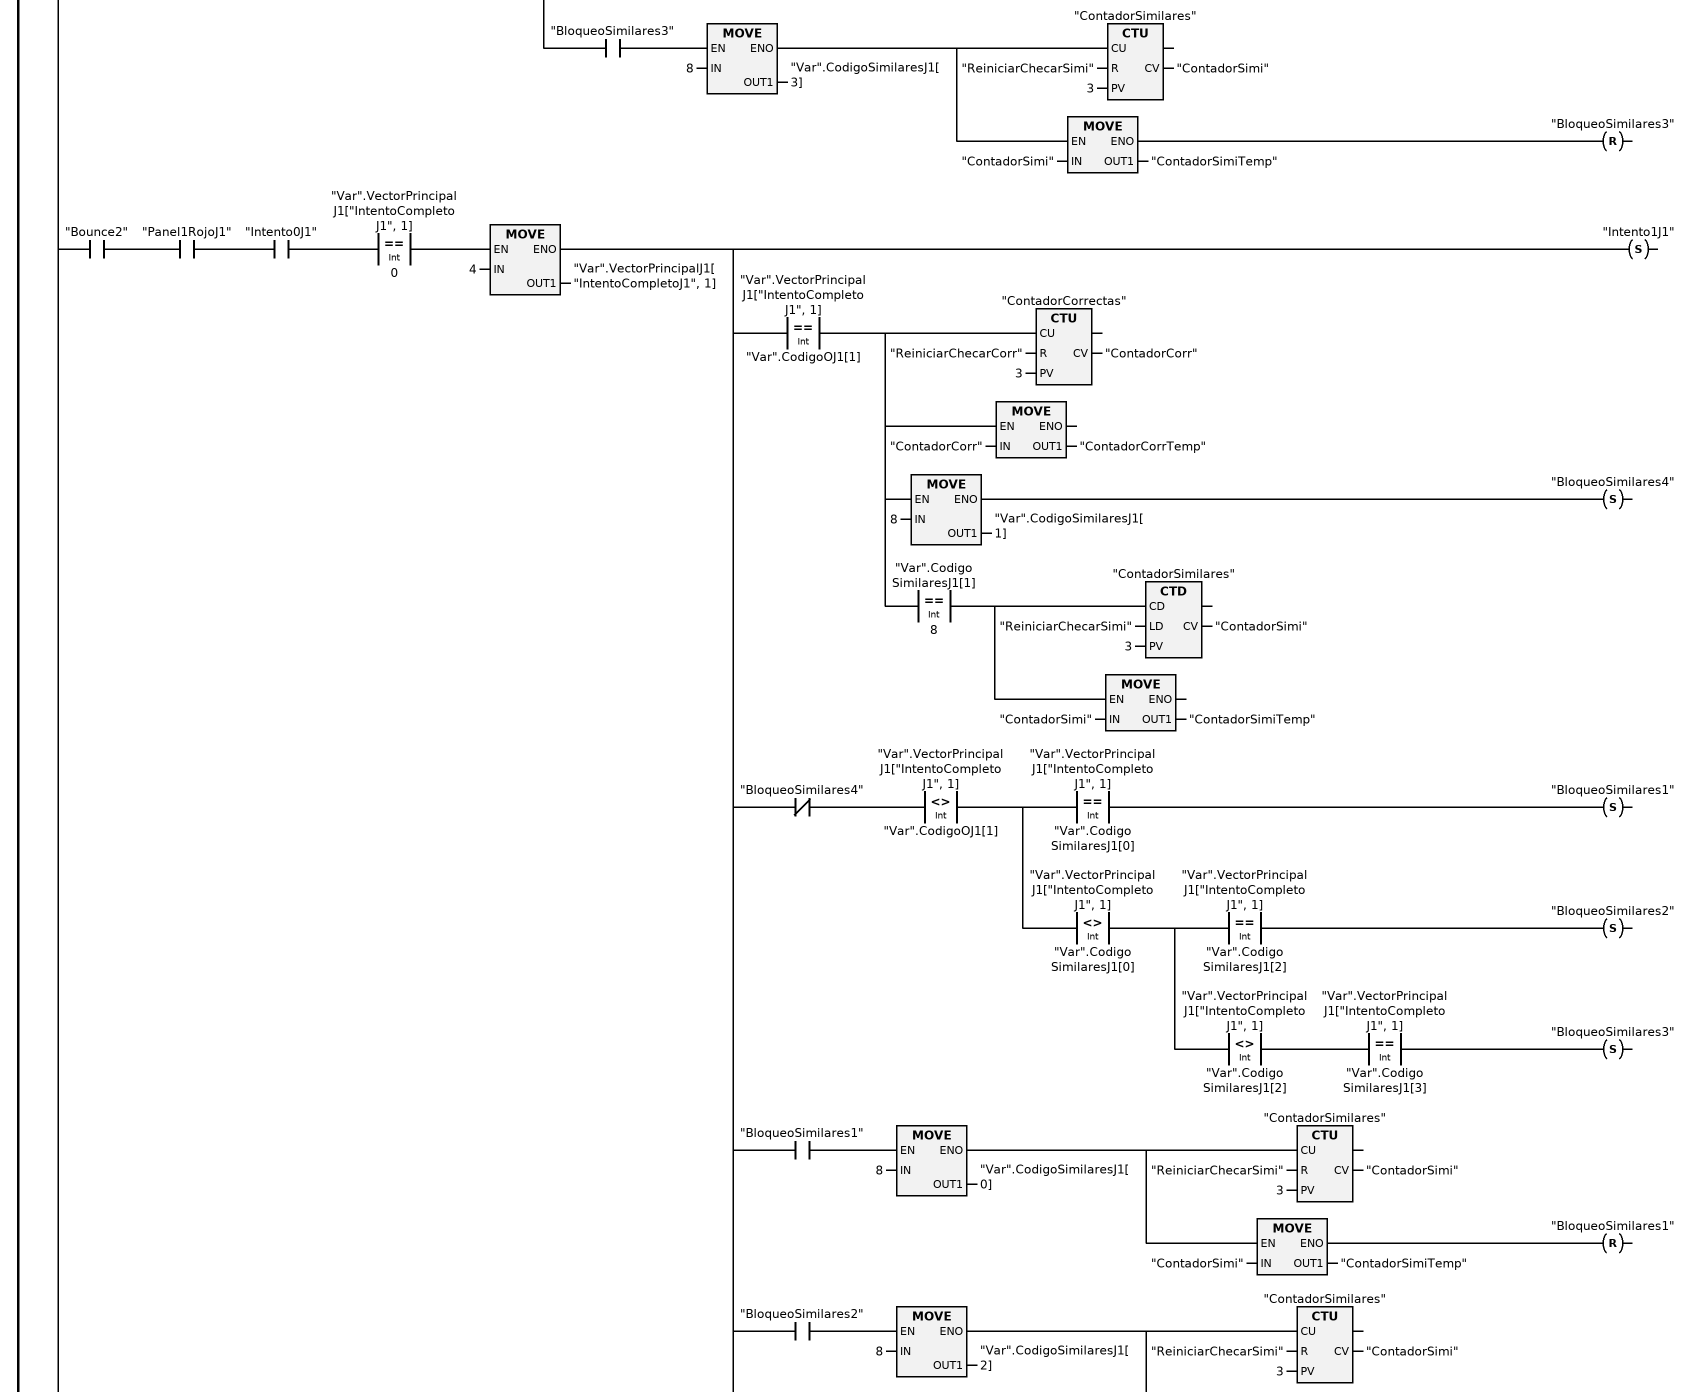
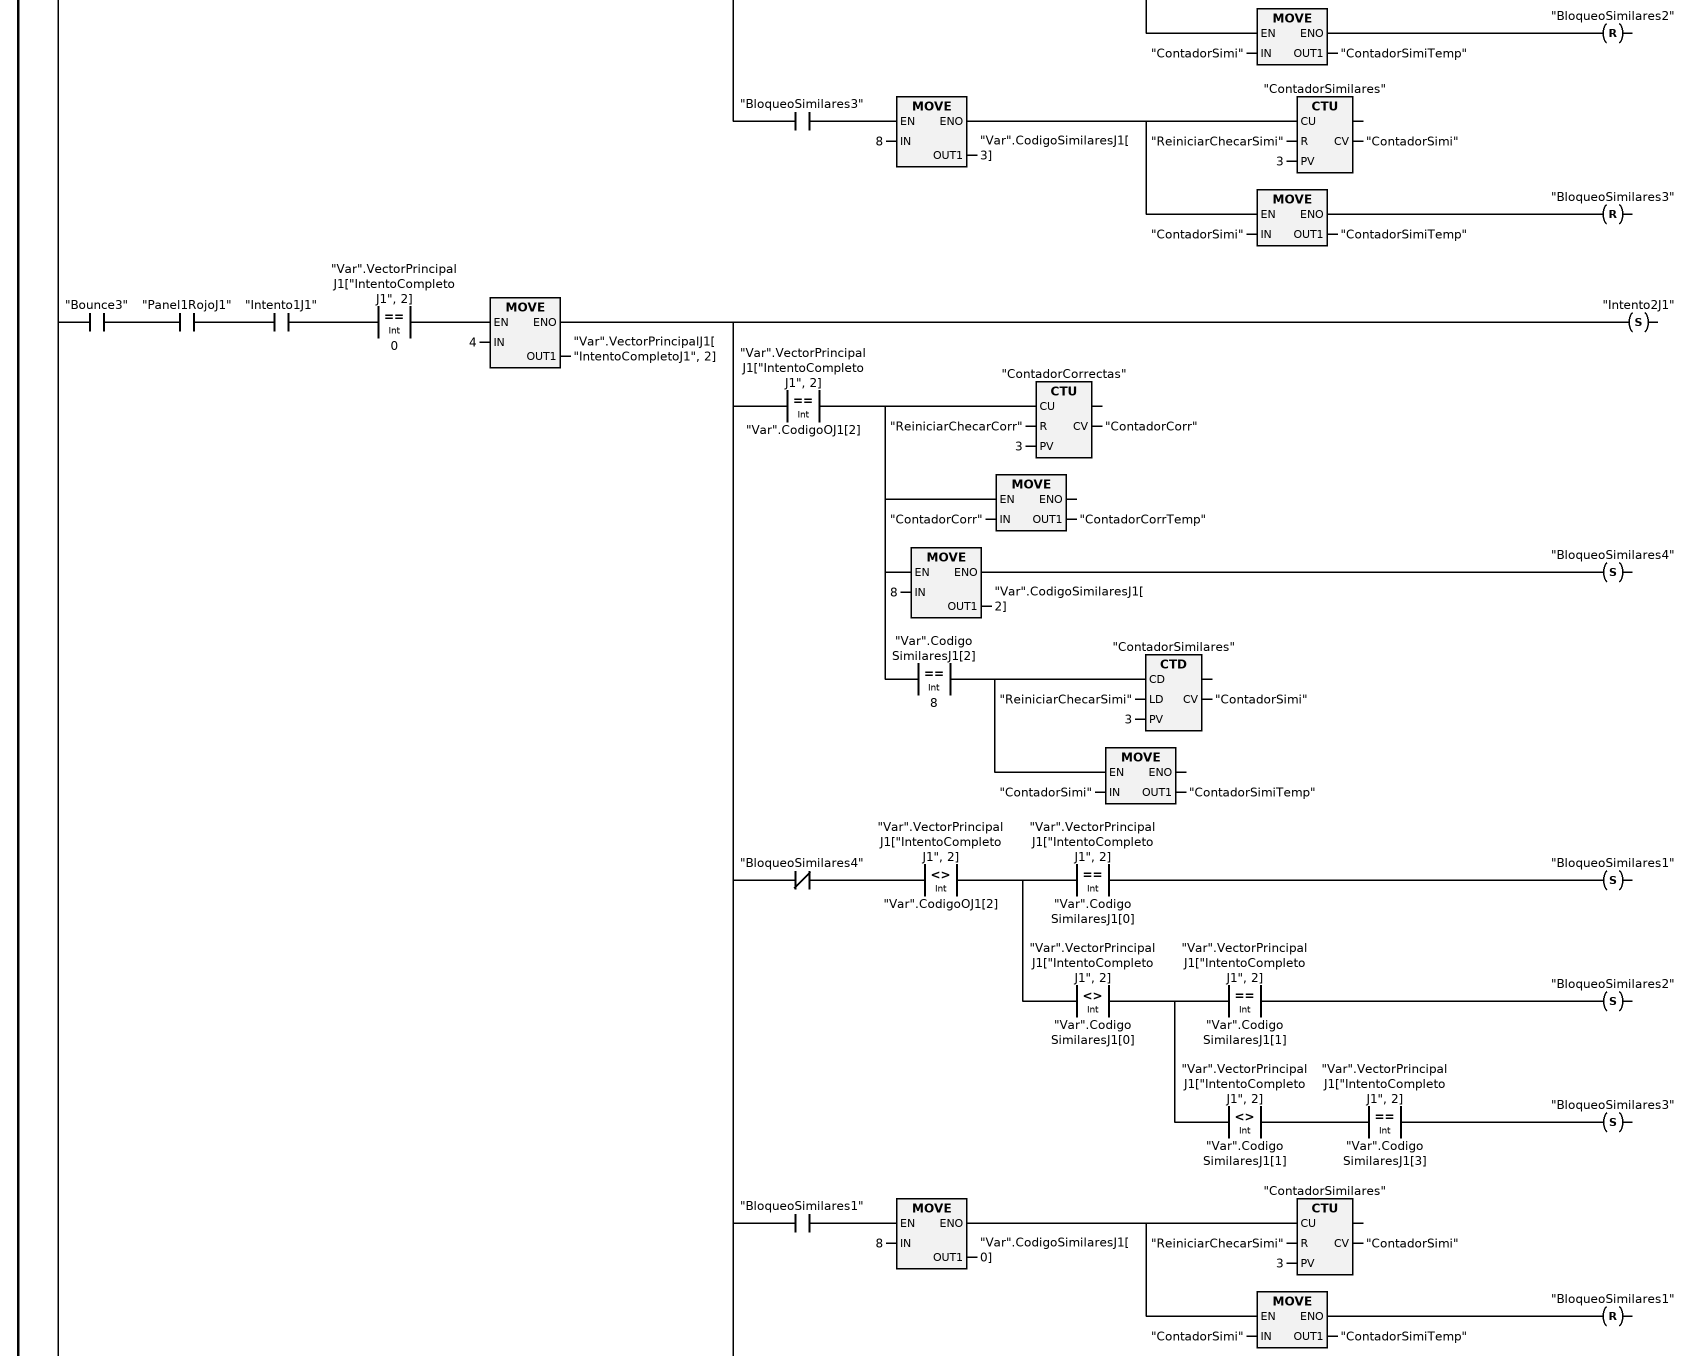
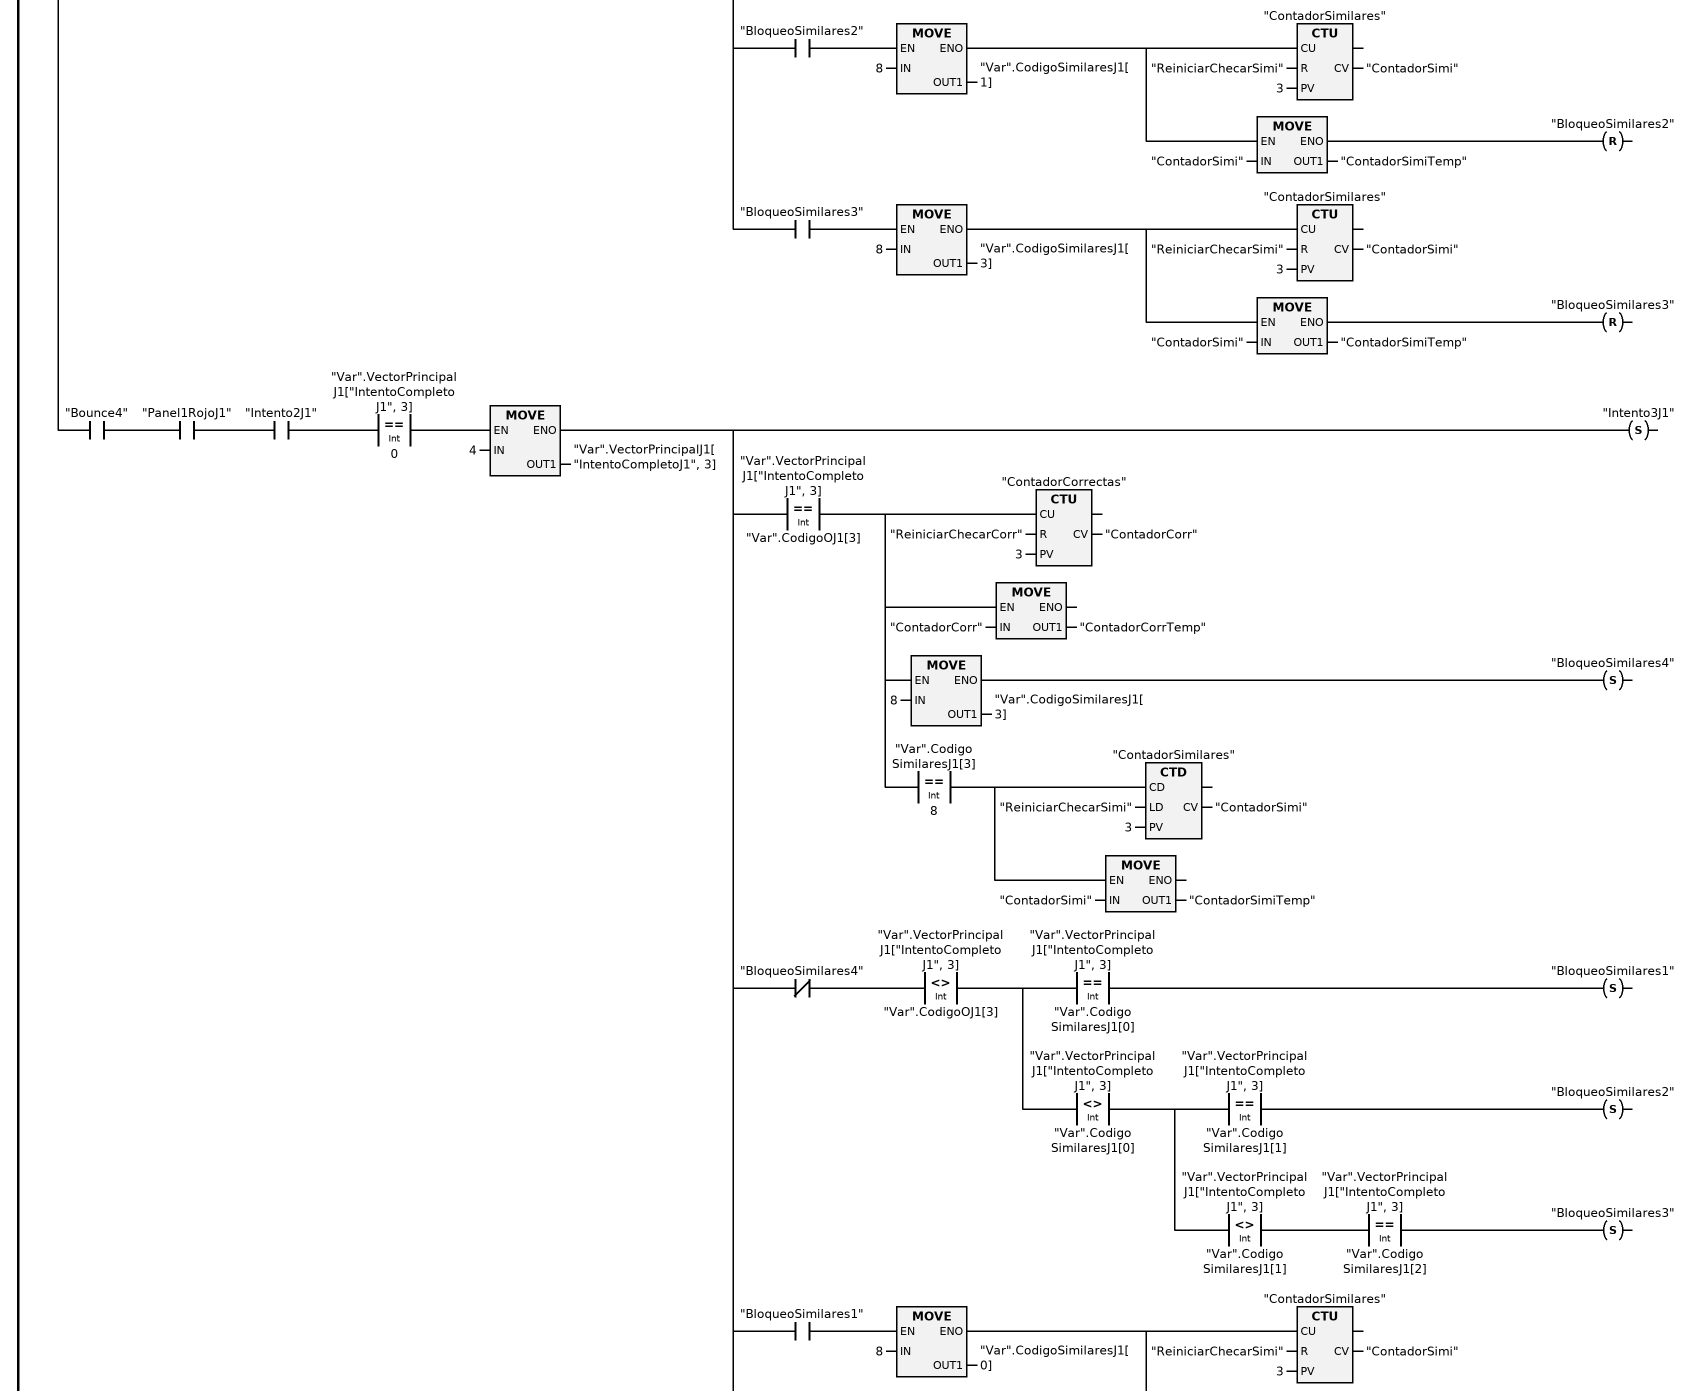
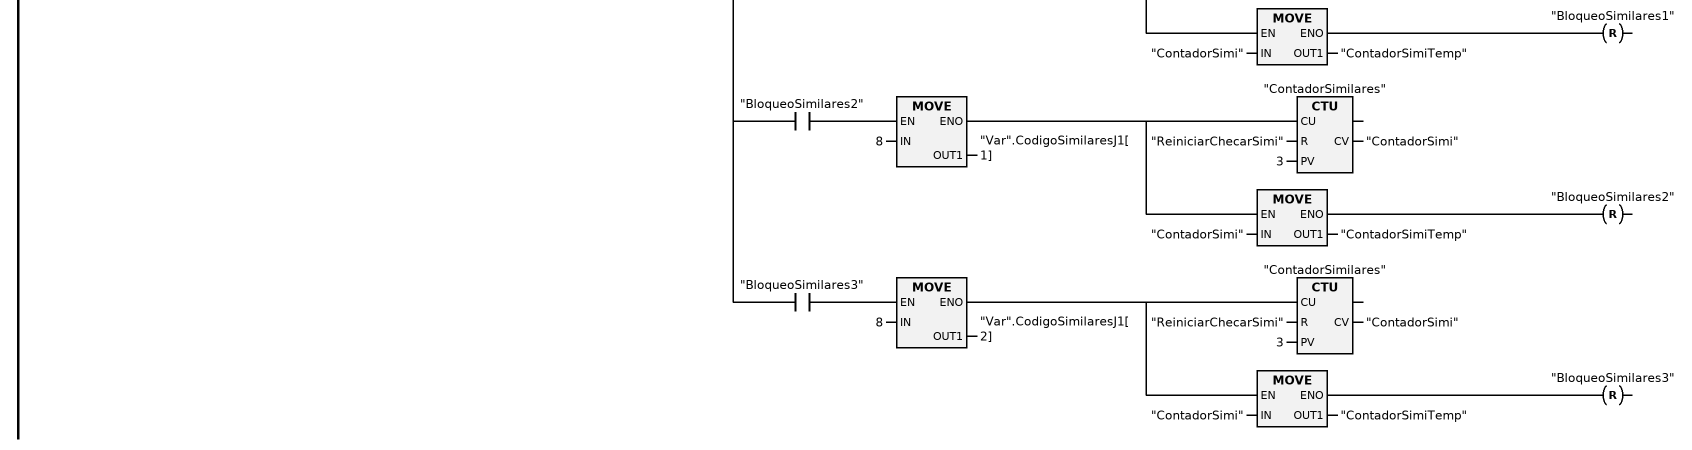
   #_w1 := "Panel1RojoJ1" AND ("Var".VectorPrincipalJ1["IntentoCompletoJ1", 0] = 0) AND "Bounce1";
   IF #_w1 THEN
       "Var".VectorPrincipalJ1["IntentoCompletoJ1", 0] := 4;
       "Intento0J1" := TRUE;
   END_IF;
   #_w2 := #_w1 AND ("Var".VectorPrincipalJ1["IntentoCompletoJ1", 0] = "Var".CodigoOJ1[0]);
   "ContadorCorrectas".CTU(CU := #_w2, R := "ReiniciarChecarCorr", PV := 3, CV => "ContadorCorr");
   IF #_w2 THEN
       "ContadorCorrTemp" := "ContadorCorr";
       "Var".CodigoSimilaresJ1[0] := 8;
       "BloqueoSimilares4" := TRUE;
   END_IF;
   #_w3 := #_w2 AND ("Var".CodigoSimilaresJ1[0] = 8);
   "ContadorSimilares".CTD(CD := #_w3, LD := "ReiniciarChecarSimi", PV := 3, CV => "ContadorSimi");
   IF #_w3 THEN "ContadorSimiTemp" := "ContadorSimi"; END_IF;
   #_w4 := #_w1 AND NOT "BloqueoSimilares4" AND ("Var".VectorPrincipalJ1["IntentoCompletoJ1", 0] <> "Var".CodigoOJ1[0]);
   IF #_w4 AND ("Var".VectorPrincipalJ1["IntentoCompletoJ1", 0] = "Var".CodigoSimilaresJ1[1]) THEN
       "BloqueoSimilares1" := TRUE;
   END_IF;
   #_w5 := #_w4 AND ("Var".VectorPrincipalJ1["IntentoCompletoJ1", 0] <> "Var".CodigoSimilaresJ1[1]);
   IF #_w5 AND ("Var".VectorPrincipalJ1["IntentoCompletoJ1", 0] = "Var".CodigoSimilaresJ1[2]) THEN
       "BloqueoSimilares2" := TRUE;
   END_IF;
   IF #_w5 AND ("Var".VectorPrincipalJ1["IntentoCompletoJ1", 0] <> "Var".CodigoSimilaresJ1[2]) AND ("Var".VectorPrincipalJ1["IntentoCompletoJ1", 0] = "Var".CodigoSimilaresJ1[3]) THEN
       "BloqueoSimilares3" := TRUE;
   END_IF;
   #_w6 := #_w1 AND "BloqueoSimilares1";
   IF #_w6 THEN "Var".CodigoSimilaresJ1[1] := 8; END_IF;
   "ContadorSimilares".CTU(CU := #_w6, R := "ReiniciarChecarSimi", PV := 3, CV => "ContadorSimi");
   IF #_w6 THEN
       "ContadorSimiTemp" := "ContadorSimi";
       "BloqueoSimilares1" := FALSE;
   END_IF;
   #_w7 := #_w1 AND "BloqueoSimilares2";
   IF #_w7 THEN "Var".CodigoSimilaresJ1[2] := 8; END_IF;
   "ContadorSimilares".CTU(CU := #_w7, R := "ReiniciarChecarSimi", PV := 3, CV => "ContadorSimi");
   IF #_w7 THEN
       "ContadorSimiTemp" := "ContadorSimi";
       "BloqueoSimilares2" := FALSE;
   END_IF;
   #_w8 := #_w1 AND "BloqueoSimilares3";
   IF #_w8 THEN "Var".CodigoSimilaresJ1[3] := 8; END_IF;
   "ContadorSimilares".CTU(CU := #_w8, R := "ReiniciarChecarSimi", PV := 3, CV => "ContadorSimi");
   IF #_w8 THEN
       "ContadorSimiTemp" := "ContadorSimi";
       "BloqueoSimilares3" := FALSE;
   END_IF;
   #_w9 := "Panel1RojoJ1" AND "Bounce2" AND "Panel1RojoJ1" AND "Intento0J1" AND ("Var".VectorPrincipalJ1["IntentoCompletoJ1", 1] = 0);
   IF #_w9 THEN
       "Var".VectorPrincipalJ1["IntentoCompletoJ1", 1] := 4;
       "Intento1J1" := TRUE;
   END_IF;
   #_w10 := #_w9 AND ("Var".VectorPrincipalJ1["IntentoCompletoJ1", 1] = "Var".CodigoOJ1[1]);
   "ContadorCorrectas".CTU(CU := #_w10, R := "ReiniciarChecarCorr", PV := 3, CV => "ContadorCorr");
   IF #_w10 THEN
       "ContadorCorrTemp" := "ContadorCorr";
       "Var".CodigoSimilaresJ1[1] := 8;
       "BloqueoSimilares4" := TRUE;
   END_IF;
   #_w11 := #_w10 AND ("Var".CodigoSimilaresJ1[1] = 8);
   "ContadorSimilares".CTD(CD := #_w11, LD := "ReiniciarChecarSimi", PV := 3, CV => "ContadorSimi");
   IF #_w11 THEN "ContadorSimiTemp" := "ContadorSimi"; END_IF;
   #_w12 := #_w9 AND NOT "BloqueoSimilares4" AND ("Var".VectorPrincipalJ1["IntentoCompletoJ1", 1] <> "Var".CodigoOJ1[1]);
   IF #_w12 AND ("Var".VectorPrincipalJ1["IntentoCompletoJ1", 1] = "Var".CodigoSimilaresJ1[0]) THEN
       "BloqueoSimilares1" := TRUE;
   END_IF;
   #_w13 := #_w12 AND ("Var".VectorPrincipalJ1["IntentoCompletoJ1", 1] <> "Var".CodigoSimilaresJ1[0]);
   IF #_w13 AND ("Var".VectorPrincipalJ1["IntentoCompletoJ1", 1] = "Var".CodigoSimilaresJ1[2]) THEN
       "BloqueoSimilares2" := TRUE;
   END_IF;
   IF #_w13 AND ("Var".VectorPrincipalJ1["IntentoCompletoJ1", 1] <> "Var".CodigoSimilaresJ1[2]) AND ("Var".VectorPrincipalJ1["IntentoCompletoJ1", 1] = "Var".CodigoSimilaresJ1[3]) THEN
       "BloqueoSimilares3" := TRUE;
   END_IF;
   #_w14 := #_w9 AND "BloqueoSimilares1";
   IF #_w14 THEN "Var".CodigoSimilaresJ1[0] := 8; END_IF;
   "ContadorSimilares".CTU(CU := #_w14, R := "ReiniciarChecarSimi", PV := 3, CV => "ContadorSimi");
   IF #_w14 THEN
       "ContadorSimiTemp" := "ContadorSimi";
       "BloqueoSimilares1" := FALSE;
   END_IF;
   #_w15 := #_w9 AND "BloqueoSimilares2";
   IF #_w15 THEN "Var".CodigoSimilaresJ1[2] := 8; END_IF;
   "ContadorSimilares".CTU(CU := #_w15, R := "ReiniciarChecarSimi", PV := 3, CV => "ContadorSimi");
   IF #_w15 THEN
       "ContadorSimiTemp" := "ContadorSimi";
       "BloqueoSimilares2" := FALSE;
   END_IF;
   #_w16 := #_w9 AND "BloqueoSimilares3";
   IF #_w16 THEN "Var".CodigoSimilaresJ1[3] := 8; END_IF;
   "ContadorSimilares".CTU(CU := #_w16, R := "ReiniciarChecarSimi", PV := 3, CV => "ContadorSimi");
   IF #_w16 THEN
       "ContadorSimiTemp" := "ContadorSimi";
       "BloqueoSimilares3" := FALSE;
   END_IF;
   #_w17 := "Panel1RojoJ1" AND "Bounce3" AND "Panel1RojoJ1" AND "Intento1J1" AND ("Var".VectorPrincipalJ1["IntentoCompletoJ1", 2] = 0);
   IF #_w17 THEN
       "Var".VectorPrincipalJ1["IntentoCompletoJ1", 2] := 4;
       "Intento2J1" := TRUE;
   END_IF;
   #_w18 := #_w17 AND ("Var".VectorPrincipalJ1["IntentoCompletoJ1", 2] = "Var".CodigoOJ1[2]);
   "ContadorCorrectas".CTU(CU := #_w18, R := "ReiniciarChecarCorr", PV := 3, CV => "ContadorCorr");
   IF #_w18 THEN
       "ContadorCorrTemp" := "ContadorCorr";
       "Var".CodigoSimilaresJ1[2] := 8;
       "BloqueoSimilares4" := TRUE;
   END_IF;
   #_w19 := #_w18 AND ("Var".CodigoSimilaresJ1[2] = 8);
   "ContadorSimilares".CTD(CD := #_w19, LD := "ReiniciarChecarSimi", PV := 3, CV => "ContadorSimi");
   IF #_w19 THEN "ContadorSimiTemp" := "ContadorSimi"; END_IF;
   #_w20 := #_w17 AND NOT "BloqueoSimilares4" AND ("Var".VectorPrincipalJ1["IntentoCompletoJ1", 2] <> "Var".CodigoOJ1[2]);
   IF #_w20 AND ("Var".VectorPrincipalJ1["IntentoCompletoJ1", 2] = "Var".CodigoSimilaresJ1[0]) THEN
       "BloqueoSimilares1" := TRUE;
   END_IF;
   #_w21 := #_w20 AND ("Var".VectorPrincipalJ1["IntentoCompletoJ1", 2] <> "Var".CodigoSimilaresJ1[0]);
   IF #_w21 AND ("Var".VectorPrincipalJ1["IntentoCompletoJ1", 2] = "Var".CodigoSimilaresJ1[1]) THEN
       "BloqueoSimilares2" := TRUE;
   END_IF;
   IF #_w21 AND ("Var".VectorPrincipalJ1["IntentoCompletoJ1", 2] <> "Var".CodigoSimilaresJ1[1]) AND ("Var".VectorPrincipalJ1["IntentoCompletoJ1", 2] = "Var".CodigoSimilaresJ1[3]) THEN
       "BloqueoSimilares3" := TRUE;
   END_IF;
   #_w22 := #_w17 AND "BloqueoSimilares1";
   IF #_w22 THEN "Var".CodigoSimilaresJ1[0] := 8; END_IF;
   "ContadorSimilares".CTU(CU := #_w22, R := "ReiniciarChecarSimi", PV := 3, CV => "ContadorSimi");
   IF #_w22 THEN
       "ContadorSimiTemp" := "ContadorSimi";
       "BloqueoSimilares1" := FALSE;
   END_IF;
   #_w23 := #_w17 AND "BloqueoSimilares2";
   IF #_w23 THEN "Var".CodigoSimilaresJ1[1] := 8; END_IF;
   "ContadorSimilares".CTU(CU := #_w23, R := "ReiniciarChecarSimi", PV := 3, CV => "ContadorSimi");
   IF #_w23 THEN
       "ContadorSimiTemp" := "ContadorSimi";
       "BloqueoSimilares2" := FALSE;
   END_IF;
   #_w24 := #_w17 AND "BloqueoSimilares3";
   IF #_w24 THEN "Var".CodigoSimilaresJ1[3] := 8; END_IF;
   "ContadorSimilares".CTU(CU := #_w24, R := "ReiniciarChecarSimi", PV := 3, CV => "ContadorSimi");
   IF #_w24 THEN
       "ContadorSimiTemp" := "ContadorSimi";
       "BloqueoSimilares3" := FALSE;
   END_IF;
   #_w25 := "Panel1RojoJ1" AND "Bounce4" AND "Panel1RojoJ1" AND "Intento2J1" AND ("Var".VectorPrincipalJ1["IntentoCompletoJ1", 3] = 0);
   IF #_w25 THEN
       "Var".VectorPrincipalJ1["IntentoCompletoJ1", 3] := 4;
       "Intento3J1" := TRUE;
   END_IF;
   #_w26 := #_w25 AND ("Var".VectorPrincipalJ1["IntentoCompletoJ1", 3] = "Var".CodigoOJ1[3]);
   "ContadorCorrectas".CTU(CU := #_w26, R := "ReiniciarChecarCorr", PV := 3, CV => "ContadorCorr");
   IF #_w26 THEN
       "ContadorCorrTemp" := "ContadorCorr";
       "Var".CodigoSimilaresJ1[3] := 8;
       "BloqueoSimilares4" := TRUE;
   END_IF;
   #_w27 := #_w26 AND ("Var".CodigoSimilaresJ1[3] = 8);
   "ContadorSimilares".CTD(CD := #_w27, LD := "ReiniciarChecarSimi", PV := 3, CV => "ContadorSimi");
   IF #_w27 THEN "ContadorSimiTemp" := "ContadorSimi"; END_IF;
   #_w28 := #_w25 AND NOT "BloqueoSimilares4" AND ("Var".VectorPrincipalJ1["IntentoCompletoJ1", 3] <> "Var".CodigoOJ1[3]);
   IF #_w28 AND ("Var".VectorPrincipalJ1["IntentoCompletoJ1", 3] = "Var".CodigoSimilaresJ1[0]) THEN
       "BloqueoSimilares1" := TRUE;
   END_IF;
   #_w29 := #_w28 AND ("Var".VectorPrincipalJ1["IntentoCompletoJ1", 3] <> "Var".CodigoSimilaresJ1[0]);
   IF #_w29 AND ("Var".VectorPrincipalJ1["IntentoCompletoJ1", 3] = "Var".CodigoSimilaresJ1[1]) THEN
       "BloqueoSimilares2" := TRUE;
   END_IF;
   IF #_w29 AND ("Var".VectorPrincipalJ1["IntentoCompletoJ1", 3] <> "Var".CodigoSimilaresJ1[1]) AND ("Var".VectorPrincipalJ1["IntentoCompletoJ1", 3] = "Var".CodigoSimilaresJ1[2]) THEN
       "BloqueoSimilares3" := TRUE;
   END_IF;
   #_w30 := #_w25 AND "BloqueoSimilares1";
   IF #_w30 THEN "Var".CodigoSimilaresJ1[0] := 8; END_IF;
   "ContadorSimilares".CTU(CU := #_w30, R := "ReiniciarChecarSimi", PV := 3, CV => "ContadorSimi");
   IF #_w30 THEN
       "ContadorSimiTemp" := "ContadorSimi";
       "BloqueoSimilares1" := FALSE;
   END_IF;
   #_w31 := #_w25 AND "BloqueoSimilares2";
   IF #_w31 THEN "Var".CodigoSimilaresJ1[1] := 8; END_IF;
   "ContadorSimilares".CTU(CU := #_w31, R := "ReiniciarChecarSimi", PV := 3, CV => "ContadorSimi");
   IF #_w31 THEN
       "ContadorSimiTemp" := "ContadorSimi";
       "BloqueoSimilares2" := FALSE;
   END_IF;
   #_w32 := #_w25 AND "BloqueoSimilares3";
   IF #_w32 THEN "Var".CodigoSimilaresJ1[2] := 8; END_IF;
   "ContadorSimilares".CTU(CU := #_w32, R := "ReiniciarChecarSimi", PV := 3, CV => "ContadorSimi");
   IF #_w32 THEN
       "ContadorSimiTemp" := "ContadorSimi";
       "BloqueoSimilares3" := FALSE;
   END_IF;
END_REGION

REGION Network 10: Azul
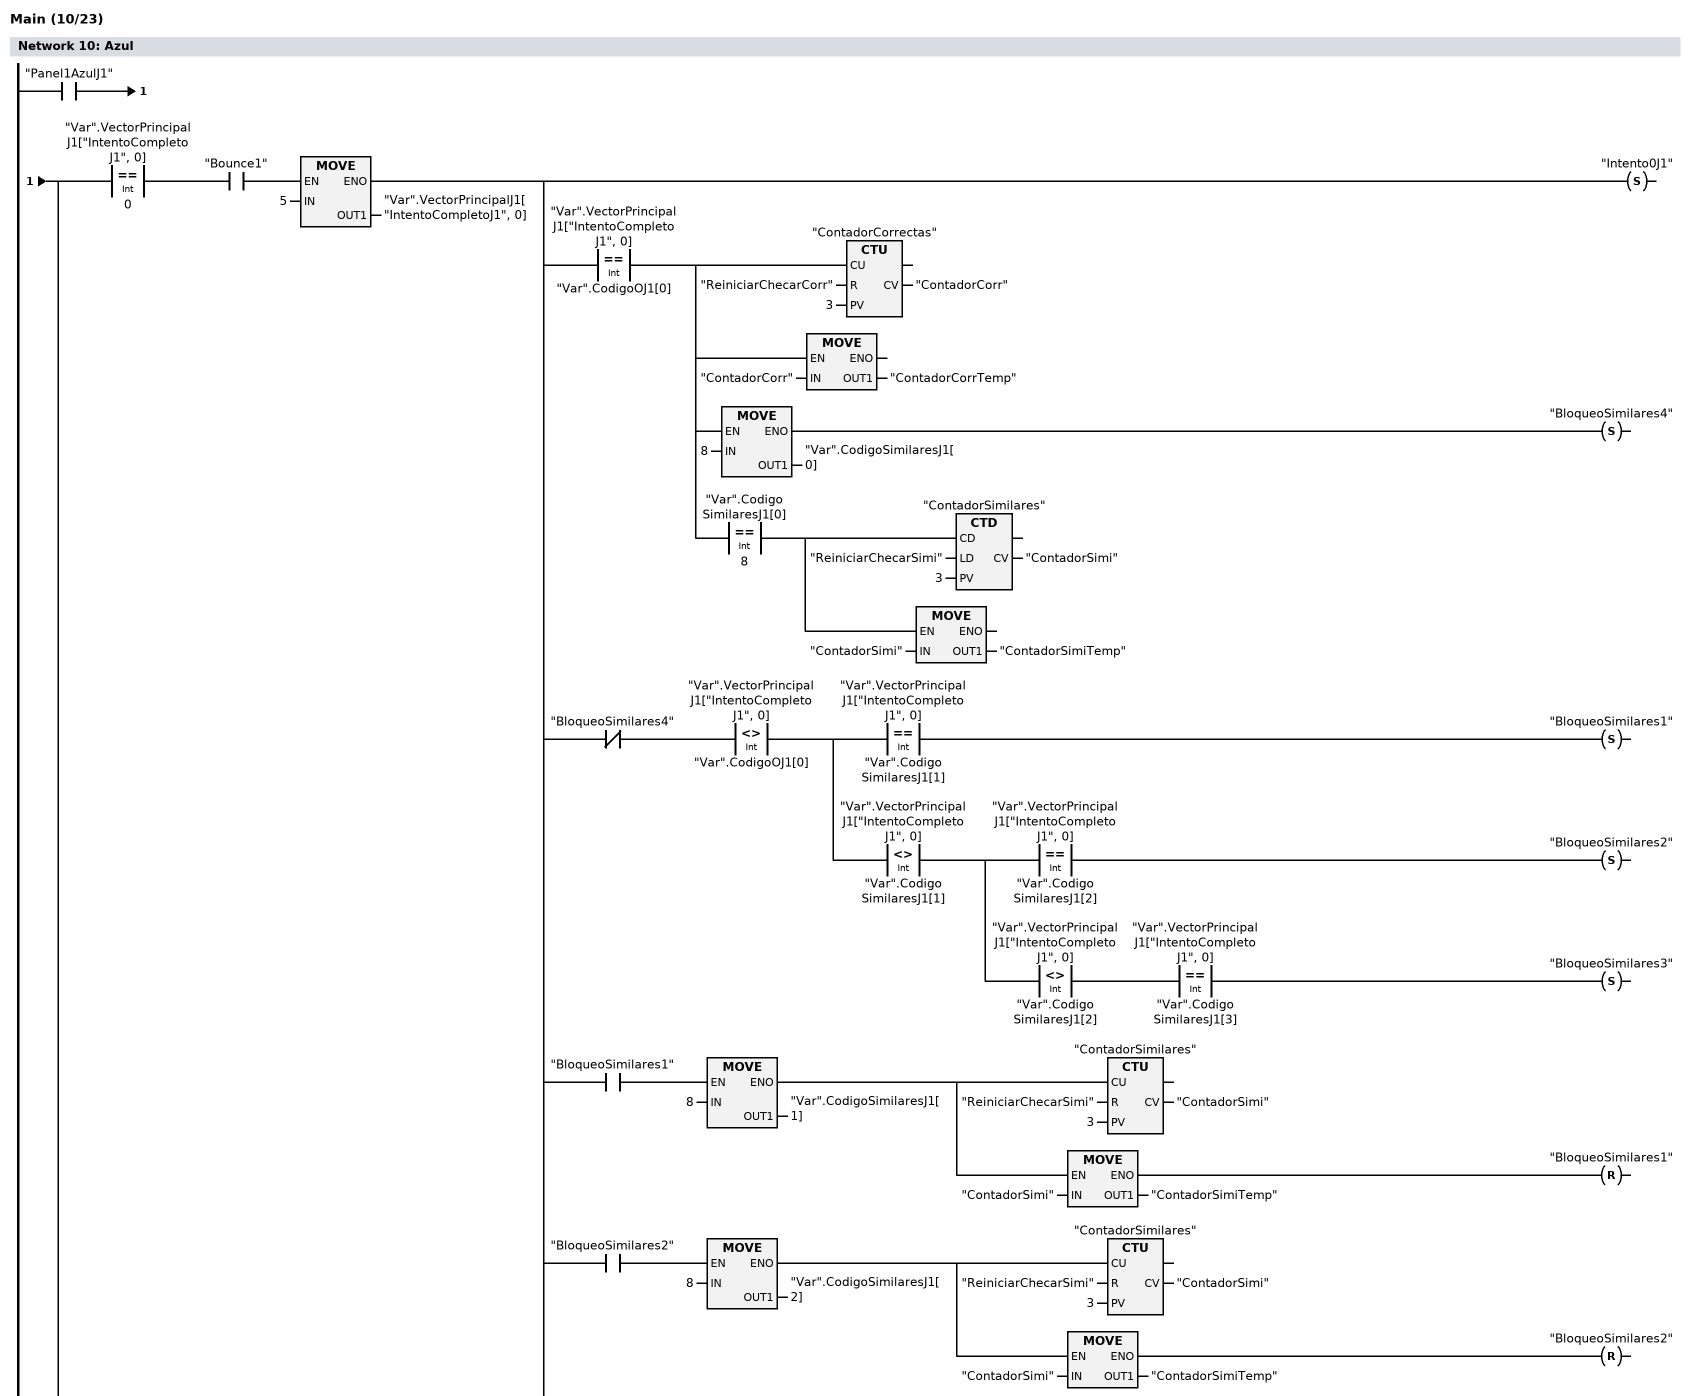
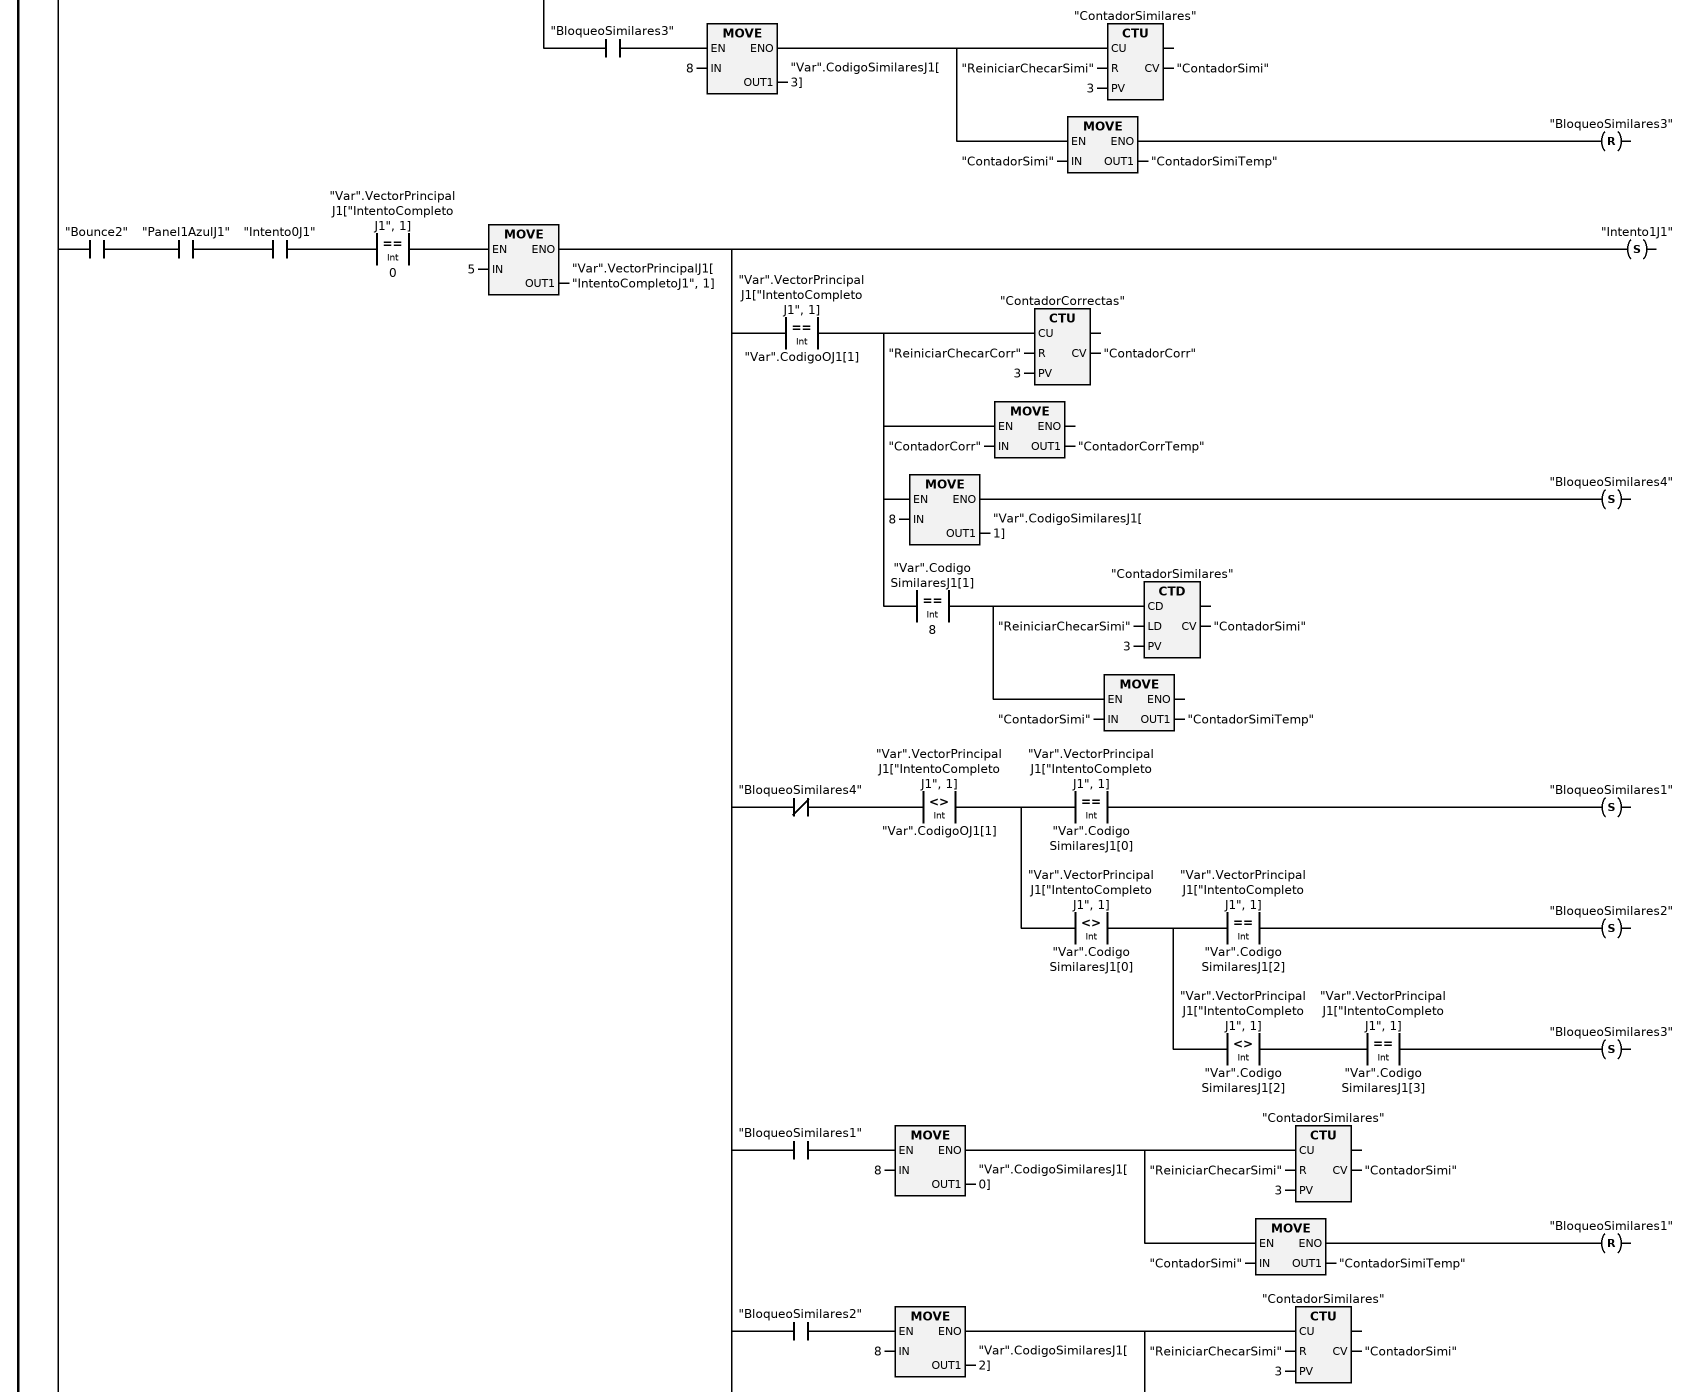
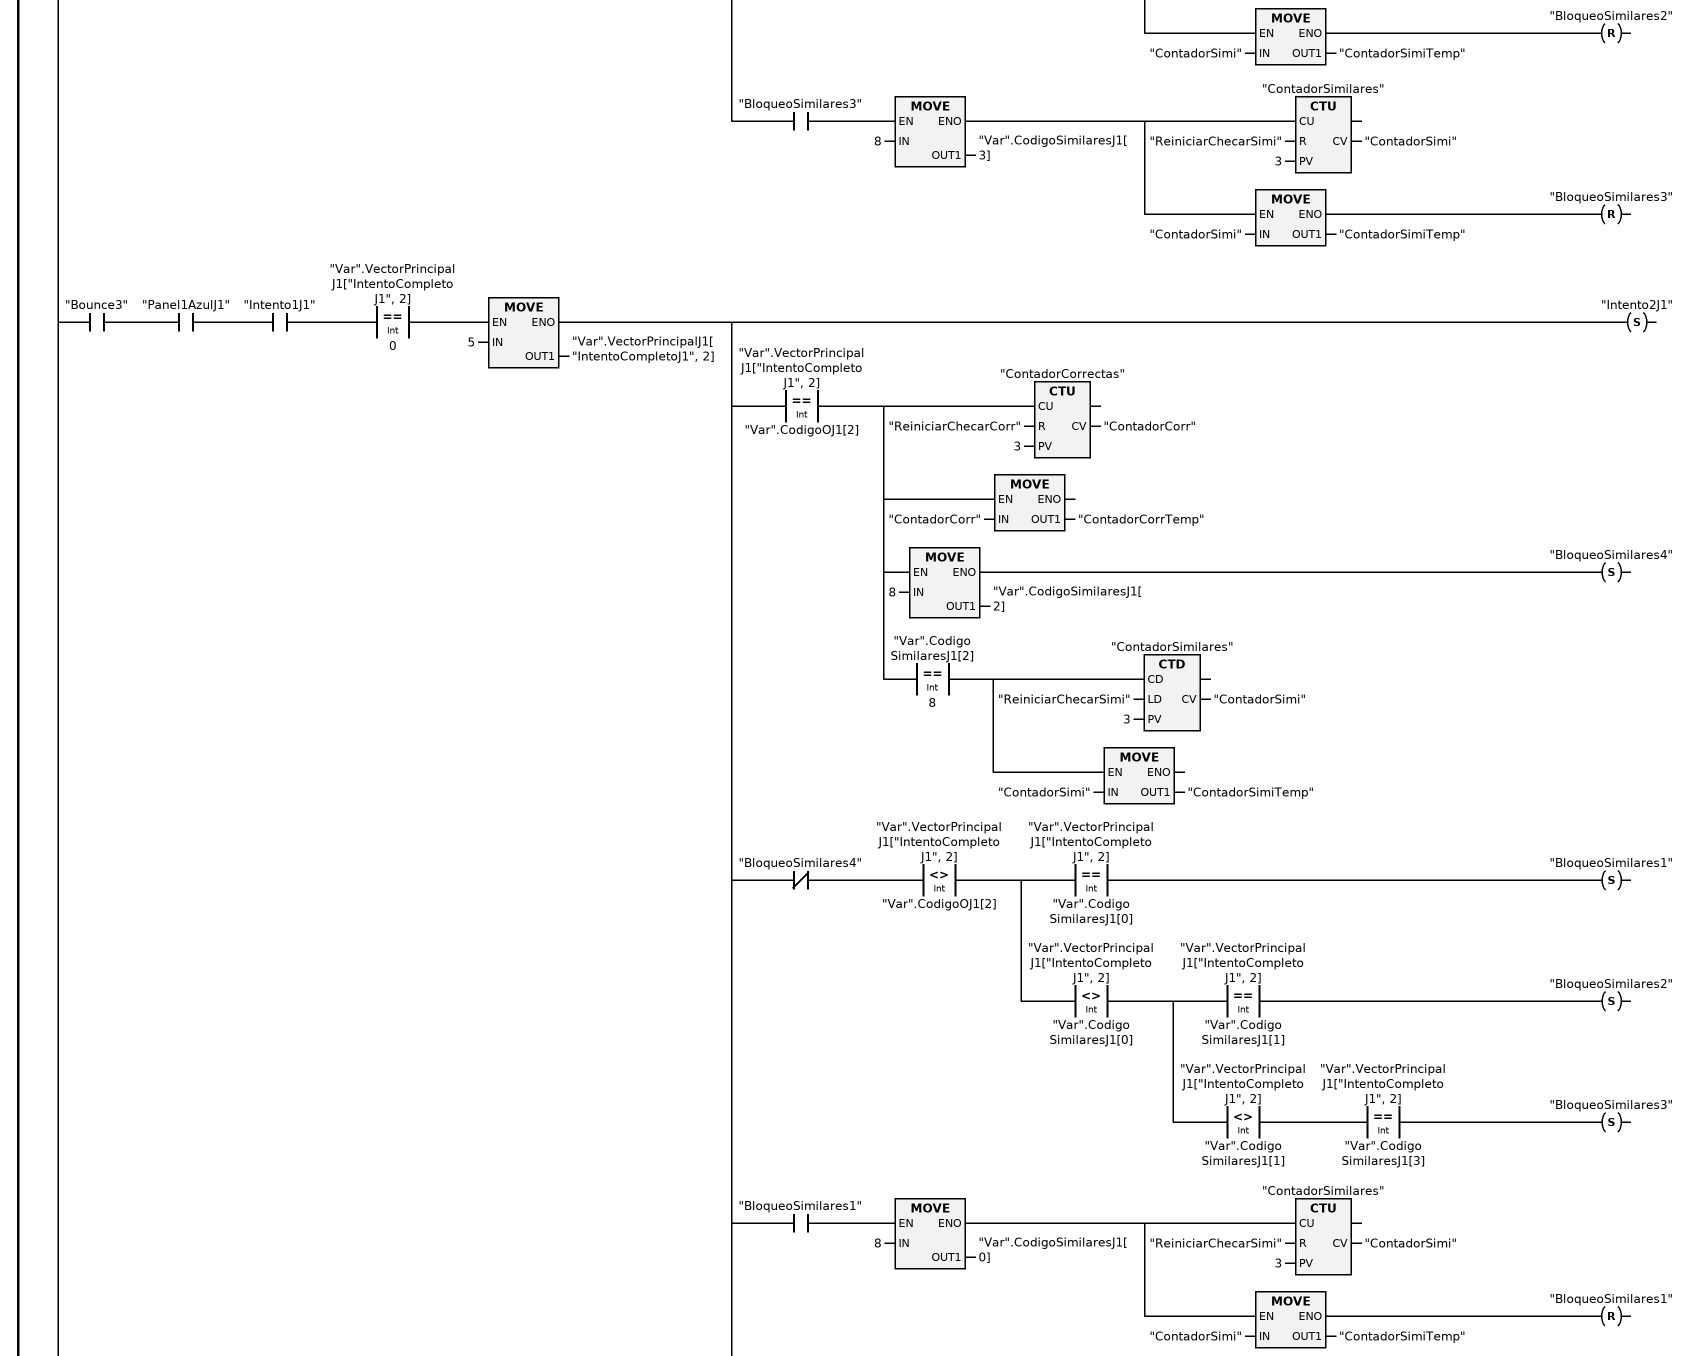
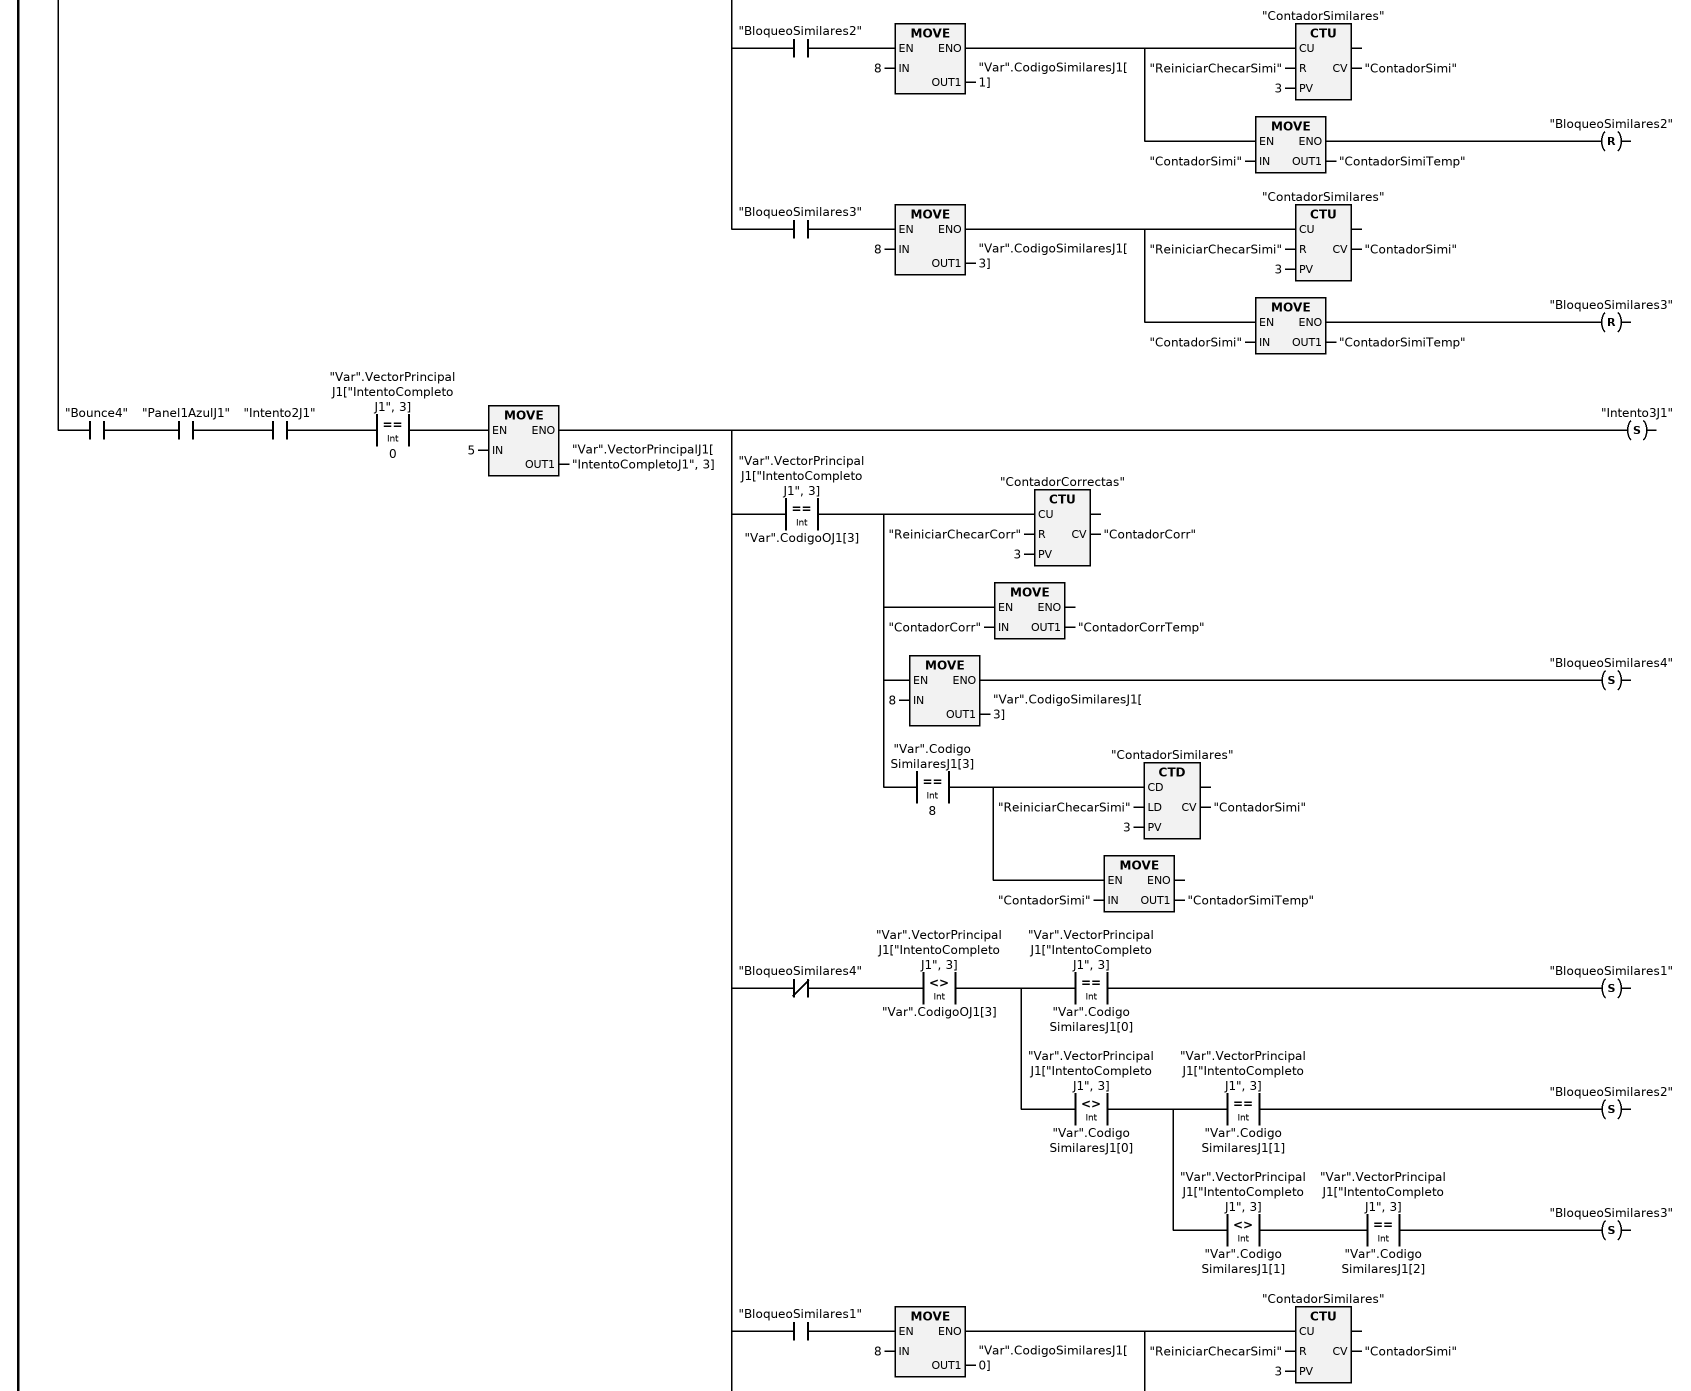
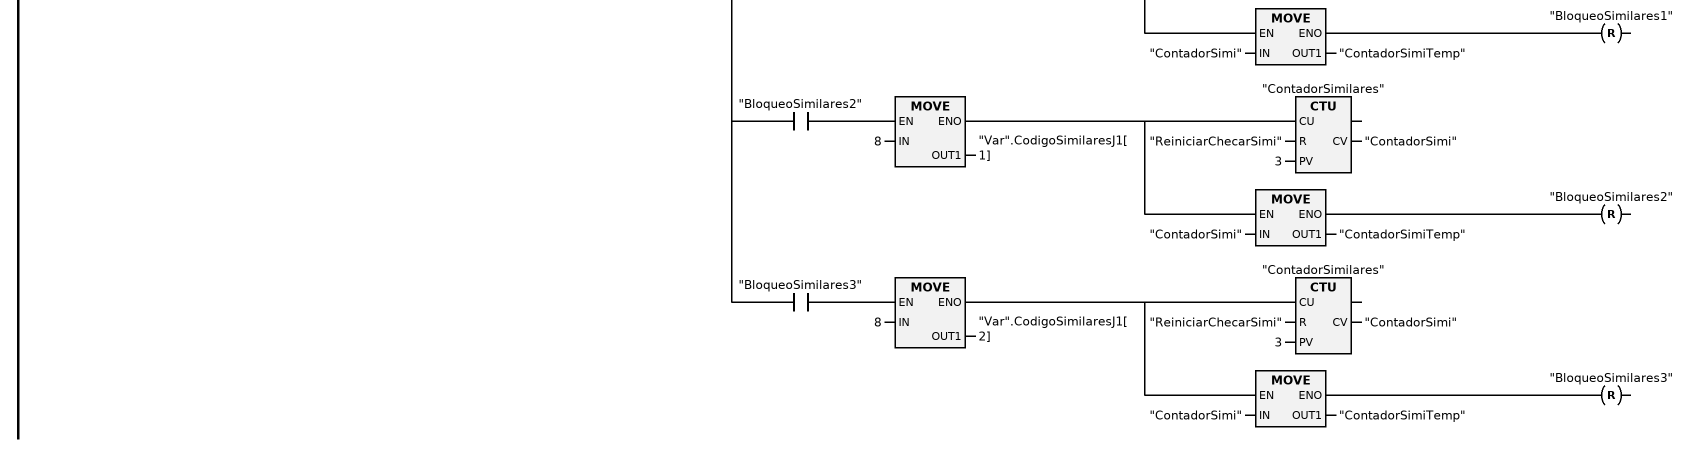
   #_w1 := "Panel1AzulJ1" AND ("Var".VectorPrincipalJ1["IntentoCompletoJ1", 0] = 0) AND "Bounce1";
   IF #_w1 THEN
       "Var".VectorPrincipalJ1["IntentoCompletoJ1", 0] := 5;
       "Intento0J1" := TRUE;
   END_IF;
   #_w2 := #_w1 AND ("Var".VectorPrincipalJ1["IntentoCompletoJ1", 0] = "Var".CodigoOJ1[0]);
   "ContadorCorrectas".CTU(CU := #_w2, R := "ReiniciarChecarCorr", PV := 3, CV => "ContadorCorr");
   IF #_w2 THEN
       "ContadorCorrTemp" := "ContadorCorr";
       "Var".CodigoSimilaresJ1[0] := 8;
       "BloqueoSimilares4" := TRUE;
   END_IF;
   #_w3 := #_w2 AND ("Var".CodigoSimilaresJ1[0] = 8);
   "ContadorSimilares".CTD(CD := #_w3, LD := "ReiniciarChecarSimi", PV := 3, CV => "ContadorSimi");
   IF #_w3 THEN "ContadorSimiTemp" := "ContadorSimi"; END_IF;
   #_w4 := #_w1 AND NOT "BloqueoSimilares4" AND ("Var".VectorPrincipalJ1["IntentoCompletoJ1", 0] <> "Var".CodigoOJ1[0]);
   IF #_w4 AND ("Var".VectorPrincipalJ1["IntentoCompletoJ1", 0] = "Var".CodigoSimilaresJ1[1]) THEN
       "BloqueoSimilares1" := TRUE;
   END_IF;
   #_w5 := #_w4 AND ("Var".VectorPrincipalJ1["IntentoCompletoJ1", 0] <> "Var".CodigoSimilaresJ1[1]);
   IF #_w5 AND ("Var".VectorPrincipalJ1["IntentoCompletoJ1", 0] = "Var".CodigoSimilaresJ1[2]) THEN
       "BloqueoSimilares2" := TRUE;
   END_IF;
   IF #_w5 AND ("Var".VectorPrincipalJ1["IntentoCompletoJ1", 0] <> "Var".CodigoSimilaresJ1[2]) AND ("Var".VectorPrincipalJ1["IntentoCompletoJ1", 0] = "Var".CodigoSimilaresJ1[3]) THEN
       "BloqueoSimilares3" := TRUE;
   END_IF;
   #_w6 := #_w1 AND "BloqueoSimilares1";
   IF #_w6 THEN "Var".CodigoSimilaresJ1[1] := 8; END_IF;
   "ContadorSimilares".CTU(CU := #_w6, R := "ReiniciarChecarSimi", PV := 3, CV => "ContadorSimi");
   IF #_w6 THEN
       "ContadorSimiTemp" := "ContadorSimi";
       "BloqueoSimilares1" := FALSE;
   END_IF;
   #_w7 := #_w1 AND "BloqueoSimilares2";
   IF #_w7 THEN "Var".CodigoSimilaresJ1[2] := 8; END_IF;
   "ContadorSimilares".CTU(CU := #_w7, R := "ReiniciarChecarSimi", PV := 3, CV => "ContadorSimi");
   IF #_w7 THEN
       "ContadorSimiTemp" := "ContadorSimi";
       "BloqueoSimilares2" := FALSE;
   END_IF;
   #_w8 := #_w1 AND "BloqueoSimilares3";
   IF #_w8 THEN "Var".CodigoSimilaresJ1[3] := 8; END_IF;
   "ContadorSimilares".CTU(CU := #_w8, R := "ReiniciarChecarSimi", PV := 3, CV => "ContadorSimi");
   IF #_w8 THEN
       "ContadorSimiTemp" := "ContadorSimi";
       "BloqueoSimilares3" := FALSE;
   END_IF;
   #_w9 := "Panel1AzulJ1" AND "Bounce2" AND "Panel1AzulJ1" AND "Intento0J1" AND ("Var".VectorPrincipalJ1["IntentoCompletoJ1", 1] = 0);
   IF #_w9 THEN
       "Var".VectorPrincipalJ1["IntentoCompletoJ1", 1] := 5;
       "Intento1J1" := TRUE;
   END_IF;
   #_w10 := #_w9 AND ("Var".VectorPrincipalJ1["IntentoCompletoJ1", 1] = "Var".CodigoOJ1[1]);
   "ContadorCorrectas".CTU(CU := #_w10, R := "ReiniciarChecarCorr", PV := 3, CV => "ContadorCorr");
   IF #_w10 THEN
       "ContadorCorrTemp" := "ContadorCorr";
       "Var".CodigoSimilaresJ1[1] := 8;
       "BloqueoSimilares4" := TRUE;
   END_IF;
   #_w11 := #_w10 AND ("Var".CodigoSimilaresJ1[1] = 8);
   "ContadorSimilares".CTD(CD := #_w11, LD := "ReiniciarChecarSimi", PV := 3, CV => "ContadorSimi");
   IF #_w11 THEN "ContadorSimiTemp" := "ContadorSimi"; END_IF;
   #_w12 := #_w9 AND NOT "BloqueoSimilares4" AND ("Var".VectorPrincipalJ1["IntentoCompletoJ1", 1] <> "Var".CodigoOJ1[1]);
   IF #_w12 AND ("Var".VectorPrincipalJ1["IntentoCompletoJ1", 1] = "Var".CodigoSimilaresJ1[0]) THEN
       "BloqueoSimilares1" := TRUE;
   END_IF;
   #_w13 := #_w12 AND ("Var".VectorPrincipalJ1["IntentoCompletoJ1", 1] <> "Var".CodigoSimilaresJ1[0]);
   IF #_w13 AND ("Var".VectorPrincipalJ1["IntentoCompletoJ1", 1] = "Var".CodigoSimilaresJ1[2]) THEN
       "BloqueoSimilares2" := TRUE;
   END_IF;
   IF #_w13 AND ("Var".VectorPrincipalJ1["IntentoCompletoJ1", 1] <> "Var".CodigoSimilaresJ1[2]) AND ("Var".VectorPrincipalJ1["IntentoCompletoJ1", 1] = "Var".CodigoSimilaresJ1[3]) THEN
       "BloqueoSimilares3" := TRUE;
   END_IF;
   #_w14 := #_w9 AND "BloqueoSimilares1";
   IF #_w14 THEN "Var".CodigoSimilaresJ1[0] := 8; END_IF;
   "ContadorSimilares".CTU(CU := #_w14, R := "ReiniciarChecarSimi", PV := 3, CV => "ContadorSimi");
   IF #_w14 THEN
       "ContadorSimiTemp" := "ContadorSimi";
       "BloqueoSimilares1" := FALSE;
   END_IF;
   #_w15 := #_w9 AND "BloqueoSimilares2";
   IF #_w15 THEN "Var".CodigoSimilaresJ1[2] := 8; END_IF;
   "ContadorSimilares".CTU(CU := #_w15, R := "ReiniciarChecarSimi", PV := 3, CV => "ContadorSimi");
   IF #_w15 THEN
       "ContadorSimiTemp" := "ContadorSimi";
       "BloqueoSimilares2" := FALSE;
   END_IF;
   #_w16 := #_w9 AND "BloqueoSimilares3";
   IF #_w16 THEN "Var".CodigoSimilaresJ1[3] := 8; END_IF;
   "ContadorSimilares".CTU(CU := #_w16, R := "ReiniciarChecarSimi", PV := 3, CV => "ContadorSimi");
   IF #_w16 THEN
       "ContadorSimiTemp" := "ContadorSimi";
       "BloqueoSimilares3" := FALSE;
   END_IF;
   #_w17 := "Panel1AzulJ1" AND "Bounce3" AND "Panel1AzulJ1" AND "Intento1J1" AND ("Var".VectorPrincipalJ1["IntentoCompletoJ1", 2] = 0);
   IF #_w17 THEN
       "Var".VectorPrincipalJ1["IntentoCompletoJ1", 2] := 5;
       "Intento2J1" := TRUE;
   END_IF;
   #_w18 := #_w17 AND ("Var".VectorPrincipalJ1["IntentoCompletoJ1", 2] = "Var".CodigoOJ1[2]);
   "ContadorCorrectas".CTU(CU := #_w18, R := "ReiniciarChecarCorr", PV := 3, CV => "ContadorCorr");
   IF #_w18 THEN
       "ContadorCorrTemp" := "ContadorCorr";
       "Var".CodigoSimilaresJ1[2] := 8;
       "BloqueoSimilares4" := TRUE;
   END_IF;
   #_w19 := #_w18 AND ("Var".CodigoSimilaresJ1[2] = 8);
   "ContadorSimilares".CTD(CD := #_w19, LD := "ReiniciarChecarSimi", PV := 3, CV => "ContadorSimi");
   IF #_w19 THEN "ContadorSimiTemp" := "ContadorSimi"; END_IF;
   #_w20 := #_w17 AND NOT "BloqueoSimilares4" AND ("Var".VectorPrincipalJ1["IntentoCompletoJ1", 2] <> "Var".CodigoOJ1[2]);
   IF #_w20 AND ("Var".VectorPrincipalJ1["IntentoCompletoJ1", 2] = "Var".CodigoSimilaresJ1[0]) THEN
       "BloqueoSimilares1" := TRUE;
   END_IF;
   #_w21 := #_w20 AND ("Var".VectorPrincipalJ1["IntentoCompletoJ1", 2] <> "Var".CodigoSimilaresJ1[0]);
   IF #_w21 AND ("Var".VectorPrincipalJ1["IntentoCompletoJ1", 2] = "Var".CodigoSimilaresJ1[1]) THEN
       "BloqueoSimilares2" := TRUE;
   END_IF;
   IF #_w21 AND ("Var".VectorPrincipalJ1["IntentoCompletoJ1", 2] <> "Var".CodigoSimilaresJ1[1]) AND ("Var".VectorPrincipalJ1["IntentoCompletoJ1", 2] = "Var".CodigoSimilaresJ1[3]) THEN
       "BloqueoSimilares3" := TRUE;
   END_IF;
   #_w22 := #_w17 AND "BloqueoSimilares1";
   IF #_w22 THEN "Var".CodigoSimilaresJ1[0] := 8; END_IF;
   "ContadorSimilares".CTU(CU := #_w22, R := "ReiniciarChecarSimi", PV := 3, CV => "ContadorSimi");
   IF #_w22 THEN
       "ContadorSimiTemp" := "ContadorSimi";
       "BloqueoSimilares1" := FALSE;
   END_IF;
   #_w23 := #_w17 AND "BloqueoSimilares2";
   IF #_w23 THEN "Var".CodigoSimilaresJ1[1] := 8; END_IF;
   "ContadorSimilares".CTU(CU := #_w23, R := "ReiniciarChecarSimi", PV := 3, CV => "ContadorSimi");
   IF #_w23 THEN
       "ContadorSimiTemp" := "ContadorSimi";
       "BloqueoSimilares2" := FALSE;
   END_IF;
   #_w24 := #_w17 AND "BloqueoSimilares3";
   IF #_w24 THEN "Var".CodigoSimilaresJ1[3] := 8; END_IF;
   "ContadorSimilares".CTU(CU := #_w24, R := "ReiniciarChecarSimi", PV := 3, CV => "ContadorSimi");
   IF #_w24 THEN
       "ContadorSimiTemp" := "ContadorSimi";
       "BloqueoSimilares3" := FALSE;
   END_IF;
   #_w25 := "Panel1AzulJ1" AND "Bounce4" AND "Panel1AzulJ1" AND "Intento2J1" AND ("Var".VectorPrincipalJ1["IntentoCompletoJ1", 3] = 0);
   IF #_w25 THEN
       "Var".VectorPrincipalJ1["IntentoCompletoJ1", 3] := 5;
       "Intento3J1" := TRUE;
   END_IF;
   #_w26 := #_w25 AND ("Var".VectorPrincipalJ1["IntentoCompletoJ1", 3] = "Var".CodigoOJ1[3]);
   "ContadorCorrectas".CTU(CU := #_w26, R := "ReiniciarChecarCorr", PV := 3, CV => "ContadorCorr");
   IF #_w26 THEN
       "ContadorCorrTemp" := "ContadorCorr";
       "Var".CodigoSimilaresJ1[3] := 8;
       "BloqueoSimilares4" := TRUE;
   END_IF;
   #_w27 := #_w26 AND ("Var".CodigoSimilaresJ1[3] = 8);
   "ContadorSimilares".CTD(CD := #_w27, LD := "ReiniciarChecarSimi", PV := 3, CV => "ContadorSimi");
   IF #_w27 THEN "ContadorSimiTemp" := "ContadorSimi"; END_IF;
   #_w28 := #_w25 AND NOT "BloqueoSimilares4" AND ("Var".VectorPrincipalJ1["IntentoCompletoJ1", 3] <> "Var".CodigoOJ1[3]);
   IF #_w28 AND ("Var".VectorPrincipalJ1["IntentoCompletoJ1", 3] = "Var".CodigoSimilaresJ1[0]) THEN
       "BloqueoSimilares1" := TRUE;
   END_IF;
   #_w29 := #_w28 AND ("Var".VectorPrincipalJ1["IntentoCompletoJ1", 3] <> "Var".CodigoSimilaresJ1[0]);
   IF #_w29 AND ("Var".VectorPrincipalJ1["IntentoCompletoJ1", 3] = "Var".CodigoSimilaresJ1[1]) THEN
       "BloqueoSimilares2" := TRUE;
   END_IF;
   IF #_w29 AND ("Var".VectorPrincipalJ1["IntentoCompletoJ1", 3] <> "Var".CodigoSimilaresJ1[1]) AND ("Var".VectorPrincipalJ1["IntentoCompletoJ1", 3] = "Var".CodigoSimilaresJ1[2]) THEN
       "BloqueoSimilares3" := TRUE;
   END_IF;
   #_w30 := #_w25 AND "BloqueoSimilares1";
   IF #_w30 THEN "Var".CodigoSimilaresJ1[0] := 8; END_IF;
   "ContadorSimilares".CTU(CU := #_w30, R := "ReiniciarChecarSimi", PV := 3, CV => "ContadorSimi");
   IF #_w30 THEN
       "ContadorSimiTemp" := "ContadorSimi";
       "BloqueoSimilares1" := FALSE;
   END_IF;
   #_w31 := #_w25 AND "BloqueoSimilares2";
   IF #_w31 THEN "Var".CodigoSimilaresJ1[1] := 8; END_IF;
   "ContadorSimilares".CTU(CU := #_w31, R := "ReiniciarChecarSimi", PV := 3, CV => "ContadorSimi");
   IF #_w31 THEN
       "ContadorSimiTemp" := "ContadorSimi";
       "BloqueoSimilares2" := FALSE;
   END_IF;
   #_w32 := #_w25 AND "BloqueoSimilares3";
   IF #_w32 THEN "Var".CodigoSimilaresJ1[2] := 8; END_IF;
   "ContadorSimilares".CTU(CU := #_w32, R := "ReiniciarChecarSimi", PV := 3, CV => "ContadorSimi");
   IF #_w32 THEN
       "ContadorSimiTemp" := "ContadorSimi";
       "BloqueoSimilares3" := FALSE;
   END_IF;
END_REGION

REGION Network 11: Verde
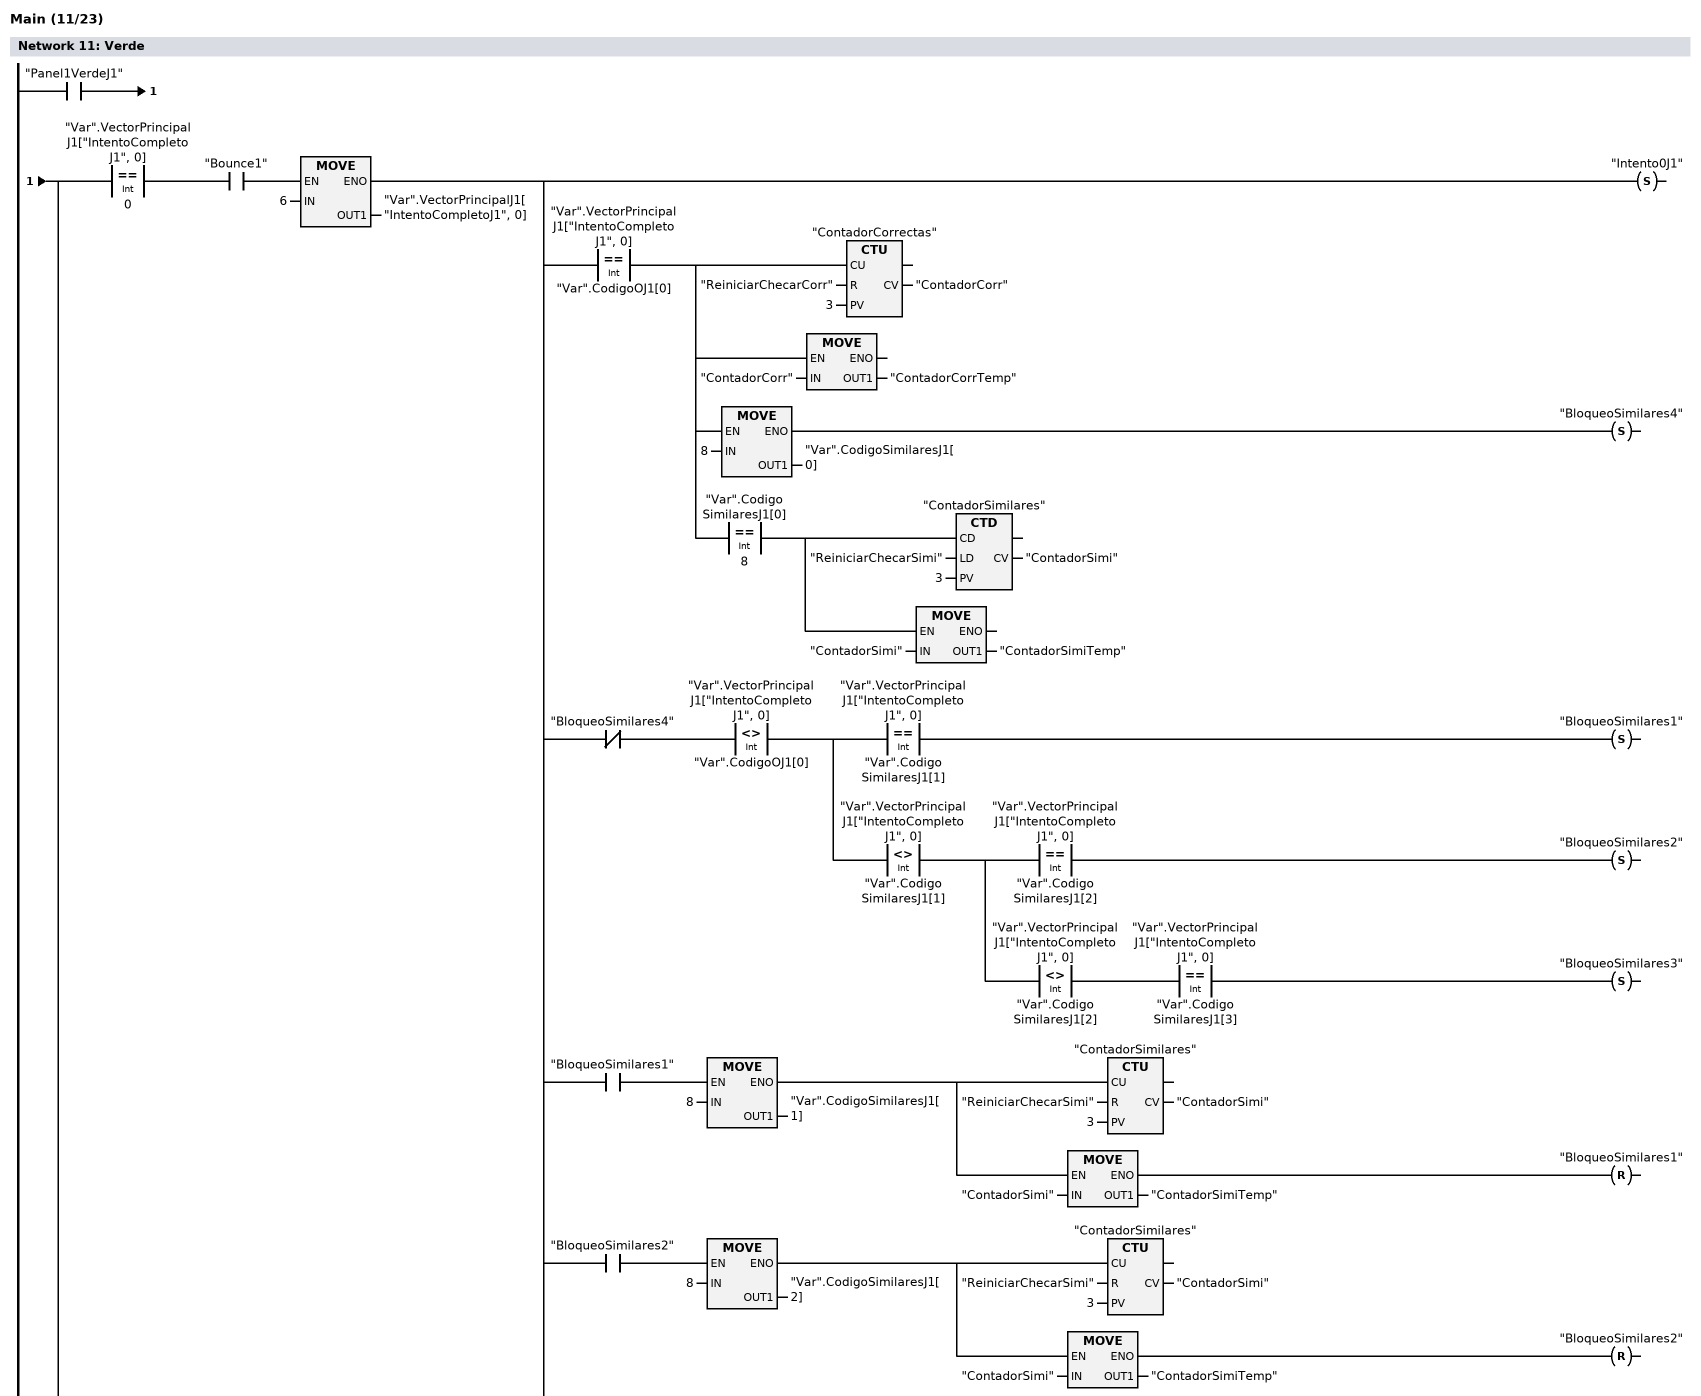
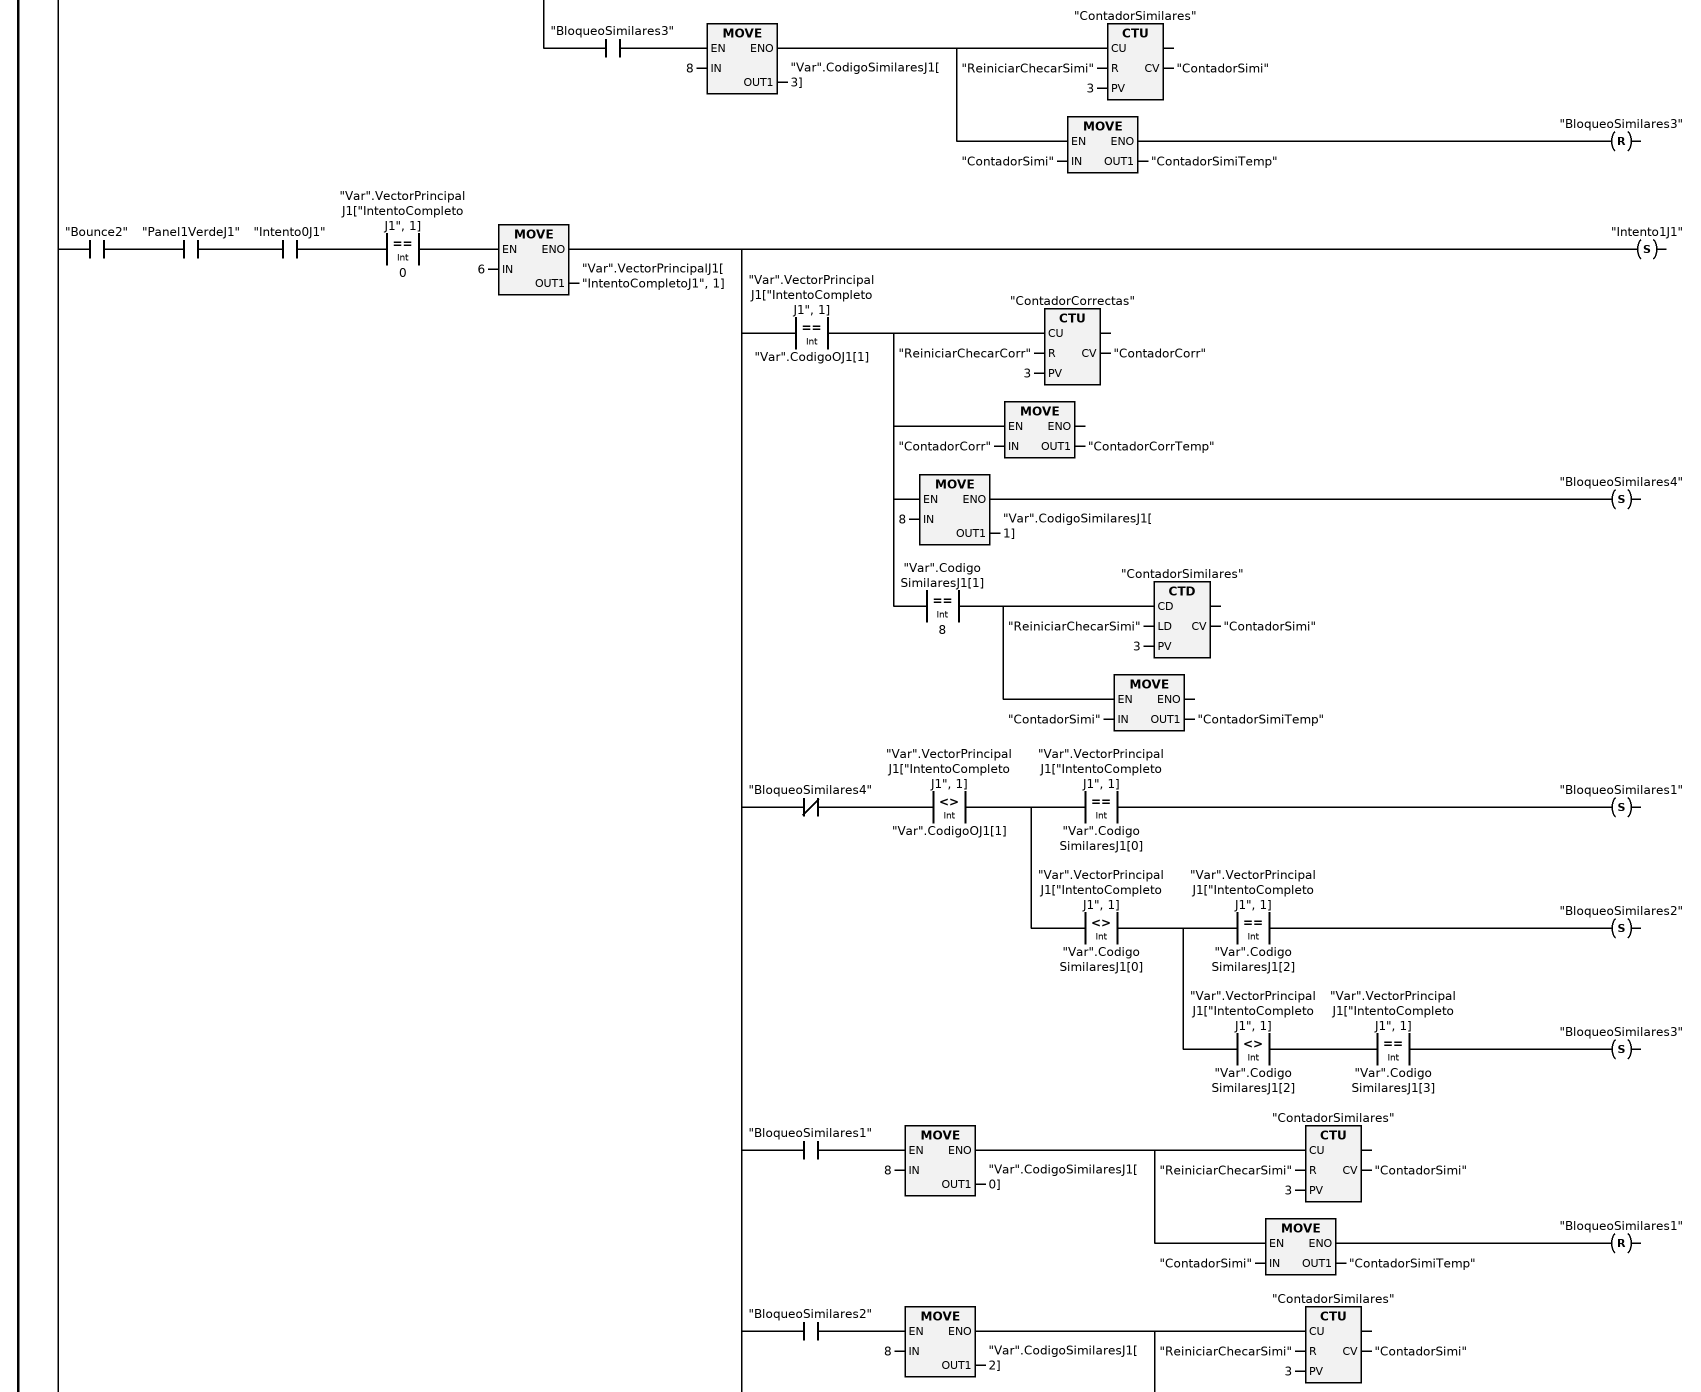
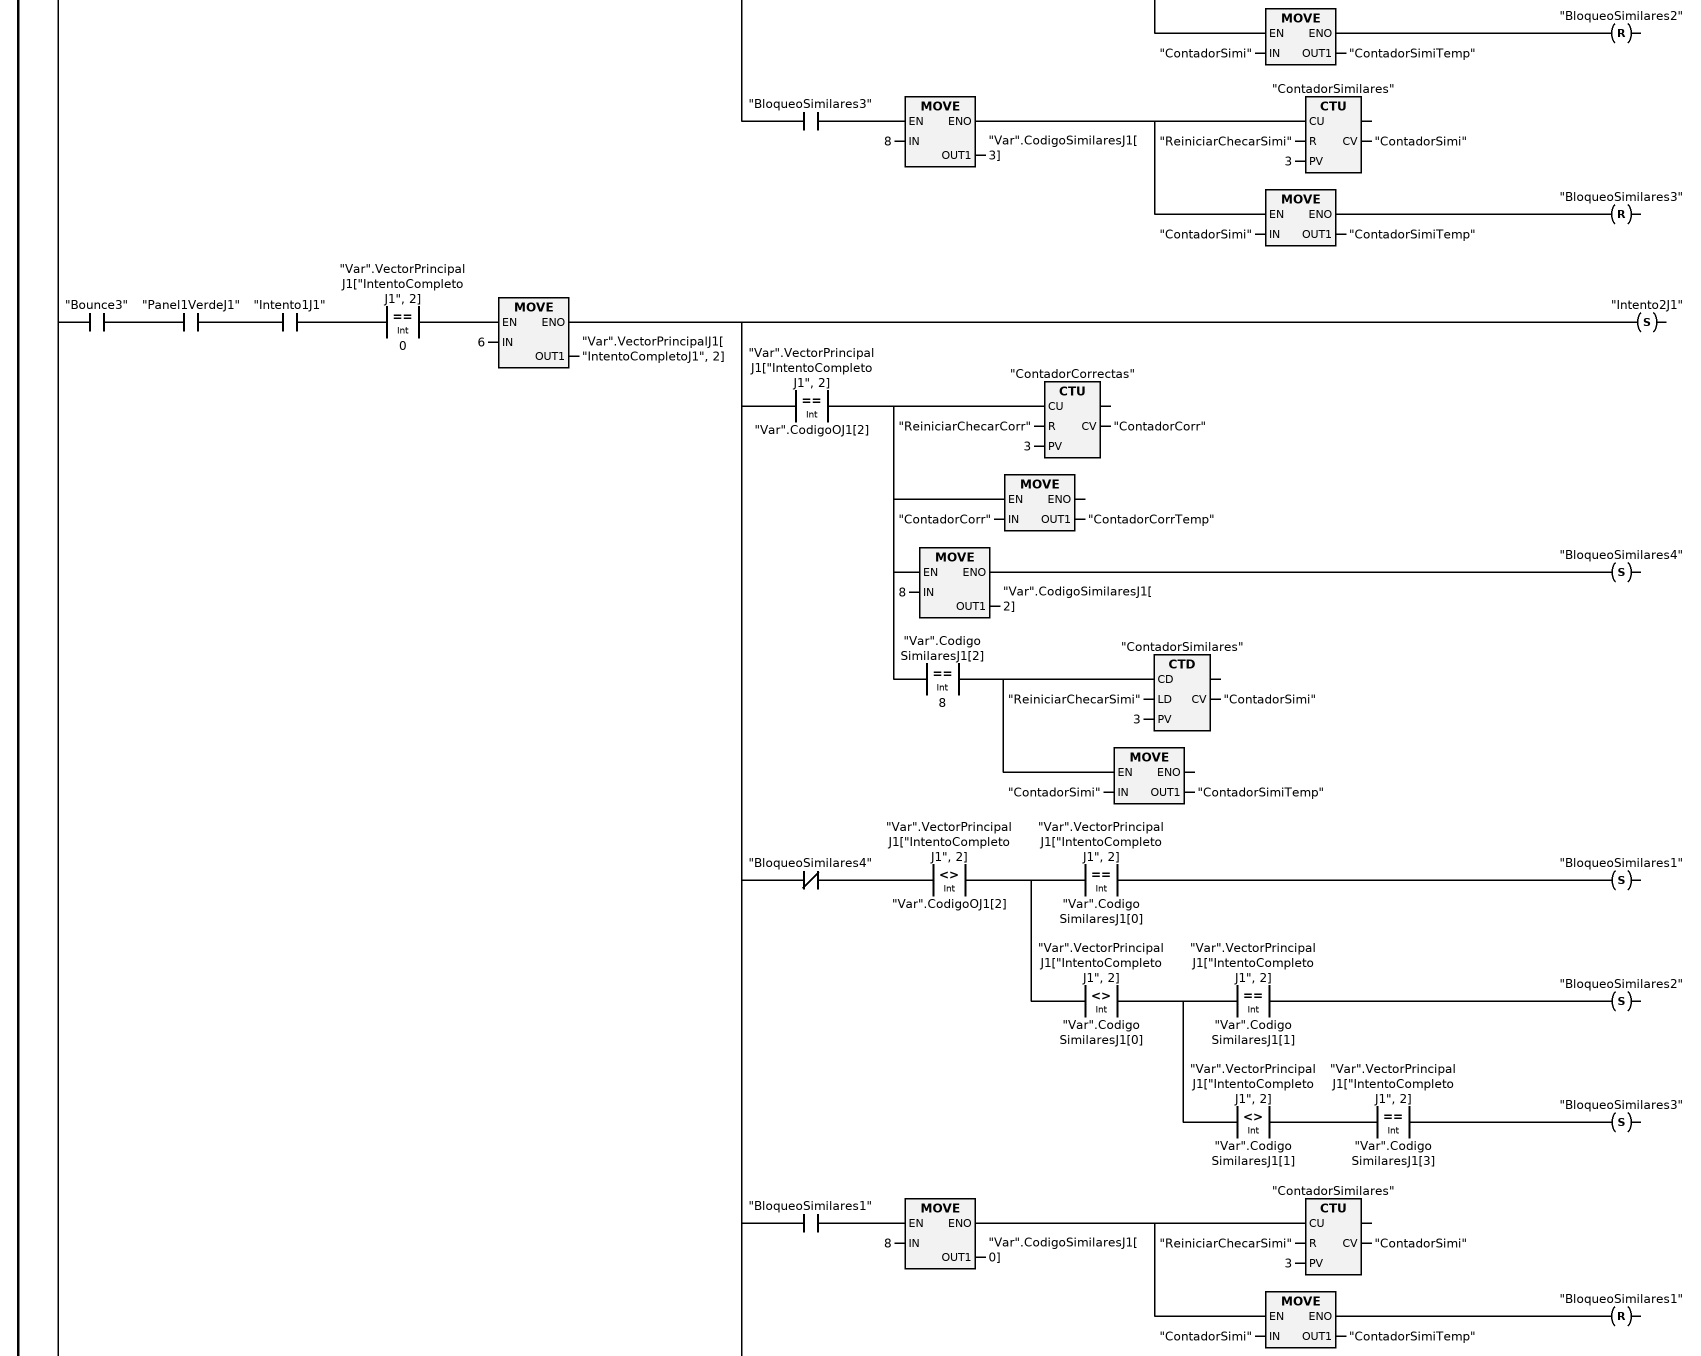
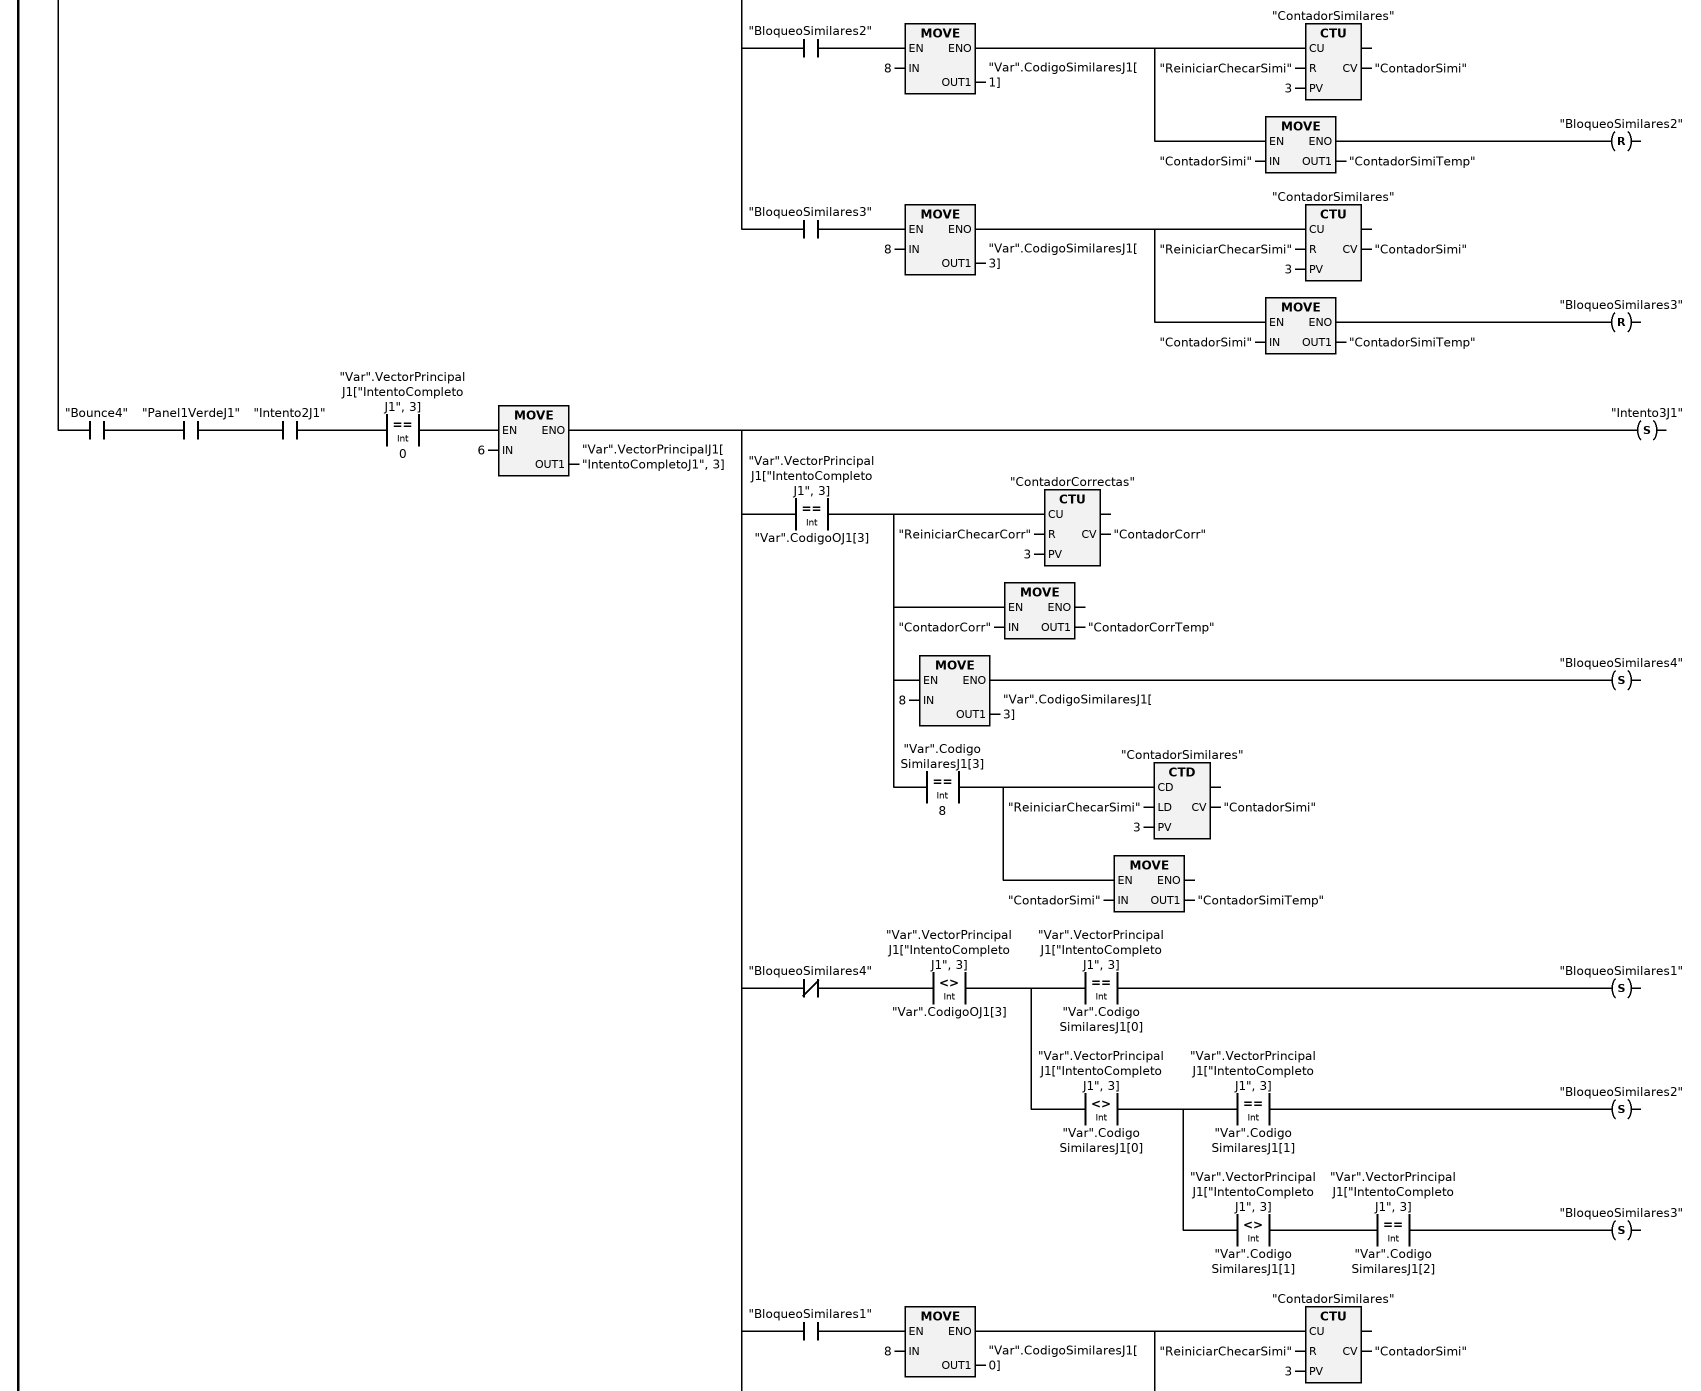
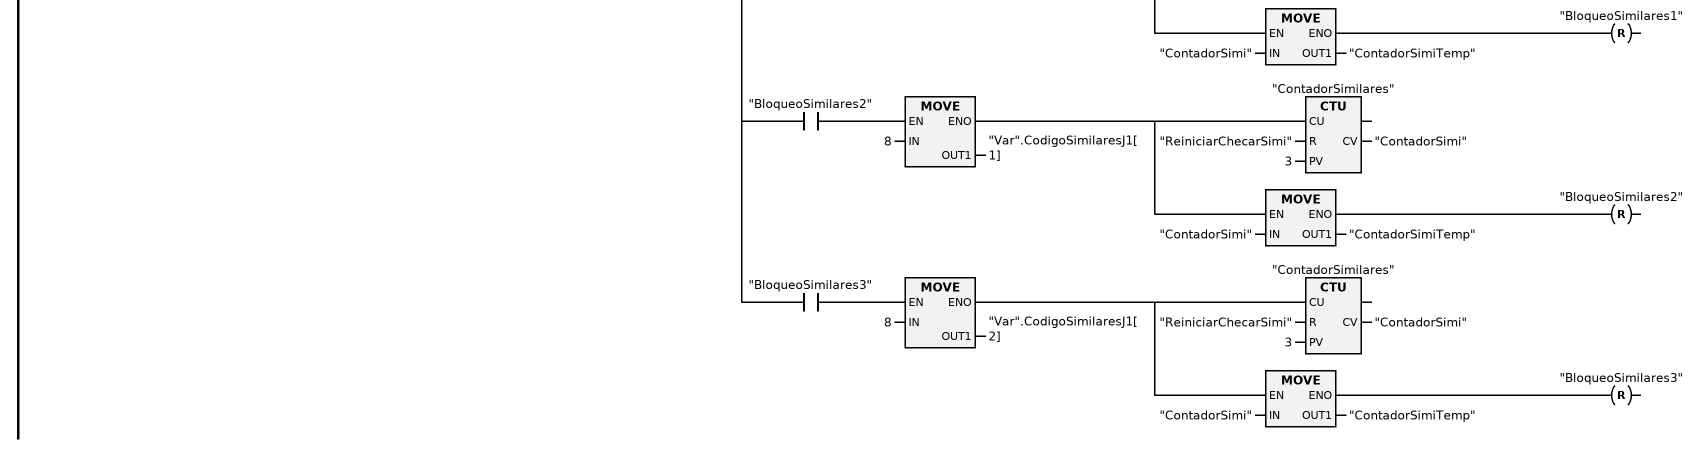
   #_w1 := "Panel1VerdeJ1" AND ("Var".VectorPrincipalJ1["IntentoCompletoJ1", 0] = 0) AND "Bounce1";
   IF #_w1 THEN
       "Var".VectorPrincipalJ1["IntentoCompletoJ1", 0] := 6;
       "Intento0J1" := TRUE;
   END_IF;
   #_w2 := #_w1 AND ("Var".VectorPrincipalJ1["IntentoCompletoJ1", 0] = "Var".CodigoOJ1[0]);
   "ContadorCorrectas".CTU(CU := #_w2, R := "ReiniciarChecarCorr", PV := 3, CV => "ContadorCorr");
   IF #_w2 THEN
       "ContadorCorrTemp" := "ContadorCorr";
       "Var".CodigoSimilaresJ1[0] := 8;
       "BloqueoSimilares4" := TRUE;
   END_IF;
   #_w3 := #_w2 AND ("Var".CodigoSimilaresJ1[0] = 8);
   "ContadorSimilares".CTD(CD := #_w3, LD := "ReiniciarChecarSimi", PV := 3, CV => "ContadorSimi");
   IF #_w3 THEN "ContadorSimiTemp" := "ContadorSimi"; END_IF;
   #_w4 := #_w1 AND NOT "BloqueoSimilares4" AND ("Var".VectorPrincipalJ1["IntentoCompletoJ1", 0] <> "Var".CodigoOJ1[0]);
   IF #_w4 AND ("Var".VectorPrincipalJ1["IntentoCompletoJ1", 0] = "Var".CodigoSimilaresJ1[1]) THEN
       "BloqueoSimilares1" := TRUE;
   END_IF;
   #_w5 := #_w4 AND ("Var".VectorPrincipalJ1["IntentoCompletoJ1", 0] <> "Var".CodigoSimilaresJ1[1]);
   IF #_w5 AND ("Var".VectorPrincipalJ1["IntentoCompletoJ1", 0] = "Var".CodigoSimilaresJ1[2]) THEN
       "BloqueoSimilares2" := TRUE;
   END_IF;
   IF #_w5 AND ("Var".VectorPrincipalJ1["IntentoCompletoJ1", 0] <> "Var".CodigoSimilaresJ1[2]) AND ("Var".VectorPrincipalJ1["IntentoCompletoJ1", 0] = "Var".CodigoSimilaresJ1[3]) THEN
       "BloqueoSimilares3" := TRUE;
   END_IF;
   #_w6 := #_w1 AND "BloqueoSimilares1";
   IF #_w6 THEN "Var".CodigoSimilaresJ1[1] := 8; END_IF;
   "ContadorSimilares".CTU(CU := #_w6, R := "ReiniciarChecarSimi", PV := 3, CV => "ContadorSimi");
   IF #_w6 THEN
       "ContadorSimiTemp" := "ContadorSimi";
       "BloqueoSimilares1" := FALSE;
   END_IF;
   #_w7 := #_w1 AND "BloqueoSimilares2";
   IF #_w7 THEN "Var".CodigoSimilaresJ1[2] := 8; END_IF;
   "ContadorSimilares".CTU(CU := #_w7, R := "ReiniciarChecarSimi", PV := 3, CV => "ContadorSimi");
   IF #_w7 THEN
       "ContadorSimiTemp" := "ContadorSimi";
       "BloqueoSimilares2" := FALSE;
   END_IF;
   #_w8 := #_w1 AND "BloqueoSimilares3";
   IF #_w8 THEN "Var".CodigoSimilaresJ1[3] := 8; END_IF;
   "ContadorSimilares".CTU(CU := #_w8, R := "ReiniciarChecarSimi", PV := 3, CV => "ContadorSimi");
   IF #_w8 THEN
       "ContadorSimiTemp" := "ContadorSimi";
       "BloqueoSimilares3" := FALSE;
   END_IF;
   #_w9 := "Panel1VerdeJ1" AND "Bounce2" AND "Panel1VerdeJ1" AND "Intento0J1" AND ("Var".VectorPrincipalJ1["IntentoCompletoJ1", 1] = 0);
   IF #_w9 THEN
       "Var".VectorPrincipalJ1["IntentoCompletoJ1", 1] := 6;
       "Intento1J1" := TRUE;
   END_IF;
   #_w10 := #_w9 AND ("Var".VectorPrincipalJ1["IntentoCompletoJ1", 1] = "Var".CodigoOJ1[1]);
   "ContadorCorrectas".CTU(CU := #_w10, R := "ReiniciarChecarCorr", PV := 3, CV => "ContadorCorr");
   IF #_w10 THEN
       "ContadorCorrTemp" := "ContadorCorr";
       "Var".CodigoSimilaresJ1[1] := 8;
       "BloqueoSimilares4" := TRUE;
   END_IF;
   #_w11 := #_w10 AND ("Var".CodigoSimilaresJ1[1] = 8);
   "ContadorSimilares".CTD(CD := #_w11, LD := "ReiniciarChecarSimi", PV := 3, CV => "ContadorSimi");
   IF #_w11 THEN "ContadorSimiTemp" := "ContadorSimi"; END_IF;
   #_w12 := #_w9 AND NOT "BloqueoSimilares4" AND ("Var".VectorPrincipalJ1["IntentoCompletoJ1", 1] <> "Var".CodigoOJ1[1]);
   IF #_w12 AND ("Var".VectorPrincipalJ1["IntentoCompletoJ1", 1] = "Var".CodigoSimilaresJ1[0]) THEN
       "BloqueoSimilares1" := TRUE;
   END_IF;
   #_w13 := #_w12 AND ("Var".VectorPrincipalJ1["IntentoCompletoJ1", 1] <> "Var".CodigoSimilaresJ1[0]);
   IF #_w13 AND ("Var".VectorPrincipalJ1["IntentoCompletoJ1", 1] = "Var".CodigoSimilaresJ1[2]) THEN
       "BloqueoSimilares2" := TRUE;
   END_IF;
   IF #_w13 AND ("Var".VectorPrincipalJ1["IntentoCompletoJ1", 1] <> "Var".CodigoSimilaresJ1[2]) AND ("Var".VectorPrincipalJ1["IntentoCompletoJ1", 1] = "Var".CodigoSimilaresJ1[3]) THEN
       "BloqueoSimilares3" := TRUE;
   END_IF;
   #_w14 := #_w9 AND "BloqueoSimilares1";
   IF #_w14 THEN "Var".CodigoSimilaresJ1[0] := 8; END_IF;
   "ContadorSimilares".CTU(CU := #_w14, R := "ReiniciarChecarSimi", PV := 3, CV => "ContadorSimi");
   IF #_w14 THEN
       "ContadorSimiTemp" := "ContadorSimi";
       "BloqueoSimilares1" := FALSE;
   END_IF;
   #_w15 := #_w9 AND "BloqueoSimilares2";
   IF #_w15 THEN "Var".CodigoSimilaresJ1[2] := 8; END_IF;
   "ContadorSimilares".CTU(CU := #_w15, R := "ReiniciarChecarSimi", PV := 3, CV => "ContadorSimi");
   IF #_w15 THEN
       "ContadorSimiTemp" := "ContadorSimi";
       "BloqueoSimilares2" := FALSE;
   END_IF;
   #_w16 := #_w9 AND "BloqueoSimilares3";
   IF #_w16 THEN "Var".CodigoSimilaresJ1[3] := 8; END_IF;
   "ContadorSimilares".CTU(CU := #_w16, R := "ReiniciarChecarSimi", PV := 3, CV => "ContadorSimi");
   IF #_w16 THEN
       "ContadorSimiTemp" := "ContadorSimi";
       "BloqueoSimilares3" := FALSE;
   END_IF;
   #_w17 := "Panel1VerdeJ1" AND "Bounce3" AND "Panel1VerdeJ1" AND "Intento1J1" AND ("Var".VectorPrincipalJ1["IntentoCompletoJ1", 2] = 0);
   IF #_w17 THEN
       "Var".VectorPrincipalJ1["IntentoCompletoJ1", 2] := 6;
       "Intento2J1" := TRUE;
   END_IF;
   #_w18 := #_w17 AND ("Var".VectorPrincipalJ1["IntentoCompletoJ1", 2] = "Var".CodigoOJ1[2]);
   "ContadorCorrectas".CTU(CU := #_w18, R := "ReiniciarChecarCorr", PV := 3, CV => "ContadorCorr");
   IF #_w18 THEN
       "ContadorCorrTemp" := "ContadorCorr";
       "Var".CodigoSimilaresJ1[2] := 8;
       "BloqueoSimilares4" := TRUE;
   END_IF;
   #_w19 := #_w18 AND ("Var".CodigoSimilaresJ1[2] = 8);
   "ContadorSimilares".CTD(CD := #_w19, LD := "ReiniciarChecarSimi", PV := 3, CV => "ContadorSimi");
   IF #_w19 THEN "ContadorSimiTemp" := "ContadorSimi"; END_IF;
   #_w20 := #_w17 AND NOT "BloqueoSimilares4" AND ("Var".VectorPrincipalJ1["IntentoCompletoJ1", 2] <> "Var".CodigoOJ1[2]);
   IF #_w20 AND ("Var".VectorPrincipalJ1["IntentoCompletoJ1", 2] = "Var".CodigoSimilaresJ1[0]) THEN
       "BloqueoSimilares1" := TRUE;
   END_IF;
   #_w21 := #_w20 AND ("Var".VectorPrincipalJ1["IntentoCompletoJ1", 2] <> "Var".CodigoSimilaresJ1[0]);
   IF #_w21 AND ("Var".VectorPrincipalJ1["IntentoCompletoJ1", 2] = "Var".CodigoSimilaresJ1[1]) THEN
       "BloqueoSimilares2" := TRUE;
   END_IF;
   IF #_w21 AND ("Var".VectorPrincipalJ1["IntentoCompletoJ1", 2] <> "Var".CodigoSimilaresJ1[1]) AND ("Var".VectorPrincipalJ1["IntentoCompletoJ1", 2] = "Var".CodigoSimilaresJ1[3]) THEN
       "BloqueoSimilares3" := TRUE;
   END_IF;
   #_w22 := #_w17 AND "BloqueoSimilares1";
   IF #_w22 THEN "Var".CodigoSimilaresJ1[0] := 8; END_IF;
   "ContadorSimilares".CTU(CU := #_w22, R := "ReiniciarChecarSimi", PV := 3, CV => "ContadorSimi");
   IF #_w22 THEN
       "ContadorSimiTemp" := "ContadorSimi";
       "BloqueoSimilares1" := FALSE;
   END_IF;
   #_w23 := #_w17 AND "BloqueoSimilares2";
   IF #_w23 THEN "Var".CodigoSimilaresJ1[1] := 8; END_IF;
   "ContadorSimilares".CTU(CU := #_w23, R := "ReiniciarChecarSimi", PV := 3, CV => "ContadorSimi");
   IF #_w23 THEN
       "ContadorSimiTemp" := "ContadorSimi";
       "BloqueoSimilares2" := FALSE;
   END_IF;
   #_w24 := #_w17 AND "BloqueoSimilares3";
   IF #_w24 THEN "Var".CodigoSimilaresJ1[3] := 8; END_IF;
   "ContadorSimilares".CTU(CU := #_w24, R := "ReiniciarChecarSimi", PV := 3, CV => "ContadorSimi");
   IF #_w24 THEN
       "ContadorSimiTemp" := "ContadorSimi";
       "BloqueoSimilares3" := FALSE;
   END_IF;
   #_w25 := "Panel1VerdeJ1" AND "Bounce4" AND "Panel1VerdeJ1" AND "Intento2J1" AND ("Var".VectorPrincipalJ1["IntentoCompletoJ1", 3] = 0);
   IF #_w25 THEN
       "Var".VectorPrincipalJ1["IntentoCompletoJ1", 3] := 6;
       "Intento3J1" := TRUE;
   END_IF;
   #_w26 := #_w25 AND ("Var".VectorPrincipalJ1["IntentoCompletoJ1", 3] = "Var".CodigoOJ1[3]);
   "ContadorCorrectas".CTU(CU := #_w26, R := "ReiniciarChecarCorr", PV := 3, CV => "ContadorCorr");
   IF #_w26 THEN
       "ContadorCorrTemp" := "ContadorCorr";
       "Var".CodigoSimilaresJ1[3] := 8;
       "BloqueoSimilares4" := TRUE;
   END_IF;
   #_w27 := #_w26 AND ("Var".CodigoSimilaresJ1[3] = 8);
   "ContadorSimilares".CTD(CD := #_w27, LD := "ReiniciarChecarSimi", PV := 3, CV => "ContadorSimi");
   IF #_w27 THEN "ContadorSimiTemp" := "ContadorSimi"; END_IF;
   #_w28 := #_w25 AND NOT "BloqueoSimilares4" AND ("Var".VectorPrincipalJ1["IntentoCompletoJ1", 3] <> "Var".CodigoOJ1[3]);
   IF #_w28 AND ("Var".VectorPrincipalJ1["IntentoCompletoJ1", 3] = "Var".CodigoSimilaresJ1[0]) THEN
       "BloqueoSimilares1" := TRUE;
   END_IF;
   #_w29 := #_w28 AND ("Var".VectorPrincipalJ1["IntentoCompletoJ1", 3] <> "Var".CodigoSimilaresJ1[0]);
   IF #_w29 AND ("Var".VectorPrincipalJ1["IntentoCompletoJ1", 3] = "Var".CodigoSimilaresJ1[1]) THEN
       "BloqueoSimilares2" := TRUE;
   END_IF;
   IF #_w29 AND ("Var".VectorPrincipalJ1["IntentoCompletoJ1", 3] <> "Var".CodigoSimilaresJ1[1]) AND ("Var".VectorPrincipalJ1["IntentoCompletoJ1", 3] = "Var".CodigoSimilaresJ1[2]) THEN
       "BloqueoSimilares3" := TRUE;
   END_IF;
   #_w30 := #_w25 AND "BloqueoSimilares1";
   IF #_w30 THEN "Var".CodigoSimilaresJ1[0] := 8; END_IF;
   "ContadorSimilares".CTU(CU := #_w30, R := "ReiniciarChecarSimi", PV := 3, CV => "ContadorSimi");
   IF #_w30 THEN
       "ContadorSimiTemp" := "ContadorSimi";
       "BloqueoSimilares1" := FALSE;
   END_IF;
   #_w31 := #_w25 AND "BloqueoSimilares2";
   IF #_w31 THEN "Var".CodigoSimilaresJ1[1] := 8; END_IF;
   "ContadorSimilares".CTU(CU := #_w31, R := "ReiniciarChecarSimi", PV := 3, CV => "ContadorSimi");
   IF #_w31 THEN
       "ContadorSimiTemp" := "ContadorSimi";
       "BloqueoSimilares2" := FALSE;
   END_IF;
   #_w32 := #_w25 AND "BloqueoSimilares3";
   IF #_w32 THEN "Var".CodigoSimilaresJ1[2] := 8; END_IF;
   "ContadorSimilares".CTU(CU := #_w32, R := "ReiniciarChecarSimi", PV := 3, CV => "ContadorSimi");
   IF #_w32 THEN
       "ContadorSimiTemp" := "ContadorSimi";
       "BloqueoSimilares3" := FALSE;
   END_IF;
END_REGION

REGION Network 12: Amarillo
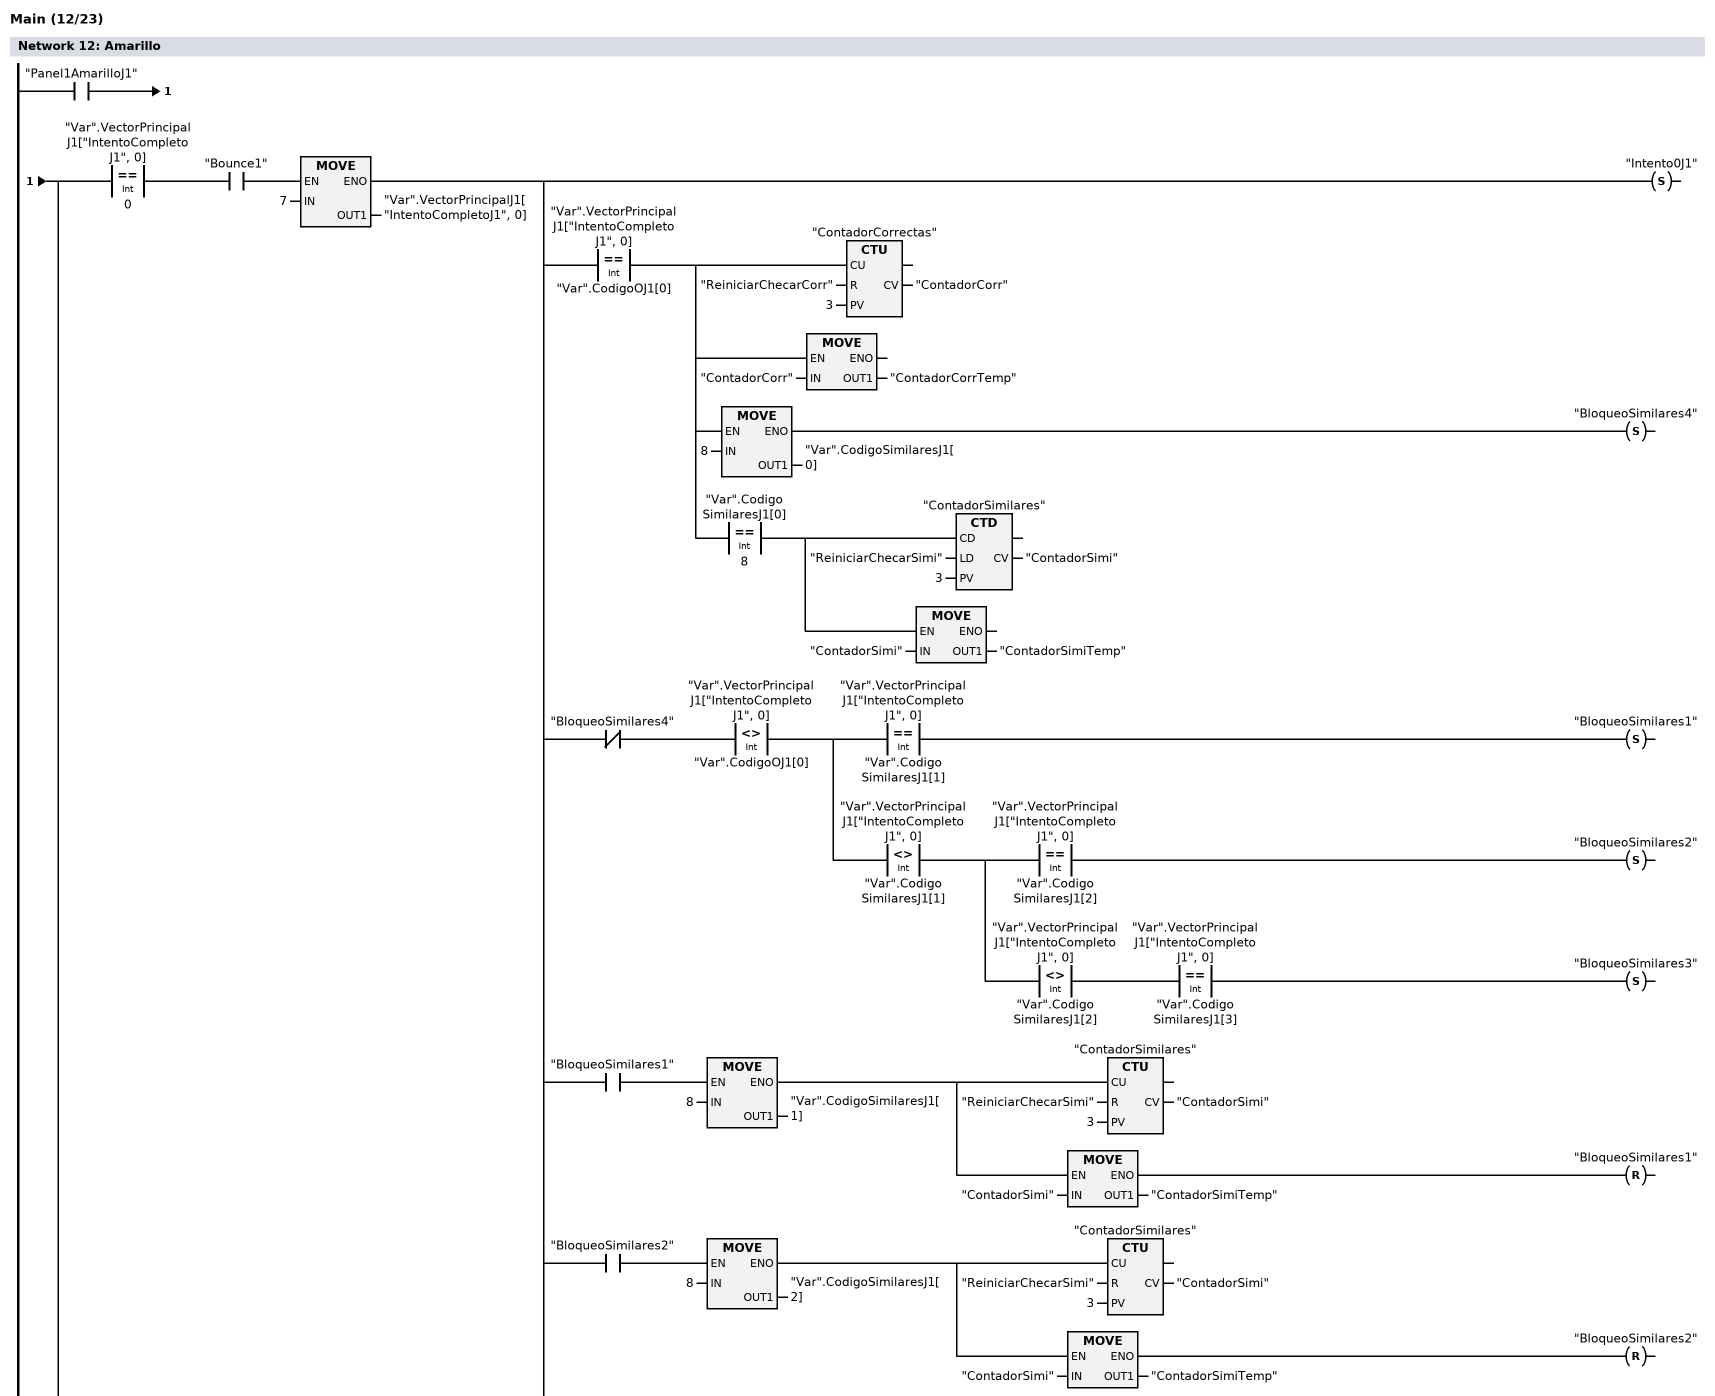
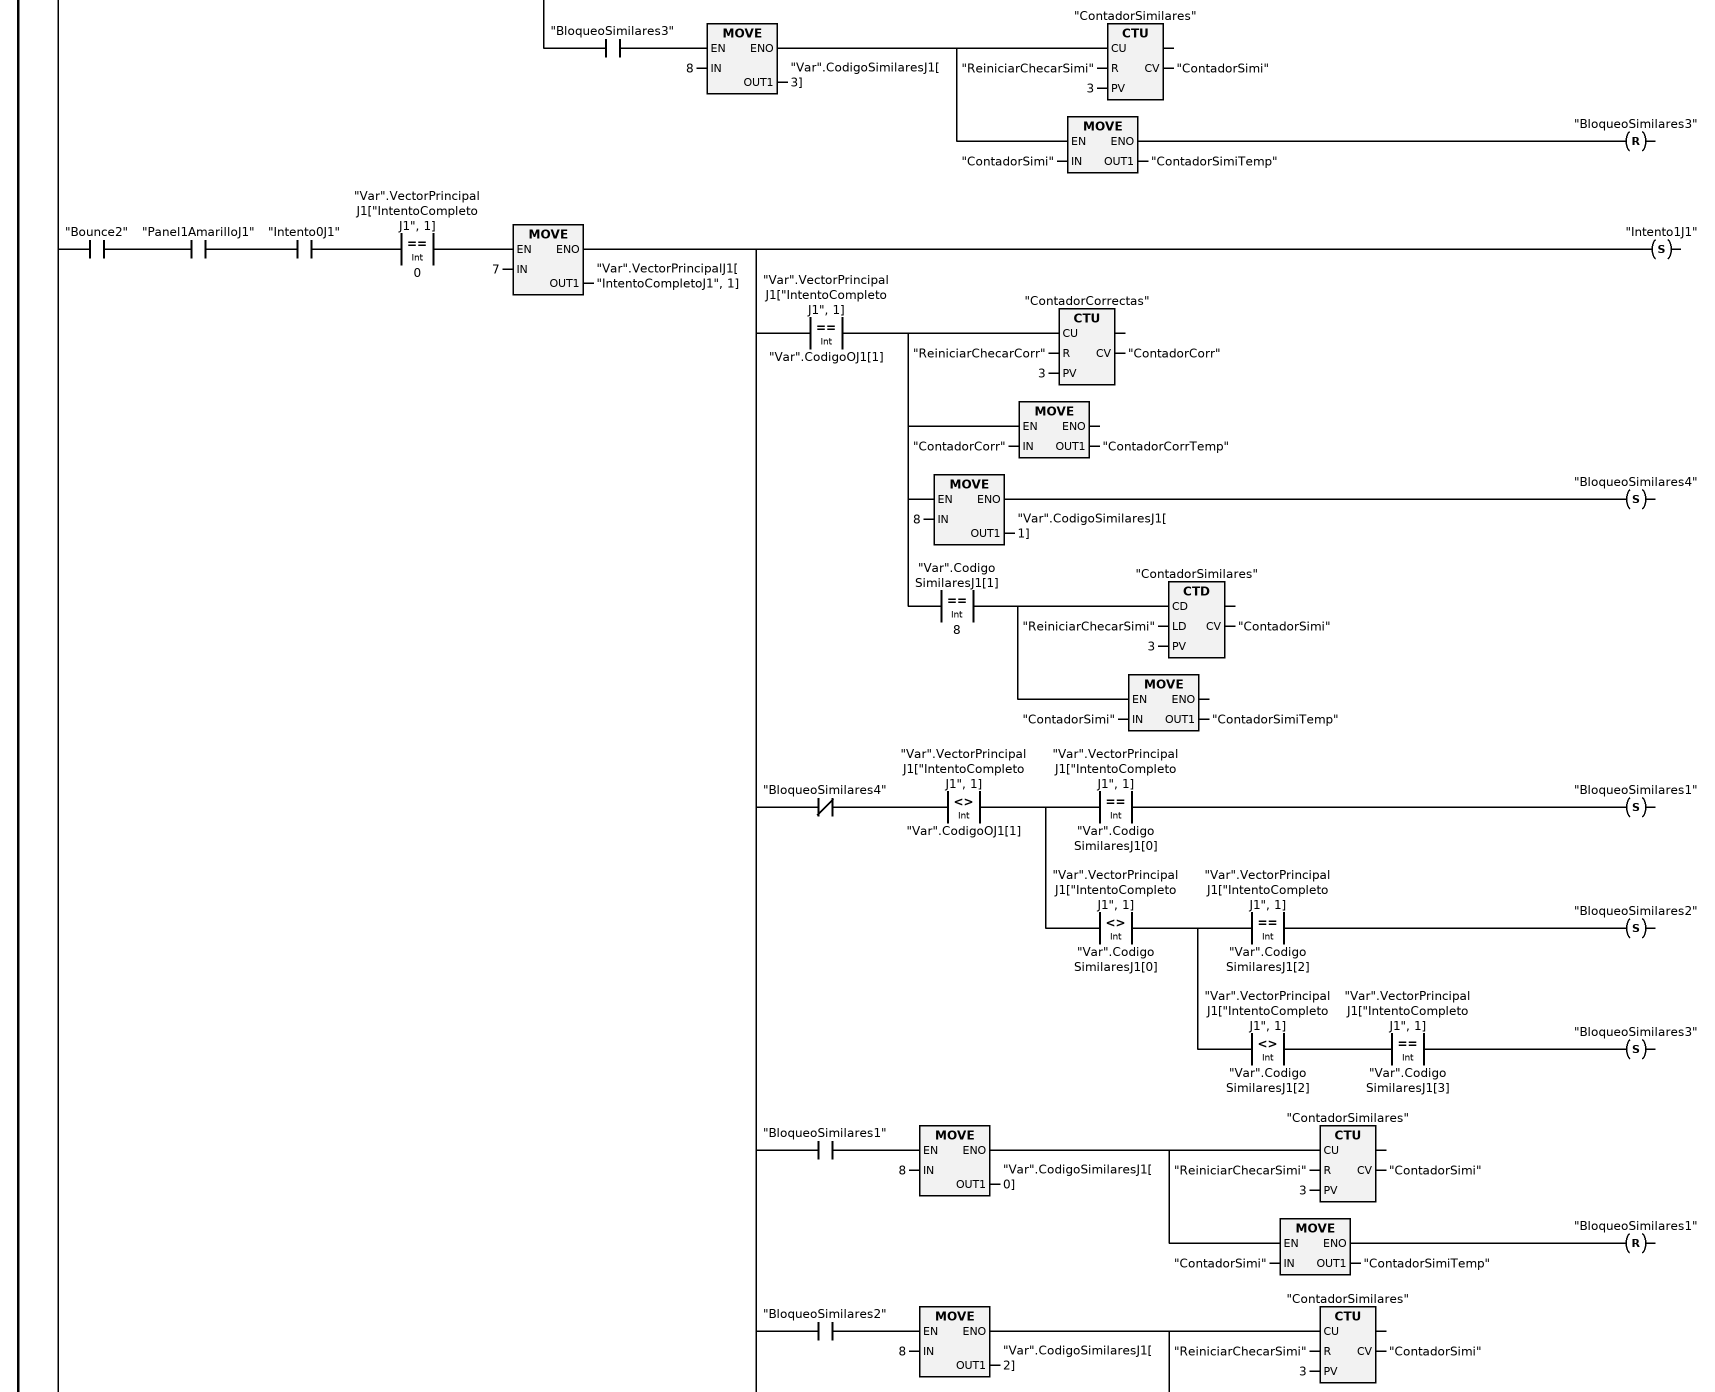
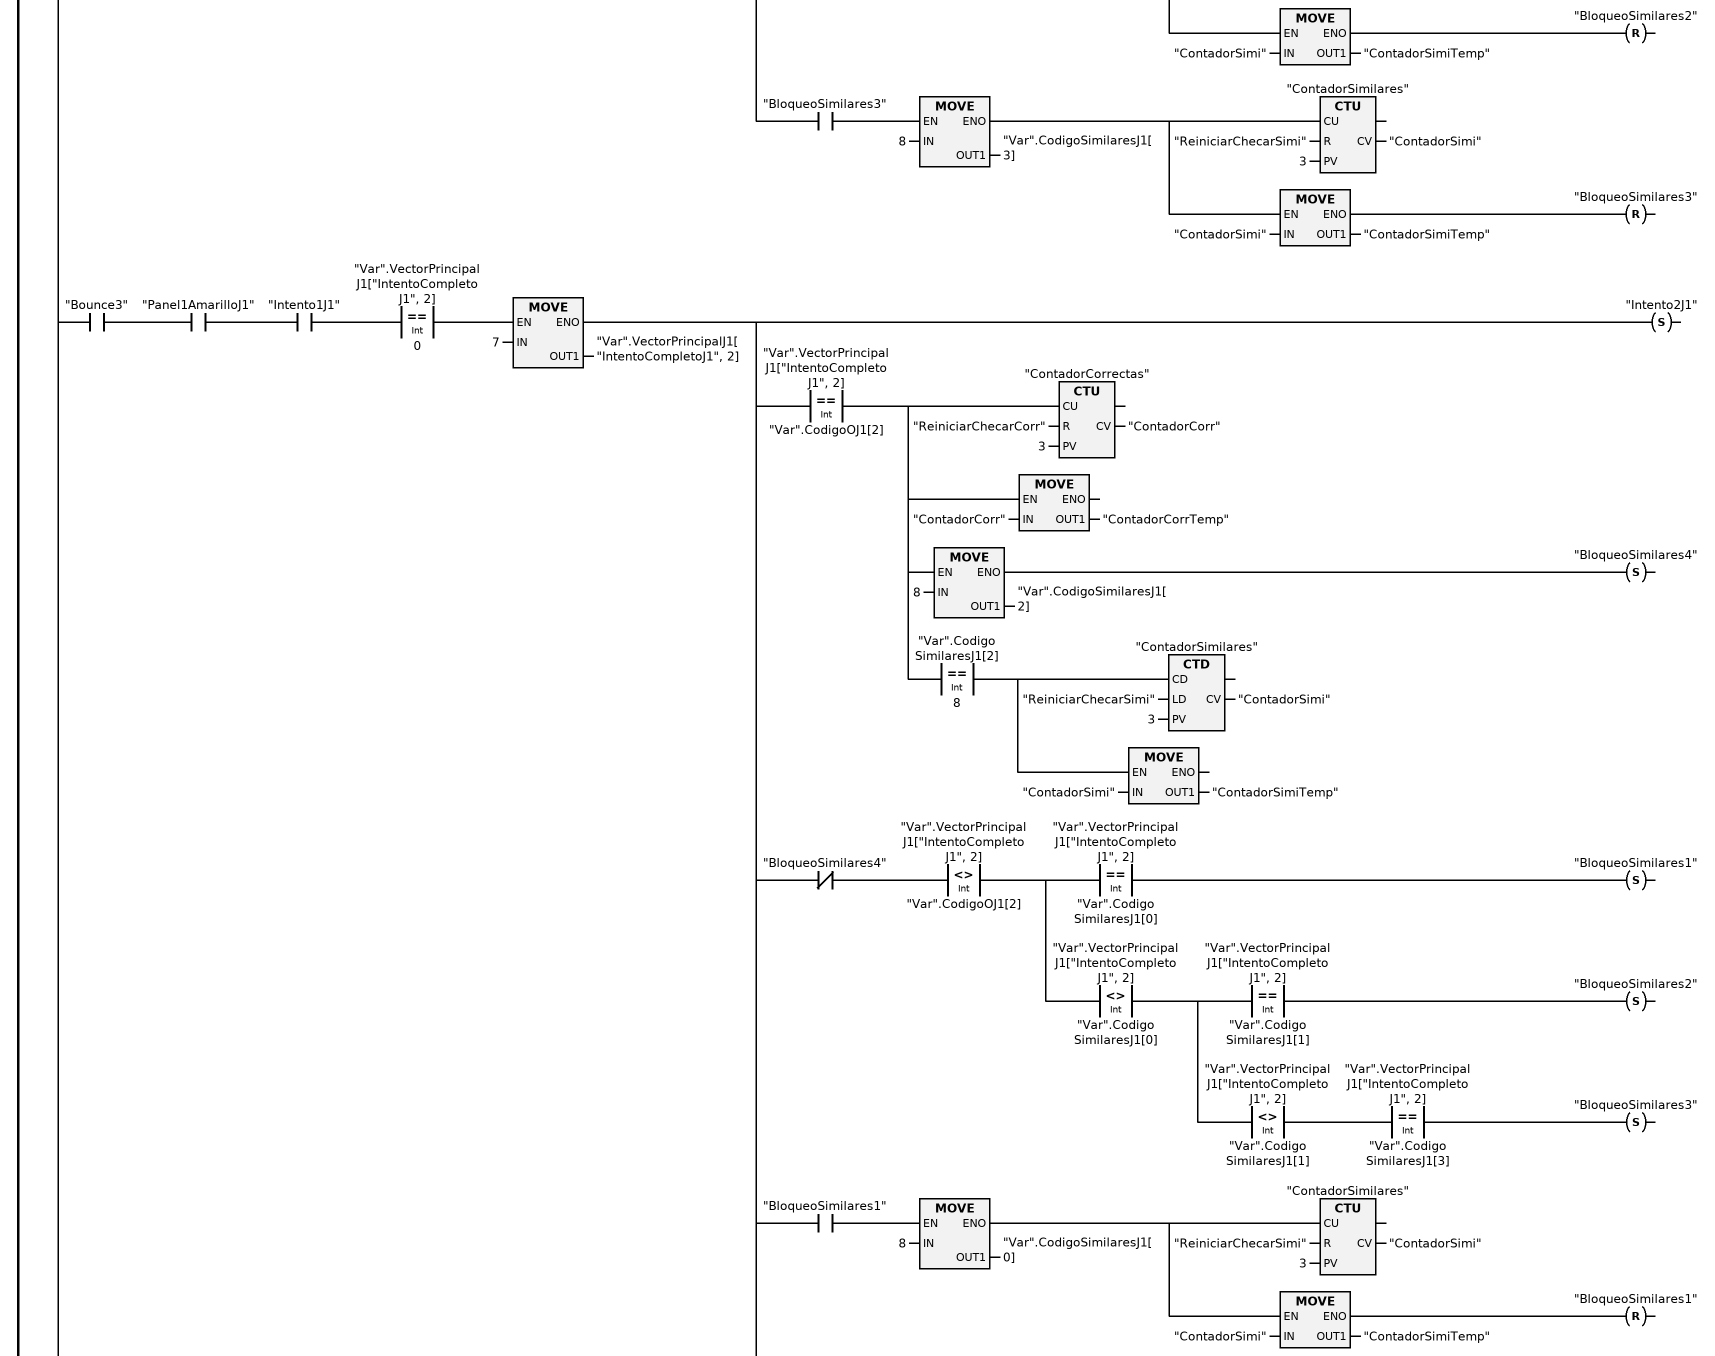
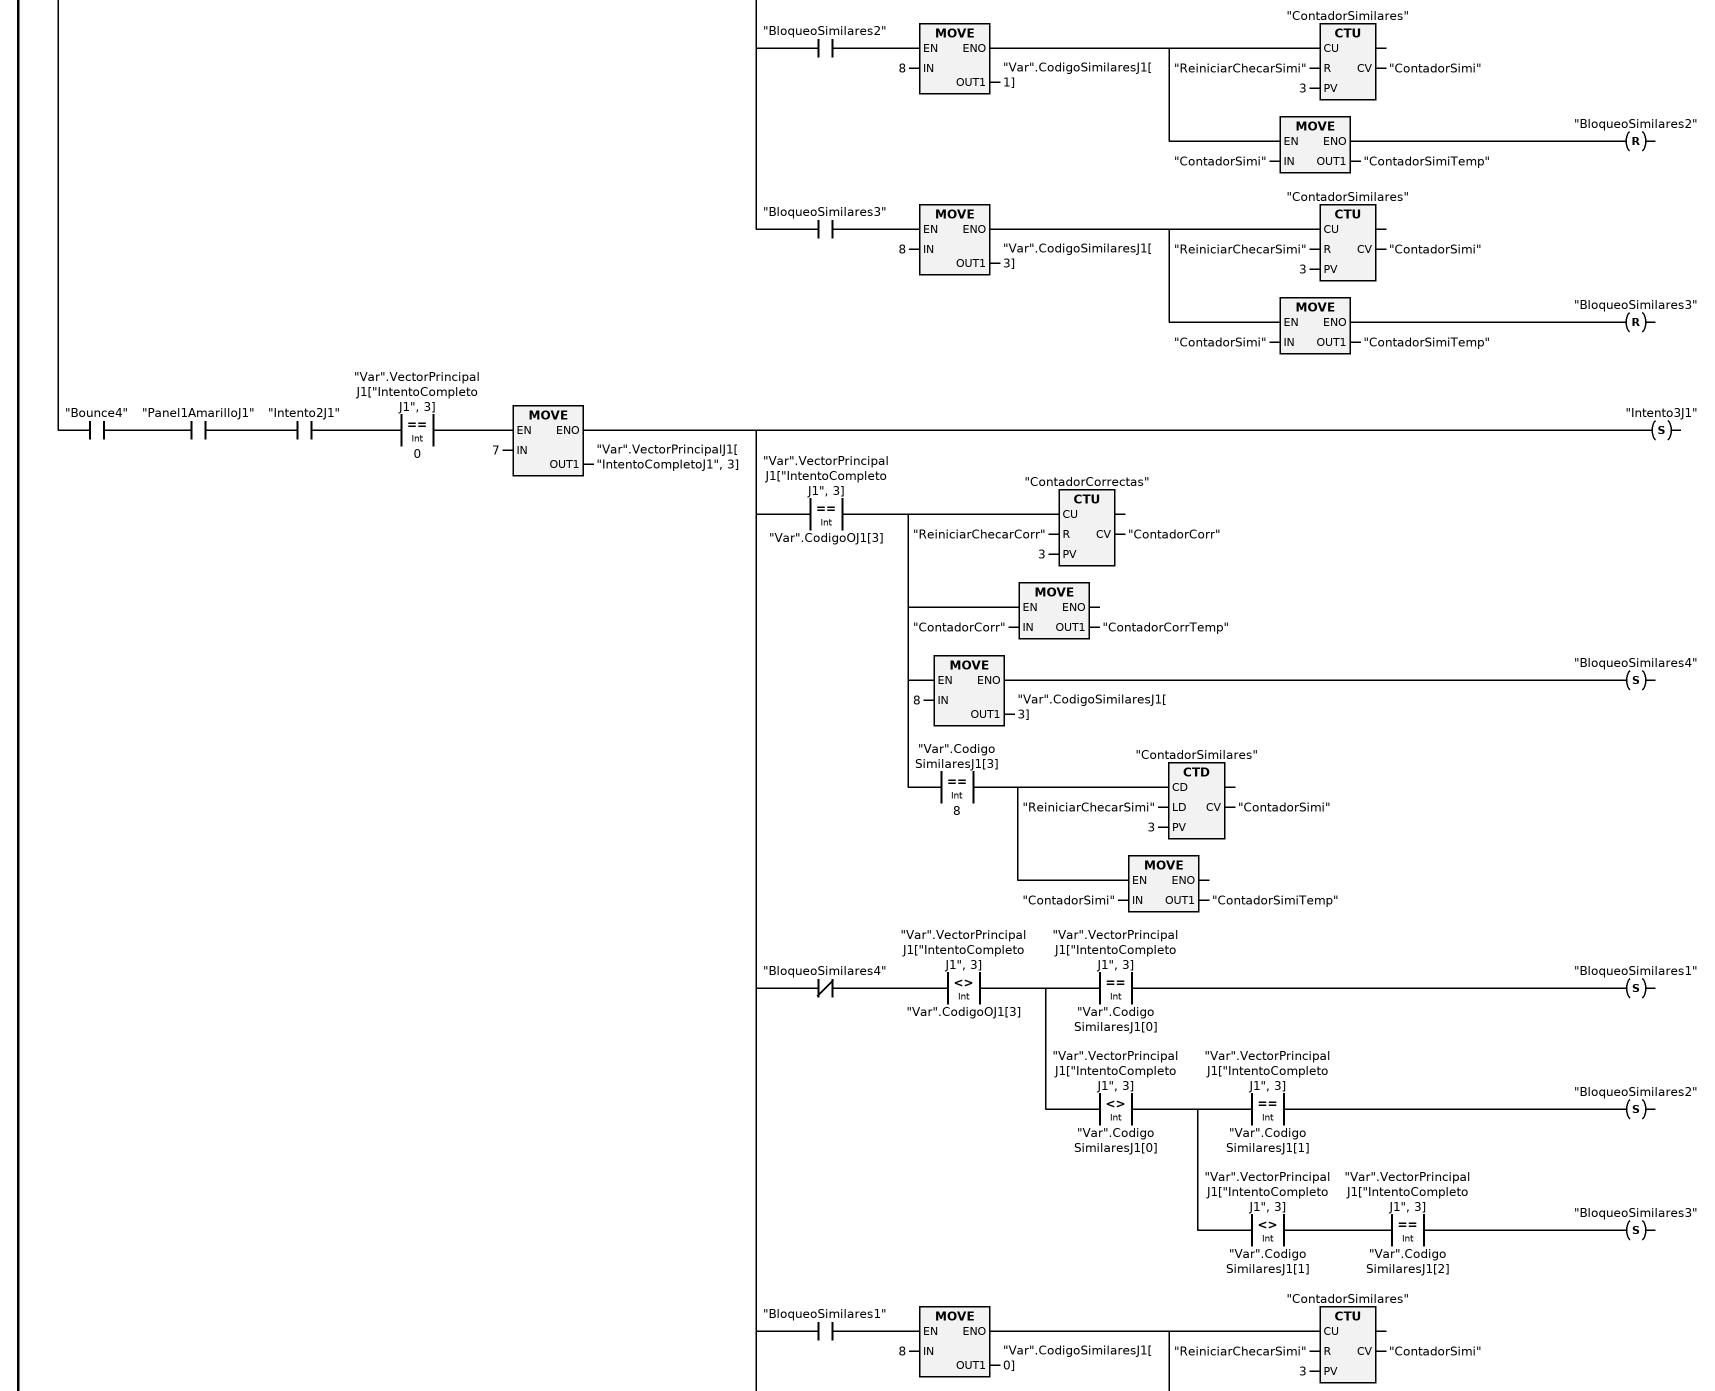
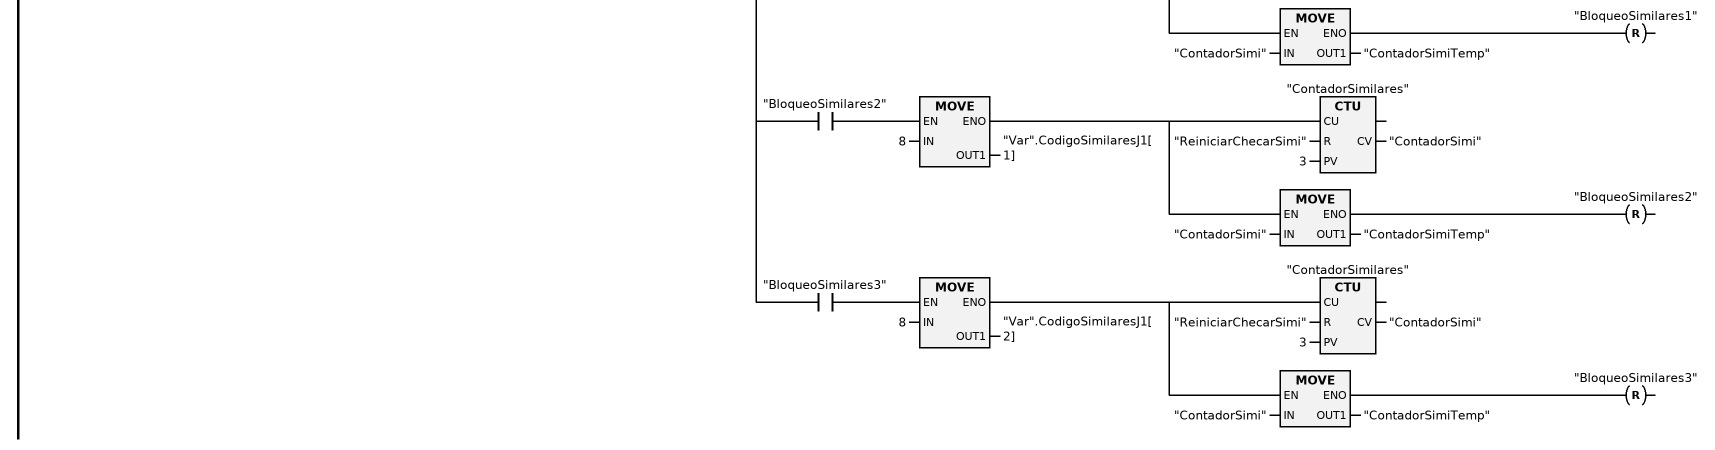
   #_w1 := "Panel1AmarilloJ1" AND ("Var".VectorPrincipalJ1["IntentoCompletoJ1", 0] = 0) AND "Bounce1";
   IF #_w1 THEN
       "Var".VectorPrincipalJ1["IntentoCompletoJ1", 0] := 7;
       "Intento0J1" := TRUE;
   END_IF;
   #_w2 := #_w1 AND ("Var".VectorPrincipalJ1["IntentoCompletoJ1", 0] = "Var".CodigoOJ1[0]);
   "ContadorCorrectas".CTU(CU := #_w2, R := "ReiniciarChecarCorr", PV := 3, CV => "ContadorCorr");
   IF #_w2 THEN
       "ContadorCorrTemp" := "ContadorCorr";
       "Var".CodigoSimilaresJ1[0] := 8;
       "BloqueoSimilares4" := TRUE;
   END_IF;
   #_w3 := #_w2 AND ("Var".CodigoSimilaresJ1[0] = 8);
   "ContadorSimilares".CTD(CD := #_w3, LD := "ReiniciarChecarSimi", PV := 3, CV => "ContadorSimi");
   IF #_w3 THEN "ContadorSimiTemp" := "ContadorSimi"; END_IF;
   #_w4 := #_w1 AND NOT "BloqueoSimilares4" AND ("Var".VectorPrincipalJ1["IntentoCompletoJ1", 0] <> "Var".CodigoOJ1[0]);
   IF #_w4 AND ("Var".VectorPrincipalJ1["IntentoCompletoJ1", 0] = "Var".CodigoSimilaresJ1[1]) THEN
       "BloqueoSimilares1" := TRUE;
   END_IF;
   #_w5 := #_w4 AND ("Var".VectorPrincipalJ1["IntentoCompletoJ1", 0] <> "Var".CodigoSimilaresJ1[1]);
   IF #_w5 AND ("Var".VectorPrincipalJ1["IntentoCompletoJ1", 0] = "Var".CodigoSimilaresJ1[2]) THEN
       "BloqueoSimilares2" := TRUE;
   END_IF;
   IF #_w5 AND ("Var".VectorPrincipalJ1["IntentoCompletoJ1", 0] <> "Var".CodigoSimilaresJ1[2]) AND ("Var".VectorPrincipalJ1["IntentoCompletoJ1", 0] = "Var".CodigoSimilaresJ1[3]) THEN
       "BloqueoSimilares3" := TRUE;
   END_IF;
   #_w6 := #_w1 AND "BloqueoSimilares1";
   IF #_w6 THEN "Var".CodigoSimilaresJ1[1] := 8; END_IF;
   "ContadorSimilares".CTU(CU := #_w6, R := "ReiniciarChecarSimi", PV := 3, CV => "ContadorSimi");
   IF #_w6 THEN
       "ContadorSimiTemp" := "ContadorSimi";
       "BloqueoSimilares1" := FALSE;
   END_IF;
   #_w7 := #_w1 AND "BloqueoSimilares2";
   IF #_w7 THEN "Var".CodigoSimilaresJ1[2] := 8; END_IF;
   "ContadorSimilares".CTU(CU := #_w7, R := "ReiniciarChecarSimi", PV := 3, CV => "ContadorSimi");
   IF #_w7 THEN
       "ContadorSimiTemp" := "ContadorSimi";
       "BloqueoSimilares2" := FALSE;
   END_IF;
   #_w8 := #_w1 AND "BloqueoSimilares3";
   IF #_w8 THEN "Var".CodigoSimilaresJ1[3] := 8; END_IF;
   "ContadorSimilares".CTU(CU := #_w8, R := "ReiniciarChecarSimi", PV := 3, CV => "ContadorSimi");
   IF #_w8 THEN
       "ContadorSimiTemp" := "ContadorSimi";
       "BloqueoSimilares3" := FALSE;
   END_IF;
   #_w9 := "Panel1AmarilloJ1" AND "Bounce2" AND "Panel1AmarilloJ1" AND "Intento0J1" AND ("Var".VectorPrincipalJ1["IntentoCompletoJ1", 1] = 0);
   IF #_w9 THEN
       "Var".VectorPrincipalJ1["IntentoCompletoJ1", 1] := 7;
       "Intento1J1" := TRUE;
   END_IF;
   #_w10 := #_w9 AND ("Var".VectorPrincipalJ1["IntentoCompletoJ1", 1] = "Var".CodigoOJ1[1]);
   "ContadorCorrectas".CTU(CU := #_w10, R := "ReiniciarChecarCorr", PV := 3, CV => "ContadorCorr");
   IF #_w10 THEN
       "ContadorCorrTemp" := "ContadorCorr";
       "Var".CodigoSimilaresJ1[1] := 8;
       "BloqueoSimilares4" := TRUE;
   END_IF;
   #_w11 := #_w10 AND ("Var".CodigoSimilaresJ1[1] = 8);
   "ContadorSimilares".CTD(CD := #_w11, LD := "ReiniciarChecarSimi", PV := 3, CV => "ContadorSimi");
   IF #_w11 THEN "ContadorSimiTemp" := "ContadorSimi"; END_IF;
   #_w12 := #_w9 AND NOT "BloqueoSimilares4" AND ("Var".VectorPrincipalJ1["IntentoCompletoJ1", 1] <> "Var".CodigoOJ1[1]);
   IF #_w12 AND ("Var".VectorPrincipalJ1["IntentoCompletoJ1", 1] = "Var".CodigoSimilaresJ1[0]) THEN
       "BloqueoSimilares1" := TRUE;
   END_IF;
   #_w13 := #_w12 AND ("Var".VectorPrincipalJ1["IntentoCompletoJ1", 1] <> "Var".CodigoSimilaresJ1[0]);
   IF #_w13 AND ("Var".VectorPrincipalJ1["IntentoCompletoJ1", 1] = "Var".CodigoSimilaresJ1[2]) THEN
       "BloqueoSimilares2" := TRUE;
   END_IF;
   IF #_w13 AND ("Var".VectorPrincipalJ1["IntentoCompletoJ1", 1] <> "Var".CodigoSimilaresJ1[2]) AND ("Var".VectorPrincipalJ1["IntentoCompletoJ1", 1] = "Var".CodigoSimilaresJ1[3]) THEN
       "BloqueoSimilares3" := TRUE;
   END_IF;
   #_w14 := #_w9 AND "BloqueoSimilares1";
   IF #_w14 THEN "Var".CodigoSimilaresJ1[0] := 8; END_IF;
   "ContadorSimilares".CTU(CU := #_w14, R := "ReiniciarChecarSimi", PV := 3, CV => "ContadorSimi");
   IF #_w14 THEN
       "ContadorSimiTemp" := "ContadorSimi";
       "BloqueoSimilares1" := FALSE;
   END_IF;
   #_w15 := #_w9 AND "BloqueoSimilares2";
   IF #_w15 THEN "Var".CodigoSimilaresJ1[2] := 8; END_IF;
   "ContadorSimilares".CTU(CU := #_w15, R := "ReiniciarChecarSimi", PV := 3, CV => "ContadorSimi");
   IF #_w15 THEN
       "ContadorSimiTemp" := "ContadorSimi";
       "BloqueoSimilares2" := FALSE;
   END_IF;
   #_w16 := #_w9 AND "BloqueoSimilares3";
   IF #_w16 THEN "Var".CodigoSimilaresJ1[3] := 8; END_IF;
   "ContadorSimilares".CTU(CU := #_w16, R := "ReiniciarChecarSimi", PV := 3, CV => "ContadorSimi");
   IF #_w16 THEN
       "ContadorSimiTemp" := "ContadorSimi";
       "BloqueoSimilares3" := FALSE;
   END_IF;
   #_w17 := "Panel1AmarilloJ1" AND "Bounce3" AND "Panel1AmarilloJ1" AND "Intento1J1" AND ("Var".VectorPrincipalJ1["IntentoCompletoJ1", 2] = 0);
   IF #_w17 THEN
       "Var".VectorPrincipalJ1["IntentoCompletoJ1", 2] := 7;
       "Intento2J1" := TRUE;
   END_IF;
   #_w18 := #_w17 AND ("Var".VectorPrincipalJ1["IntentoCompletoJ1", 2] = "Var".CodigoOJ1[2]);
   "ContadorCorrectas".CTU(CU := #_w18, R := "ReiniciarChecarCorr", PV := 3, CV => "ContadorCorr");
   IF #_w18 THEN
       "ContadorCorrTemp" := "ContadorCorr";
       "Var".CodigoSimilaresJ1[2] := 8;
       "BloqueoSimilares4" := TRUE;
   END_IF;
   #_w19 := #_w18 AND ("Var".CodigoSimilaresJ1[2] = 8);
   "ContadorSimilares".CTD(CD := #_w19, LD := "ReiniciarChecarSimi", PV := 3, CV => "ContadorSimi");
   IF #_w19 THEN "ContadorSimiTemp" := "ContadorSimi"; END_IF;
   #_w20 := #_w17 AND NOT "BloqueoSimilares4" AND ("Var".VectorPrincipalJ1["IntentoCompletoJ1", 2] <> "Var".CodigoOJ1[2]);
   IF #_w20 AND ("Var".VectorPrincipalJ1["IntentoCompletoJ1", 2] = "Var".CodigoSimilaresJ1[0]) THEN
       "BloqueoSimilares1" := TRUE;
   END_IF;
   #_w21 := #_w20 AND ("Var".VectorPrincipalJ1["IntentoCompletoJ1", 2] <> "Var".CodigoSimilaresJ1[0]);
   IF #_w21 AND ("Var".VectorPrincipalJ1["IntentoCompletoJ1", 2] = "Var".CodigoSimilaresJ1[1]) THEN
       "BloqueoSimilares2" := TRUE;
   END_IF;
   IF #_w21 AND ("Var".VectorPrincipalJ1["IntentoCompletoJ1", 2] <> "Var".CodigoSimilaresJ1[1]) AND ("Var".VectorPrincipalJ1["IntentoCompletoJ1", 2] = "Var".CodigoSimilaresJ1[3]) THEN
       "BloqueoSimilares3" := TRUE;
   END_IF;
   #_w22 := #_w17 AND "BloqueoSimilares1";
   IF #_w22 THEN "Var".CodigoSimilaresJ1[0] := 8; END_IF;
   "ContadorSimilares".CTU(CU := #_w22, R := "ReiniciarChecarSimi", PV := 3, CV => "ContadorSimi");
   IF #_w22 THEN
       "ContadorSimiTemp" := "ContadorSimi";
       "BloqueoSimilares1" := FALSE;
   END_IF;
   #_w23 := #_w17 AND "BloqueoSimilares2";
   IF #_w23 THEN "Var".CodigoSimilaresJ1[1] := 8; END_IF;
   "ContadorSimilares".CTU(CU := #_w23, R := "ReiniciarChecarSimi", PV := 3, CV => "ContadorSimi");
   IF #_w23 THEN
       "ContadorSimiTemp" := "ContadorSimi";
       "BloqueoSimilares2" := FALSE;
   END_IF;
   #_w24 := #_w17 AND "BloqueoSimilares3";
   IF #_w24 THEN "Var".CodigoSimilaresJ1[3] := 8; END_IF;
   "ContadorSimilares".CTU(CU := #_w24, R := "ReiniciarChecarSimi", PV := 3, CV => "ContadorSimi");
   IF #_w24 THEN
       "ContadorSimiTemp" := "ContadorSimi";
       "BloqueoSimilares3" := FALSE;
   END_IF;
   #_w25 := "Panel1AmarilloJ1" AND "Bounce4" AND "Panel1AmarilloJ1" AND "Intento2J1" AND ("Var".VectorPrincipalJ1["IntentoCompletoJ1", 3] = 0);
   IF #_w25 THEN
       "Var".VectorPrincipalJ1["IntentoCompletoJ1", 3] := 7;
       "Intento3J1" := TRUE;
   END_IF;
   #_w26 := #_w25 AND ("Var".VectorPrincipalJ1["IntentoCompletoJ1", 3] = "Var".CodigoOJ1[3]);
   "ContadorCorrectas".CTU(CU := #_w26, R := "ReiniciarChecarCorr", PV := 3, CV => "ContadorCorr");
   IF #_w26 THEN
       "ContadorCorrTemp" := "ContadorCorr";
       "Var".CodigoSimilaresJ1[3] := 8;
       "BloqueoSimilares4" := TRUE;
   END_IF;
   #_w27 := #_w26 AND ("Var".CodigoSimilaresJ1[3] = 8);
   "ContadorSimilares".CTD(CD := #_w27, LD := "ReiniciarChecarSimi", PV := 3, CV => "ContadorSimi");
   IF #_w27 THEN "ContadorSimiTemp" := "ContadorSimi"; END_IF;
   #_w28 := #_w25 AND NOT "BloqueoSimilares4" AND ("Var".VectorPrincipalJ1["IntentoCompletoJ1", 3] <> "Var".CodigoOJ1[3]);
   IF #_w28 AND ("Var".VectorPrincipalJ1["IntentoCompletoJ1", 3] = "Var".CodigoSimilaresJ1[0]) THEN
       "BloqueoSimilares1" := TRUE;
   END_IF;
   #_w29 := #_w28 AND ("Var".VectorPrincipalJ1["IntentoCompletoJ1", 3] <> "Var".CodigoSimilaresJ1[0]);
   IF #_w29 AND ("Var".VectorPrincipalJ1["IntentoCompletoJ1", 3] = "Var".CodigoSimilaresJ1[1]) THEN
       "BloqueoSimilares2" := TRUE;
   END_IF;
   IF #_w29 AND ("Var".VectorPrincipalJ1["IntentoCompletoJ1", 3] <> "Var".CodigoSimilaresJ1[1]) AND ("Var".VectorPrincipalJ1["IntentoCompletoJ1", 3] = "Var".CodigoSimilaresJ1[2]) THEN
       "BloqueoSimilares3" := TRUE;
   END_IF;
   #_w30 := #_w25 AND "BloqueoSimilares1";
   IF #_w30 THEN "Var".CodigoSimilaresJ1[0] := 8; END_IF;
   "ContadorSimilares".CTU(CU := #_w30, R := "ReiniciarChecarSimi", PV := 3, CV => "ContadorSimi");
   IF #_w30 THEN
       "ContadorSimiTemp" := "ContadorSimi";
       "BloqueoSimilares1" := FALSE;
   END_IF;
   #_w31 := #_w25 AND "BloqueoSimilares2";
   IF #_w31 THEN "Var".CodigoSimilaresJ1[1] := 8; END_IF;
   "ContadorSimilares".CTU(CU := #_w31, R := "ReiniciarChecarSimi", PV := 3, CV => "ContadorSimi");
   IF #_w31 THEN
       "ContadorSimiTemp" := "ContadorSimi";
       "BloqueoSimilares2" := FALSE;
   END_IF;
   #_w32 := #_w25 AND "BloqueoSimilares3";
   IF #_w32 THEN "Var".CodigoSimilaresJ1[2] := 8; END_IF;
   "ContadorSimilares".CTU(CU := #_w32, R := "ReiniciarChecarSimi", PV := 3, CV => "ContadorSimi");
   IF #_w32 THEN
       "ContadorSimiTemp" := "ContadorSimi";
       "BloqueoSimilares3" := FALSE;
   END_IF;
END_REGION

REGION Network 13: Comprobar Intentos
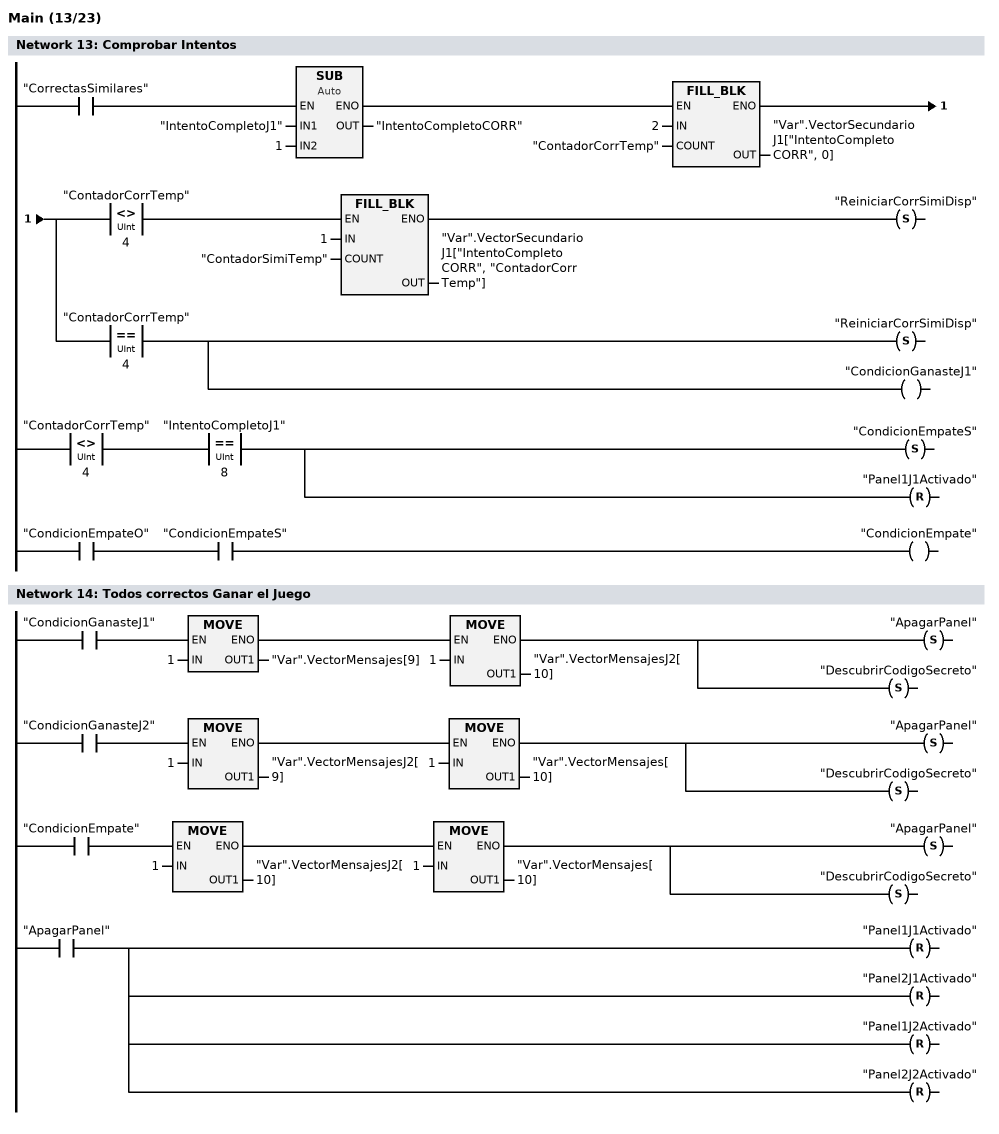
   RUNG wire#powerrail
      Contact( "CorrectasSimilares" )
      Sub(in1 := "IntentoCompletoJ1", in2 := 1, out => "IntentoCompletoCORR")
      FillBlockI(in := 2, count := "ContadorCorrTemp", out => "Var".VectorSecundarioJ1["IntentoCompletoCORR", 0])
      wire#w1
      { S7_Templates := "SrcType := UInt" } NE_Contact(in1 := "ContadorCorrTemp", in2 := 4)
      FillBlockI(in := 1, count := "ContadorSimiTemp", out => "Var".VectorSecundarioJ1["IntentoCompletoCORR", "ContadorCorrTemp"])
      S_Coil( "ReiniciarCorrSimiDisp" )
   END_RUNG
   RUNG wire#w1
      { S7_Templates := "SrcType := UInt" } EQ_Contact(in1 := "ContadorCorrTemp", in2 := 4)
      wire#w2
      S_Coil( "ReiniciarCorrSimiDisp" )
   END_RUNG
   RUNG wire#w2
      Coil( "CondicionGanasteJ1" )
   END_RUNG
   RUNG wire#powerrail
      { S7_Templates := "SrcType := UInt" } NE_Contact(in1 := "ContadorCorrTemp", in2 := 4)
      { S7_Templates := "SrcType := UInt" } EQ_Contact(in1 := "IntentoCompletoJ1", in2 := 8)
      wire#w3
      S_Coil( "CondicionEmpateS" )
   END_RUNG
   RUNG wire#w3
      R_Coil( "Panel1J1Activado" )
   END_RUNG
   RUNG wire#powerrail
      Contact( "CondicionEmpateO" )
      Contact( "CondicionEmpateS" )
      Coil( "CondicionEmpate" )
   END_RUNG
   // the same network as SCL:
   IF "CorrectasSimilares" THEN "IntentoCompletoCORR" := "IntentoCompletoJ1" - 1; END_IF;
   #_w1 := "CorrectasSimilares";
   IF #_w1 THEN
       FILL_BLK(IN := 2, COUNT := "ContadorCorrTemp", OUT => "Var".VectorSecundarioJ1["IntentoCompletoCORR", 0]);
   END_IF;
   #_w2 := #_w1 AND ("ContadorCorrTemp" <> 4);
   IF #_w2 THEN
       FILL_BLK(IN := 1,
                COUNT := "ContadorSimiTemp",
                OUT => "Var".VectorSecundarioJ1["IntentoCompletoCORR", "ContadorCorrTemp"]);
       "ReiniciarCorrSimiDisp" := TRUE;
   END_IF;
   #_w3 := #_w1 AND ("ContadorCorrTemp" = 4);
   IF #_w3 THEN "ReiniciarCorrSimiDisp" := TRUE; END_IF;
   "CondicionGanasteJ1" := #_w3;
   IF ("ContadorCorrTemp" <> 4) AND ("IntentoCompletoJ1" = 8) THEN
       "CondicionEmpateS" := TRUE;
       "Panel1J1Activado" := FALSE;
   END_IF;
   "CondicionEmpate" := "CondicionEmpateO" AND "CondicionEmpateS";
END_REGION

REGION Network 14: Todos correctos Ganar el Juego
   RUNG wire#powerrail
      Contact( "CondicionGanasteJ1" )
      Move(in := 1, out1 => "Var".VectorMensajes[9])
      Move(in := 1, out1 => "Var".VectorMensajesJ2[10])
      wire#w1
      S_Coil( "ApagarPanel" )
   END_RUNG
   RUNG wire#w1
      S_Coil( "DescubrirCodigoSecreto" )
   END_RUNG
   RUNG wire#powerrail
      Contact( "CondicionGanasteJ2" )
      Move(in := 1, out1 => "Var".VectorMensajesJ2[9])
      Move(in := 1, out1 => "Var".VectorMensajes[10])
      wire#w2
      S_Coil( "ApagarPanel" )
   END_RUNG
   RUNG wire#w2
      S_Coil( "DescubrirCodigoSecreto" )
   END_RUNG
   RUNG wire#powerrail
      Contact( "CondicionEmpate" )
      Move(in := 1, out1 => "Var".VectorMensajesJ2[10])
      Move(in := 1, out1 => "Var".VectorMensajes[10])
      wire#w3
      S_Coil( "ApagarPanel" )
   END_RUNG
   RUNG wire#w3
      S_Coil( "DescubrirCodigoSecreto" )
   END_RUNG
   RUNG wire#powerrail
      Contact( "ApagarPanel" )
      wire#w4
      R_Coil( "Panel1J1Activado" )
   END_RUNG
   RUNG wire#w4
      R_Coil( "Panel2J1Activado" )
   END_RUNG
   RUNG wire#w4
      R_Coil( "Panel1J2Activado" )
   END_RUNG
   RUNG wire#w4
      R_Coil( "Panel2J2Activado" )
   END_RUNG
   // the same network as SCL:
   IF "CondicionGanasteJ1" THEN
       "Var".VectorMensajes[9] := 1;
       "Var".VectorMensajesJ2[10] := 1;
       "ApagarPanel" := TRUE;
       "DescubrirCodigoSecreto" := TRUE;
   END_IF;
   IF "CondicionGanasteJ2" THEN
       "Var".VectorMensajesJ2[9] := 1;
       "Var".VectorMensajes[10] := 1;
       "ApagarPanel" := TRUE;
       "DescubrirCodigoSecreto" := TRUE;
   END_IF;
   IF "CondicionEmpate" THEN
       "Var".VectorMensajesJ2[10] := 1;
       "Var".VectorMensajes[10] := 1;
       "ApagarPanel" := TRUE;
       "DescubrirCodigoSecreto" := TRUE;
   END_IF;
   IF "ApagarPanel" THEN
       "Panel1J1Activado" := FALSE;
       "Panel2J1Activado" := FALSE;
       "Panel1J2Activado" := FALSE;
       "Panel2J2Activado" := FALSE;
   END_IF;
END_REGION

REGION Network 16: Seleccionar Codigo J2
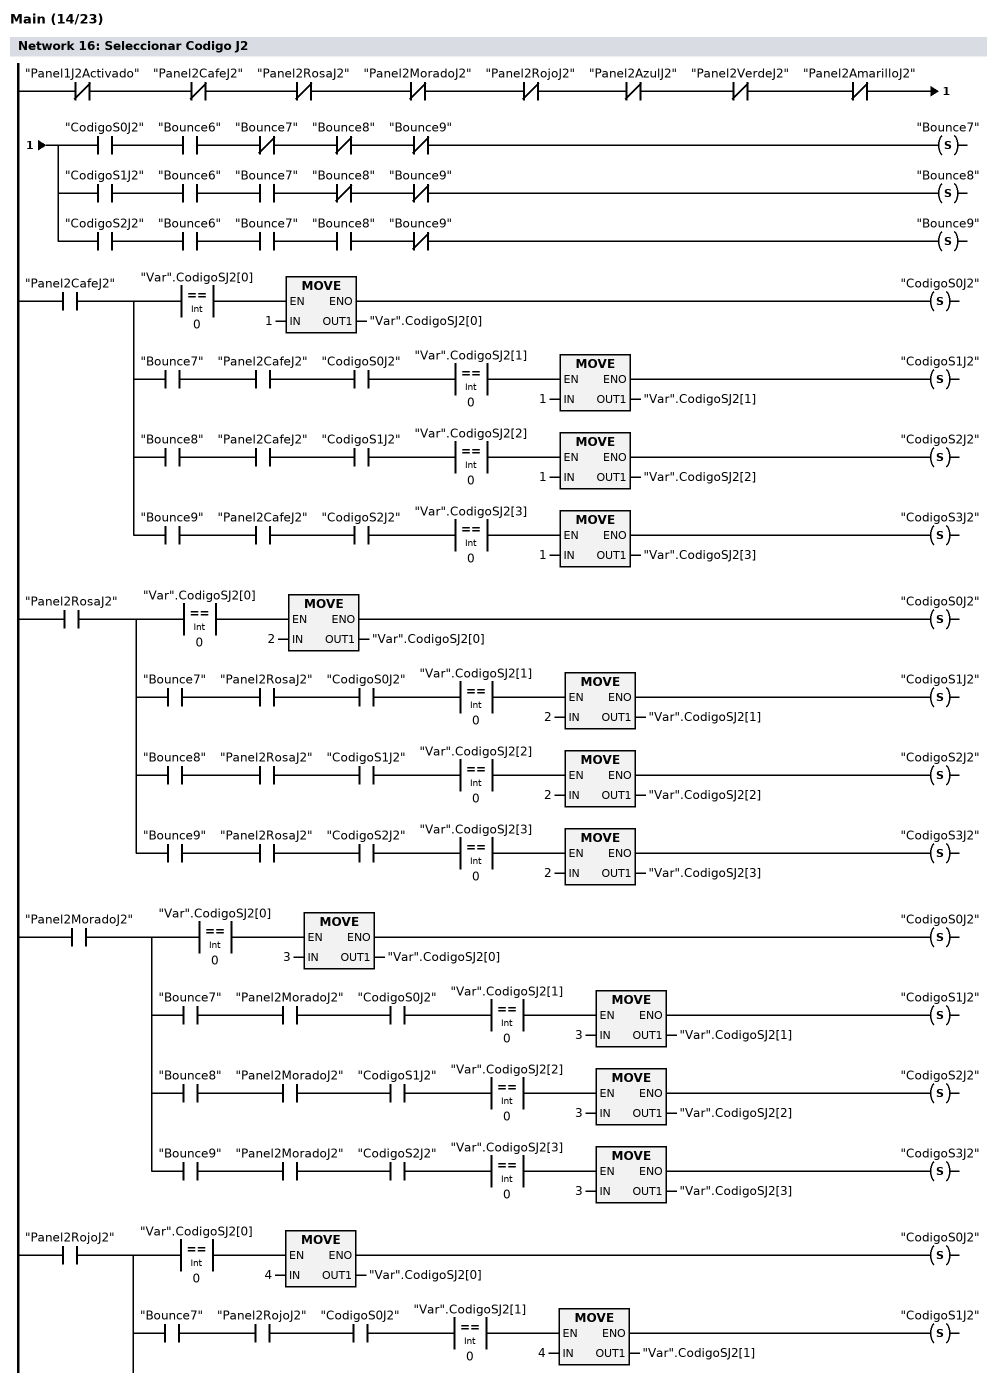
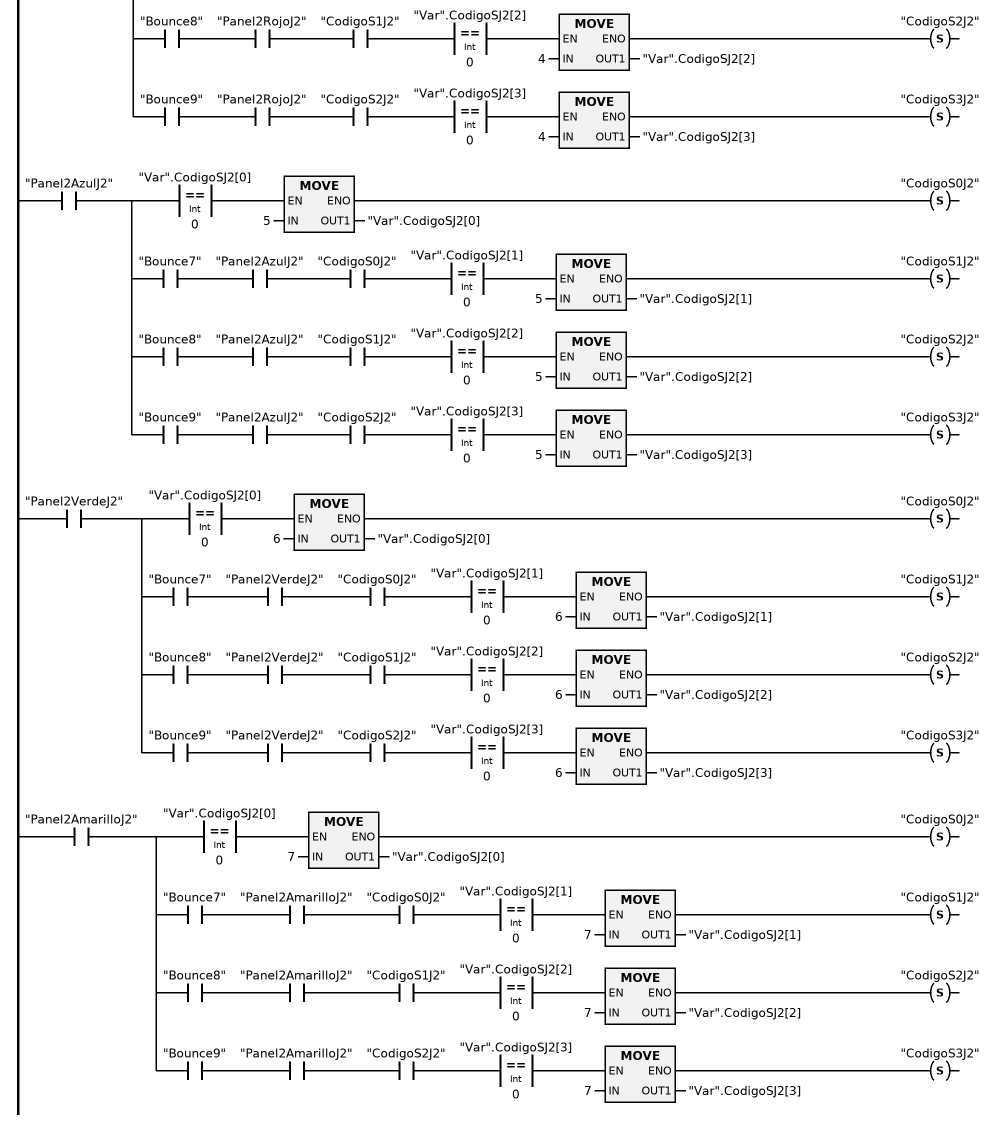
   RUNG wire#powerrail
      I_Contact( "Panel1J2Activado" )
      I_Contact( "Panel2CafeJ2" )
      I_Contact( "Panel2RosaJ2" )
      I_Contact( "Panel2MoradoJ2" )
      I_Contact( "Panel2RojoJ2" )
      I_Contact( "Panel2AzulJ2" )
      I_Contact( "Panel2VerdeJ2" )
      I_Contact( "Panel2AmarilloJ2" )
      wire#w1
      Contact( "CodigoS0J2" )
      Contact( "Bounce6" )
      I_Contact( "Bounce7" )
      I_Contact( "Bounce8" )
      I_Contact( "Bounce9" )
      S_Coil( "Bounce7" )
   END_RUNG
   RUNG wire#w1
      Contact( "CodigoS1J2" )
      Contact( "Bounce6" )
      Contact( "Bounce7" )
      I_Contact( "Bounce8" )
      I_Contact( "Bounce9" )
      S_Coil( "Bounce8" )
   END_RUNG
   RUNG wire#w1
      Contact( "CodigoS2J2" )
      Contact( "Bounce6" )
      Contact( "Bounce7" )
      Contact( "Bounce8" )
      I_Contact( "Bounce9" )
      S_Coil( "Bounce9" )
   END_RUNG
   RUNG wire#powerrail
      Contact( "Panel2CafeJ2" )
      wire#w2
      { S7_Templates := "SrcType := Int" } EQ_Contact(in1 := "Var".CodigoSJ2[0], in2 := 0)
      Move(in := 1, out1 => "Var".CodigoSJ2[0])
      S_Coil( "CodigoS0J2" )
   END_RUNG
   RUNG wire#w2
      Contact( "Bounce7" )
      Contact( "Panel2CafeJ2" )
      Contact( "CodigoS0J2" )
      { S7_Templates := "SrcType := Int" } EQ_Contact(in1 := "Var".CodigoSJ2[1], in2 := 0)
      Move(in := 1, out1 => "Var".CodigoSJ2[1])
      S_Coil( "CodigoS1J2" )
   END_RUNG
   RUNG wire#w2
      Contact( "Bounce8" )
      Contact( "Panel2CafeJ2" )
      Contact( "CodigoS1J2" )
      { S7_Templates := "SrcType := Int" } EQ_Contact(in1 := "Var".CodigoSJ2[2], in2 := 0)
      Move(in := 1, out1 => "Var".CodigoSJ2[2])
      S_Coil( "CodigoS2J2" )
   END_RUNG
   RUNG wire#w2
      Contact( "Bounce9" )
      Contact( "Panel2CafeJ2" )
      Contact( "CodigoS2J2" )
      { S7_Templates := "SrcType := Int" } EQ_Contact(in1 := "Var".CodigoSJ2[3], in2 := 0)
      Move(in := 1, out1 => "Var".CodigoSJ2[3])
      S_Coil( "CodigoS3J2" )
   END_RUNG
   RUNG wire#powerrail
      Contact( "Panel2RosaJ2" )
      wire#w3
      { S7_Templates := "SrcType := Int" } EQ_Contact(in1 := "Var".CodigoSJ2[0], in2 := 0)
      Move(in := 2, out1 => "Var".CodigoSJ2[0])
      S_Coil( "CodigoS0J2" )
   END_RUNG
   RUNG wire#w3
      Contact( "Bounce7" )
      Contact( "Panel2RosaJ2" )
      Contact( "CodigoS0J2" )
      { S7_Templates := "SrcType := Int" } EQ_Contact(in1 := "Var".CodigoSJ2[1], in2 := 0)
      Move(in := 2, out1 => "Var".CodigoSJ2[1])
      S_Coil( "CodigoS1J2" )
   END_RUNG
   RUNG wire#w3
      Contact( "Bounce8" )
      Contact( "Panel2RosaJ2" )
      Contact( "CodigoS1J2" )
      { S7_Templates := "SrcType := Int" } EQ_Contact(in1 := "Var".CodigoSJ2[2], in2 := 0)
      Move(in := 2, out1 => "Var".CodigoSJ2[2])
      S_Coil( "CodigoS2J2" )
   END_RUNG
   RUNG wire#w3
      Contact( "Bounce9" )
      Contact( "Panel2RosaJ2" )
      Contact( "CodigoS2J2" )
      { S7_Templates := "SrcType := Int" } EQ_Contact(in1 := "Var".CodigoSJ2[3], in2 := 0)
      Move(in := 2, out1 => "Var".CodigoSJ2[3])
      S_Coil( "CodigoS3J2" )
   END_RUNG
   RUNG wire#powerrail
      Contact( "Panel2MoradoJ2" )
      wire#w4
      { S7_Templates := "SrcType := Int" } EQ_Contact(in1 := "Var".CodigoSJ2[0], in2 := 0)
      Move(in := 3, out1 => "Var".CodigoSJ2[0])
      S_Coil( "CodigoS0J2" )
   END_RUNG
   RUNG wire#w4
      Contact( "Bounce7" )
      Contact( "Panel2MoradoJ2" )
      Contact( "CodigoS0J2" )
      { S7_Templates := "SrcType := Int" } EQ_Contact(in1 := "Var".CodigoSJ2[1], in2 := 0)
      Move(in := 3, out1 => "Var".CodigoSJ2[1])
      S_Coil( "CodigoS1J2" )
   END_RUNG
   RUNG wire#w4
      Contact( "Bounce8" )
      Contact( "Panel2MoradoJ2" )
      Contact( "CodigoS1J2" )
      { S7_Templates := "SrcType := Int" } EQ_Contact(in1 := "Var".CodigoSJ2[2], in2 := 0)
      Move(in := 3, out1 => "Var".CodigoSJ2[2])
      S_Coil( "CodigoS2J2" )
   END_RUNG
   RUNG wire#w4
      Contact( "Bounce9" )
      Contact( "Panel2MoradoJ2" )
      Contact( "CodigoS2J2" )
      { S7_Templates := "SrcType := Int" } EQ_Contact(in1 := "Var".CodigoSJ2[3], in2 := 0)
      Move(in := 3, out1 => "Var".CodigoSJ2[3])
      S_Coil( "CodigoS3J2" )
   END_RUNG
   RUNG wire#powerrail
      Contact( "Panel2RojoJ2" )
      wire#w5
      { S7_Templates := "SrcType := Int" } EQ_Contact(in1 := "Var".CodigoSJ2[0], in2 := 0)
      Move(in := 4, out1 => "Var".CodigoSJ2[0])
      S_Coil( "CodigoS0J2" )
   END_RUNG
   RUNG wire#w5
      Contact( "Bounce7" )
      Contact( "Panel2RojoJ2" )
      Contact( "CodigoS0J2" )
      { S7_Templates := "SrcType := Int" } EQ_Contact(in1 := "Var".CodigoSJ2[1], in2 := 0)
      Move(in := 4, out1 => "Var".CodigoSJ2[1])
      S_Coil( "CodigoS1J2" )
   END_RUNG
   RUNG wire#w5
      Contact( "Bounce8" )
      Contact( "Panel2RojoJ2" )
      Contact( "CodigoS1J2" )
      { S7_Templates := "SrcType := Int" } EQ_Contact(in1 := "Var".CodigoSJ2[2], in2 := 0)
      Move(in := 4, out1 => "Var".CodigoSJ2[2])
      S_Coil( "CodigoS2J2" )
   END_RUNG
   RUNG wire#w5
      Contact( "Bounce9" )
      Contact( "Panel2RojoJ2" )
      Contact( "CodigoS2J2" )
      { S7_Templates := "SrcType := Int" } EQ_Contact(in1 := "Var".CodigoSJ2[3], in2 := 0)
      Move(in := 4, out1 => "Var".CodigoSJ2[3])
      S_Coil( "CodigoS3J2" )
   END_RUNG
   RUNG wire#powerrail
      Contact( "Panel2AzulJ2" )
      wire#w6
      { S7_Templates := "SrcType := Int" } EQ_Contact(in1 := "Var".CodigoSJ2[0], in2 := 0)
      Move(in := 5, out1 => "Var".CodigoSJ2[0])
      S_Coil( "CodigoS0J2" )
   END_RUNG
   RUNG wire#w6
      Contact( "Bounce7" )
      Contact( "Panel2AzulJ2" )
      Contact( "CodigoS0J2" )
      { S7_Templates := "SrcType := Int" } EQ_Contact(in1 := "Var".CodigoSJ2[1], in2 := 0)
      Move(in := 5, out1 => "Var".CodigoSJ2[1])
      S_Coil( "CodigoS1J2" )
   END_RUNG
   RUNG wire#w6
      Contact( "Bounce8" )
      Contact( "Panel2AzulJ2" )
      Contact( "CodigoS1J2" )
      { S7_Templates := "SrcType := Int" } EQ_Contact(in1 := "Var".CodigoSJ2[2], in2 := 0)
      Move(in := 5, out1 => "Var".CodigoSJ2[2])
      S_Coil( "CodigoS2J2" )
   END_RUNG
   RUNG wire#w6
      Contact( "Bounce9" )
      Contact( "Panel2AzulJ2" )
      Contact( "CodigoS2J2" )
      { S7_Templates := "SrcType := Int" } EQ_Contact(in1 := "Var".CodigoSJ2[3], in2 := 0)
      Move(in := 5, out1 => "Var".CodigoSJ2[3])
      S_Coil( "CodigoS3J2" )
   END_RUNG
   RUNG wire#powerrail
      Contact( "Panel2VerdeJ2" )
      wire#w7
      { S7_Templates := "SrcType := Int" } EQ_Contact(in1 := "Var".CodigoSJ2[0], in2 := 0)
      Move(in := 6, out1 => "Var".CodigoSJ2[0])
      S_Coil( "CodigoS0J2" )
   END_RUNG
   RUNG wire#w7
      Contact( "Bounce7" )
      Contact( "Panel2VerdeJ2" )
      Contact( "CodigoS0J2" )
      { S7_Templates := "SrcType := Int" } EQ_Contact(in1 := "Var".CodigoSJ2[1], in2 := 0)
      Move(in := 6, out1 => "Var".CodigoSJ2[1])
      S_Coil( "CodigoS1J2" )
   END_RUNG
   RUNG wire#w7
      Contact( "Bounce8" )
      Contact( "Panel2VerdeJ2" )
      Contact( "CodigoS1J2" )
      { S7_Templates := "SrcType := Int" } EQ_Contact(in1 := "Var".CodigoSJ2[2], in2 := 0)
      Move(in := 6, out1 => "Var".CodigoSJ2[2])
      S_Coil( "CodigoS2J2" )
   END_RUNG
   RUNG wire#w7
      Contact( "Bounce9" )
      Contact( "Panel2VerdeJ2" )
      Contact( "CodigoS2J2" )
      { S7_Templates := "SrcType := Int" } EQ_Contact(in1 := "Var".CodigoSJ2[3], in2 := 0)
      Move(in := 6, out1 => "Var".CodigoSJ2[3])
      S_Coil( "CodigoS3J2" )
   END_RUNG
   RUNG wire#powerrail
      Contact( "Panel2AmarilloJ2" )
      wire#w8
      { S7_Templates := "SrcType := Int" } EQ_Contact(in1 := "Var".CodigoSJ2[0], in2 := 0)
      Move(in := 7, out1 => "Var".CodigoSJ2[0])
      S_Coil( "CodigoS0J2" )
   END_RUNG
   RUNG wire#w8
      Contact( "Bounce7" )
      Contact( "Panel2AmarilloJ2" )
      Contact( "CodigoS0J2" )
      { S7_Templates := "SrcType := Int" } EQ_Contact(in1 := "Var".CodigoSJ2[1], in2 := 0)
      Move(in := 7, out1 => "Var".CodigoSJ2[1])
      S_Coil( "CodigoS1J2" )
   END_RUNG
   RUNG wire#w8
      Contact( "Bounce8" )
      Contact( "Panel2AmarilloJ2" )
      Contact( "CodigoS1J2" )
      { S7_Templates := "SrcType := Int" } EQ_Contact(in1 := "Var".CodigoSJ2[2], in2 := 0)
      Move(in := 7, out1 => "Var".CodigoSJ2[2])
      S_Coil( "CodigoS2J2" )
   END_RUNG
   RUNG wire#w8
      Contact( "Bounce9" )
      Contact( "Panel2AmarilloJ2" )
      Contact( "CodigoS2J2" )
      { S7_Templates := "SrcType := Int" } EQ_Contact(in1 := "Var".CodigoSJ2[3], in2 := 0)
      Move(in := 7, out1 => "Var".CodigoSJ2[3])
      S_Coil( "CodigoS3J2" )
   END_RUNG
   // the same network as SCL:
   #_w1 := NOT "Panel1J2Activado" AND NOT "Panel2CafeJ2" AND NOT "Panel2RosaJ2" AND NOT "Panel2MoradoJ2" AND NOT "Panel2RojoJ2" AND NOT "Panel2AzulJ2" AND NOT "Panel2VerdeJ2" AND NOT "Panel2AmarilloJ2";
   IF #_w1 AND "CodigoS0J2" AND "Bounce6" AND NOT "Bounce7" AND NOT "Bounce8" AND NOT "Bounce9" THEN
       "Bounce7" := TRUE;
   END_IF;
   IF #_w1 AND "CodigoS1J2" AND "Bounce6" AND "Bounce7" AND NOT "Bounce8" AND NOT "Bounce9" THEN
       "Bounce8" := TRUE;
   END_IF;
   IF #_w1 AND "CodigoS2J2" AND "Bounce6" AND "Bounce7" AND "Bounce8" AND NOT "Bounce9" THEN
       "Bounce9" := TRUE;
   END_IF;
   #_w2 := "Panel2CafeJ2" AND ("Var".CodigoSJ2[0] = 0);
   IF #_w2 THEN
       "Var".CodigoSJ2[0] := 1;
       "CodigoS0J2" := TRUE;
   END_IF;
   #_w3 := "Panel2CafeJ2" AND "Bounce7" AND "Panel2CafeJ2" AND "CodigoS0J2" AND ("Var".CodigoSJ2[1] = 0);
   IF #_w3 THEN
       "Var".CodigoSJ2[1] := 1;
       "CodigoS1J2" := TRUE;
   END_IF;
   #_w4 := "Panel2CafeJ2" AND "Bounce8" AND "Panel2CafeJ2" AND "CodigoS1J2" AND ("Var".CodigoSJ2[2] = 0);
   IF #_w4 THEN
       "Var".CodigoSJ2[2] := 1;
       "CodigoS2J2" := TRUE;
   END_IF;
   #_w5 := "Panel2CafeJ2" AND "Bounce9" AND "Panel2CafeJ2" AND "CodigoS2J2" AND ("Var".CodigoSJ2[3] = 0);
   IF #_w5 THEN
       "Var".CodigoSJ2[3] := 1;
       "CodigoS3J2" := TRUE;
   END_IF;
   #_w6 := "Panel2RosaJ2" AND ("Var".CodigoSJ2[0] = 0);
   IF #_w6 THEN
       "Var".CodigoSJ2[0] := 2;
       "CodigoS0J2" := TRUE;
   END_IF;
   #_w7 := "Panel2RosaJ2" AND "Bounce7" AND "Panel2RosaJ2" AND "CodigoS0J2" AND ("Var".CodigoSJ2[1] = 0);
   IF #_w7 THEN
       "Var".CodigoSJ2[1] := 2;
       "CodigoS1J2" := TRUE;
   END_IF;
   #_w8 := "Panel2RosaJ2" AND "Bounce8" AND "Panel2RosaJ2" AND "CodigoS1J2" AND ("Var".CodigoSJ2[2] = 0);
   IF #_w8 THEN
       "Var".CodigoSJ2[2] := 2;
       "CodigoS2J2" := TRUE;
   END_IF;
   #_w9 := "Panel2RosaJ2" AND "Bounce9" AND "Panel2RosaJ2" AND "CodigoS2J2" AND ("Var".CodigoSJ2[3] = 0);
   IF #_w9 THEN
       "Var".CodigoSJ2[3] := 2;
       "CodigoS3J2" := TRUE;
   END_IF;
   #_w10 := "Panel2MoradoJ2" AND ("Var".CodigoSJ2[0] = 0);
   IF #_w10 THEN
       "Var".CodigoSJ2[0] := 3;
       "CodigoS0J2" := TRUE;
   END_IF;
   #_w11 := "Panel2MoradoJ2" AND "Bounce7" AND "Panel2MoradoJ2" AND "CodigoS0J2" AND ("Var".CodigoSJ2[1] = 0);
   IF #_w11 THEN
       "Var".CodigoSJ2[1] := 3;
       "CodigoS1J2" := TRUE;
   END_IF;
   #_w12 := "Panel2MoradoJ2" AND "Bounce8" AND "Panel2MoradoJ2" AND "CodigoS1J2" AND ("Var".CodigoSJ2[2] = 0);
   IF #_w12 THEN
       "Var".CodigoSJ2[2] := 3;
       "CodigoS2J2" := TRUE;
   END_IF;
   #_w13 := "Panel2MoradoJ2" AND "Bounce9" AND "Panel2MoradoJ2" AND "CodigoS2J2" AND ("Var".CodigoSJ2[3] = 0);
   IF #_w13 THEN
       "Var".CodigoSJ2[3] := 3;
       "CodigoS3J2" := TRUE;
   END_IF;
   #_w14 := "Panel2RojoJ2" AND ("Var".CodigoSJ2[0] = 0);
   IF #_w14 THEN
       "Var".CodigoSJ2[0] := 4;
       "CodigoS0J2" := TRUE;
   END_IF;
   #_w15 := "Panel2RojoJ2" AND "Bounce7" AND "Panel2RojoJ2" AND "CodigoS0J2" AND ("Var".CodigoSJ2[1] = 0);
   IF #_w15 THEN
       "Var".CodigoSJ2[1] := 4;
       "CodigoS1J2" := TRUE;
   END_IF;
   #_w16 := "Panel2RojoJ2" AND "Bounce8" AND "Panel2RojoJ2" AND "CodigoS1J2" AND ("Var".CodigoSJ2[2] = 0);
   IF #_w16 THEN
       "Var".CodigoSJ2[2] := 4;
       "CodigoS2J2" := TRUE;
   END_IF;
   #_w17 := "Panel2RojoJ2" AND "Bounce9" AND "Panel2RojoJ2" AND "CodigoS2J2" AND ("Var".CodigoSJ2[3] = 0);
   IF #_w17 THEN
       "Var".CodigoSJ2[3] := 4;
       "CodigoS3J2" := TRUE;
   END_IF;
   #_w18 := "Panel2AzulJ2" AND ("Var".CodigoSJ2[0] = 0);
   IF #_w18 THEN
       "Var".CodigoSJ2[0] := 5;
       "CodigoS0J2" := TRUE;
   END_IF;
   #_w19 := "Panel2AzulJ2" AND "Bounce7" AND "Panel2AzulJ2" AND "CodigoS0J2" AND ("Var".CodigoSJ2[1] = 0);
   IF #_w19 THEN
       "Var".CodigoSJ2[1] := 5;
       "CodigoS1J2" := TRUE;
   END_IF;
   #_w20 := "Panel2AzulJ2" AND "Bounce8" AND "Panel2AzulJ2" AND "CodigoS1J2" AND ("Var".CodigoSJ2[2] = 0);
   IF #_w20 THEN
       "Var".CodigoSJ2[2] := 5;
       "CodigoS2J2" := TRUE;
   END_IF;
   #_w21 := "Panel2AzulJ2" AND "Bounce9" AND "Panel2AzulJ2" AND "CodigoS2J2" AND ("Var".CodigoSJ2[3] = 0);
   IF #_w21 THEN
       "Var".CodigoSJ2[3] := 5;
       "CodigoS3J2" := TRUE;
   END_IF;
   #_w22 := "Panel2VerdeJ2" AND ("Var".CodigoSJ2[0] = 0);
   IF #_w22 THEN
       "Var".CodigoSJ2[0] := 6;
       "CodigoS0J2" := TRUE;
   END_IF;
   #_w23 := "Panel2VerdeJ2" AND "Bounce7" AND "Panel2VerdeJ2" AND "CodigoS0J2" AND ("Var".CodigoSJ2[1] = 0);
   IF #_w23 THEN
       "Var".CodigoSJ2[1] := 6;
       "CodigoS1J2" := TRUE;
   END_IF;
   #_w24 := "Panel2VerdeJ2" AND "Bounce8" AND "Panel2VerdeJ2" AND "CodigoS1J2" AND ("Var".CodigoSJ2[2] = 0);
   IF #_w24 THEN
       "Var".CodigoSJ2[2] := 6;
       "CodigoS2J2" := TRUE;
   END_IF;
   #_w25 := "Panel2VerdeJ2" AND "Bounce9" AND "Panel2VerdeJ2" AND "CodigoS2J2" AND ("Var".CodigoSJ2[3] = 0);
   IF #_w25 THEN
       "Var".CodigoSJ2[3] := 6;
       "CodigoS3J2" := TRUE;
   END_IF;
   #_w26 := "Panel2AmarilloJ2" AND ("Var".CodigoSJ2[0] = 0);
   IF #_w26 THEN
       "Var".CodigoSJ2[0] := 7;
       "CodigoS0J2" := TRUE;
   END_IF;
   #_w27 := "Panel2AmarilloJ2" AND "Bounce7" AND "Panel2AmarilloJ2" AND "CodigoS0J2" AND ("Var".CodigoSJ2[1] = 0);
   IF #_w27 THEN
       "Var".CodigoSJ2[1] := 7;
       "CodigoS1J2" := TRUE;
   END_IF;
   #_w28 := "Panel2AmarilloJ2" AND "Bounce8" AND "Panel2AmarilloJ2" AND "CodigoS1J2" AND ("Var".CodigoSJ2[2] = 0);
   IF #_w28 THEN
       "Var".CodigoSJ2[2] := 7;
       "CodigoS2J2" := TRUE;
   END_IF;
   #_w29 := "Panel2AmarilloJ2" AND "Bounce9" AND "Panel2AmarilloJ2" AND "CodigoS2J2" AND ("Var".CodigoSJ2[3] = 0);
   IF #_w29 THEN
       "Var".CodigoSJ2[3] := 7;
       "CodigoS3J2" := TRUE;
   END_IF;
END_REGION

REGION Network 17: Clave Secreta J2
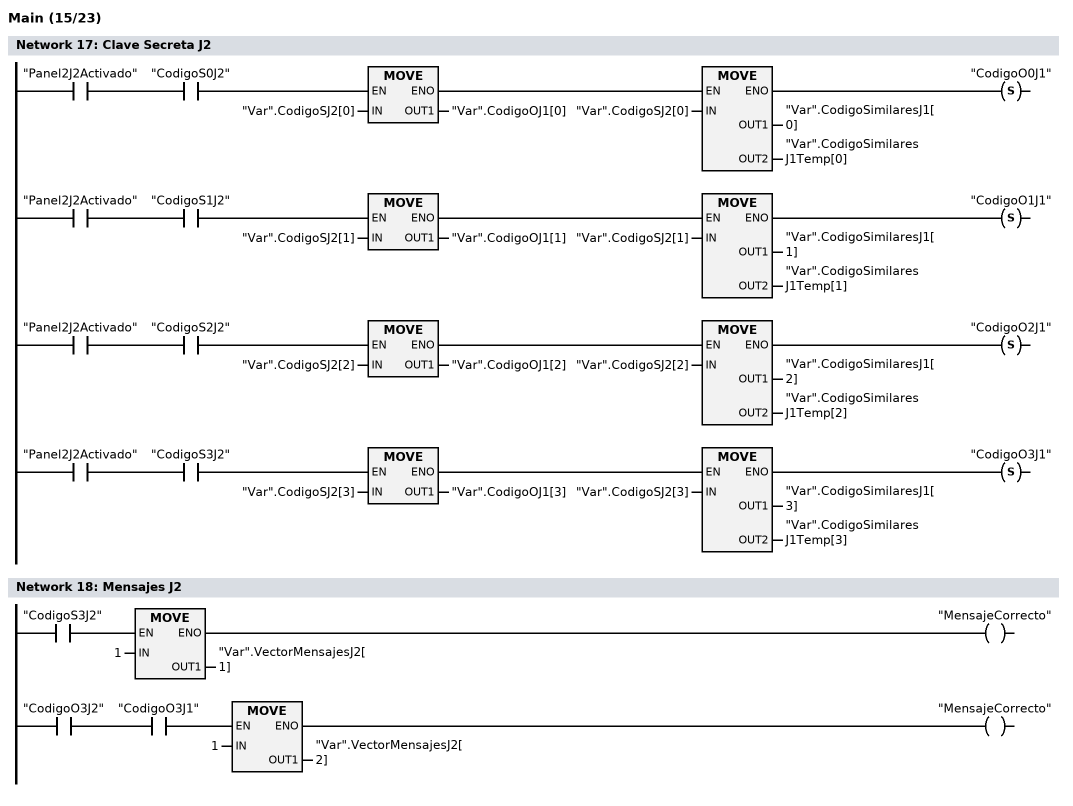
   RUNG wire#powerrail
      Contact( "Panel2J2Activado" )
      Contact( "CodigoS0J2" )
      Move(in := "Var".CodigoSJ2[0], out1 => "Var".CodigoOJ1[0])
      Move(in := "Var".CodigoSJ2[0], out1 => "Var".CodigoSimilaresJ1[0], out2 => "Var".CodigoSimilaresJ1Temp[0])
      S_Coil( "CodigoO0J1" )
   END_RUNG
   RUNG wire#powerrail
      Contact( "Panel2J2Activado" )
      Contact( "CodigoS1J2" )
      Move(in := "Var".CodigoSJ2[1], out1 => "Var".CodigoOJ1[1])
      Move(in := "Var".CodigoSJ2[1], out1 => "Var".CodigoSimilaresJ1[1], out2 => "Var".CodigoSimilaresJ1Temp[1])
      S_Coil( "CodigoO1J1" )
   END_RUNG
   RUNG wire#powerrail
      Contact( "Panel2J2Activado" )
      Contact( "CodigoS2J2" )
      Move(in := "Var".CodigoSJ2[2], out1 => "Var".CodigoOJ1[2])
      Move(in := "Var".CodigoSJ2[2], out1 => "Var".CodigoSimilaresJ1[2], out2 => "Var".CodigoSimilaresJ1Temp[2])
      S_Coil( "CodigoO2J1" )
   END_RUNG
   RUNG wire#powerrail
      Contact( "Panel2J2Activado" )
      Contact( "CodigoS3J2" )
      Move(in := "Var".CodigoSJ2[3], out1 => "Var".CodigoOJ1[3])
      Move(in := "Var".CodigoSJ2[3], out1 => "Var".CodigoSimilaresJ1[3], out2 => "Var".CodigoSimilaresJ1Temp[3])
      S_Coil( "CodigoO3J1" )
   END_RUNG
   // the same network as SCL:
   IF "Panel2J2Activado" AND "CodigoS0J2" THEN
       "Var".CodigoOJ1[0] := "Var".CodigoSJ2[0];
       "Var".CodigoSimilaresJ1[0] := "Var".CodigoSJ2[0];
       "Var".CodigoSimilaresJ1Temp[0] := "Var".CodigoSJ2[0];
       "CodigoO0J1" := TRUE;
   END_IF;
   IF "Panel2J2Activado" AND "CodigoS1J2" THEN
       "Var".CodigoOJ1[1] := "Var".CodigoSJ2[1];
       "Var".CodigoSimilaresJ1[1] := "Var".CodigoSJ2[1];
       "Var".CodigoSimilaresJ1Temp[1] := "Var".CodigoSJ2[1];
       "CodigoO1J1" := TRUE;
   END_IF;
   IF "Panel2J2Activado" AND "CodigoS2J2" THEN
       "Var".CodigoOJ1[2] := "Var".CodigoSJ2[2];
       "Var".CodigoSimilaresJ1[2] := "Var".CodigoSJ2[2];
       "Var".CodigoSimilaresJ1Temp[2] := "Var".CodigoSJ2[2];
       "CodigoO2J1" := TRUE;
   END_IF;
   IF "Panel2J2Activado" AND "CodigoS3J2" THEN
       "Var".CodigoOJ1[3] := "Var".CodigoSJ2[3];
       "Var".CodigoSimilaresJ1[3] := "Var".CodigoSJ2[3];
       "Var".CodigoSimilaresJ1Temp[3] := "Var".CodigoSJ2[3];
       "CodigoO3J1" := TRUE;
   END_IF;
END_REGION

REGION Network 18: Mensajes J2
   RUNG wire#powerrail
      Contact( "CodigoS3J2" )
      Move(in := 1, out1 => "Var".VectorMensajesJ2[1])
      Coil( "MensajeCorrecto" )
   END_RUNG
   RUNG wire#powerrail
      Contact( "CodigoO3J2" )
      Contact( "CodigoO3J1" )
      Move(in := 1, out1 => "Var".VectorMensajesJ2[2])
      Coil( "MensajeCorrecto" )
   END_RUNG
   // the same network as SCL:
   IF "CodigoS3J2" THEN "Var".VectorMensajesJ2[1] := 1; END_IF;
   "MensajeCorrecto" := "CodigoS3J2";
   #_w1 := "CodigoO3J2" AND "CodigoO3J1";
   IF #_w1 THEN "Var".VectorMensajesJ2[2] := 1; END_IF;
   "MensajeCorrecto" := #_w1;
END_REGION

REGION Network 19: Seleccionar Intentos J2
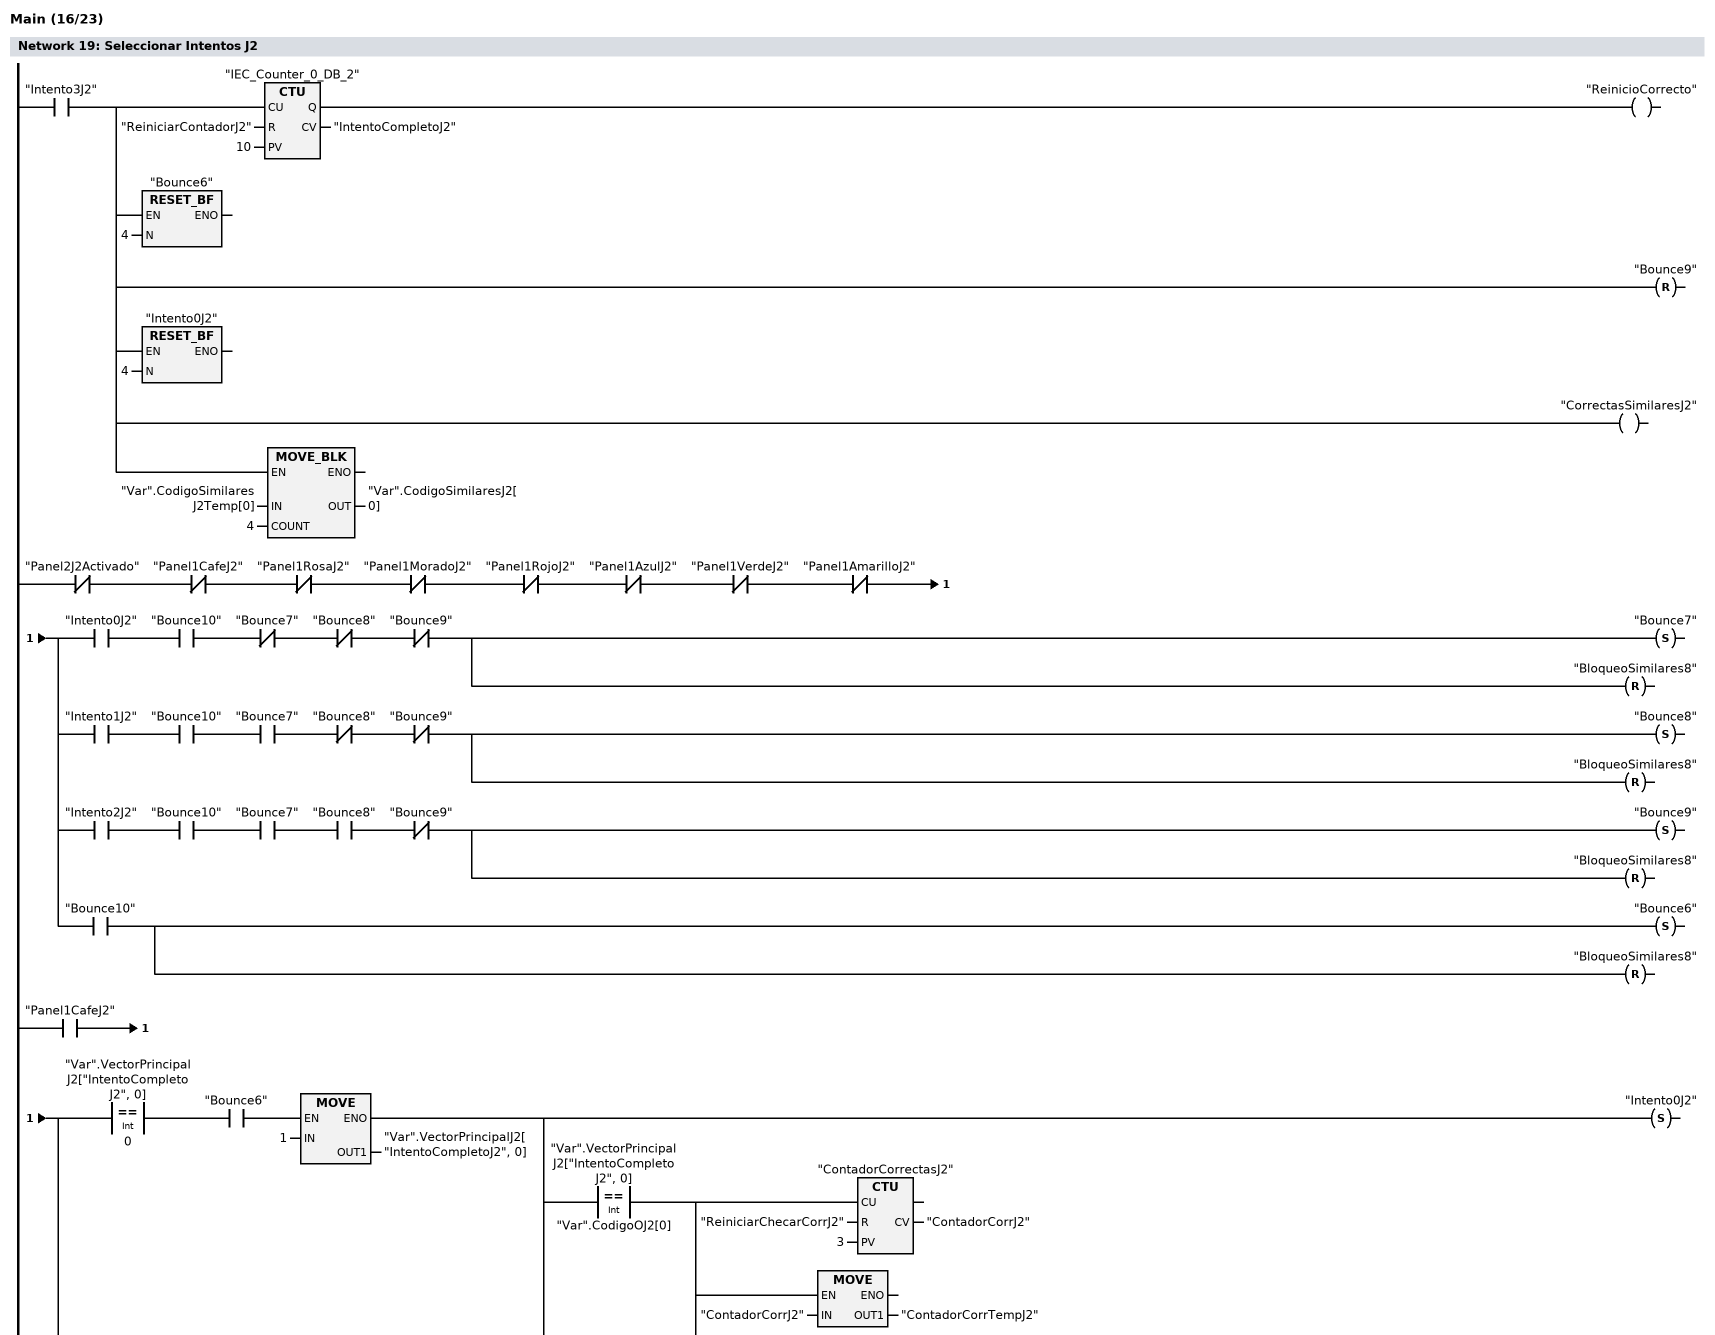
